REGION Network 16: Call the Event Manager logic for EM alarms
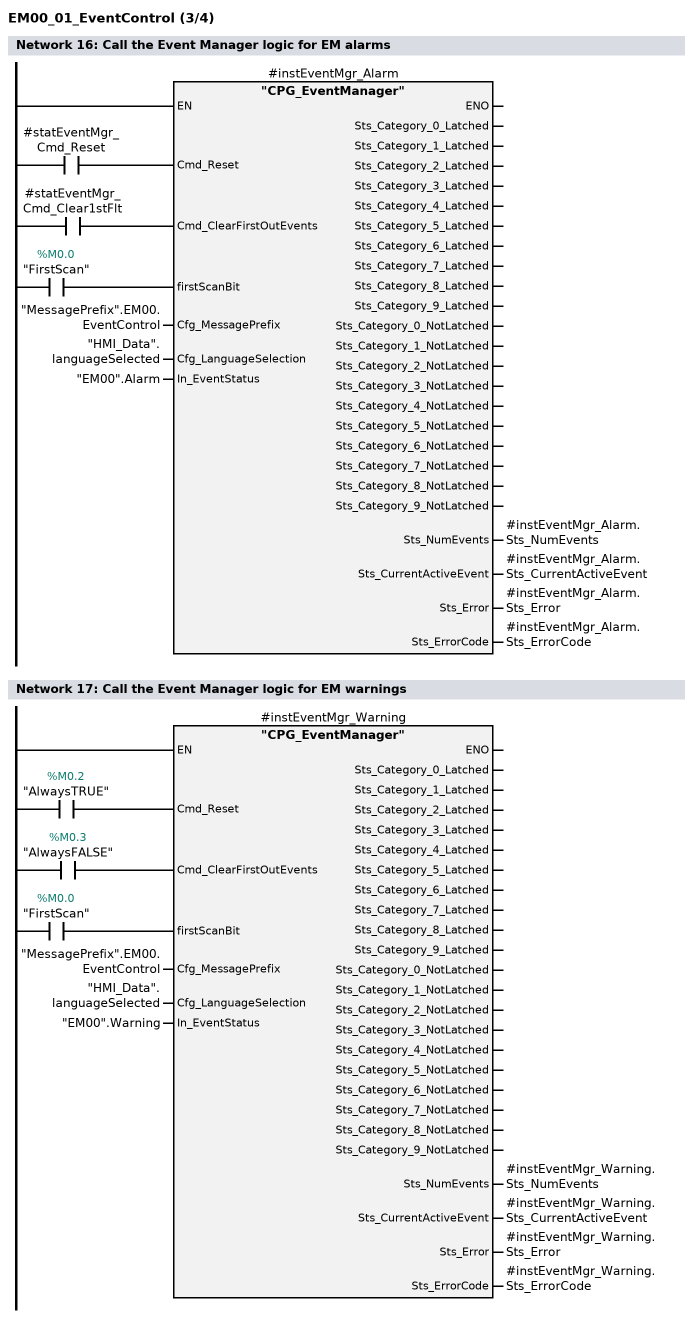
   RUNG wire#powerrail
      #instEventMgr_Alarm(Cmd_Reset := wire#w1, Cmd_ClearFirstOutEvents := wire#w2, firstScanBit := wire#w3, Cfg_MessagePrefix := "MessagePrefix".EM00.EventControl, Cfg_LanguageSelection := "HMI_Data".languageSelected, In_EventStatus := "EM00".Alarm, Sts_Category_0_Latched =>, Sts_Category_1_Latched =>, Sts_Category_2_Latched =>, Sts_Category_3_Latched =>, Sts_Category_4_Latched =>, Sts_Category_5_Latched =>, Sts_Category_6_Latched =>, Sts_Category_7_Latched =>, Sts_Category_8_Latched =>, Sts_Category_9_Latched =>, Sts_Category_0_NotLatched =>, Sts_Category_1_NotLatched =>, Sts_Category_2_NotLatched =>, Sts_Category_3_NotLatched =>, Sts_Category_4_NotLatched =>, Sts_Category_5_NotLatched =>, Sts_Category_6_NotLatched =>, Sts_Category_7_NotLatched =>, Sts_Category_8_NotLatched =>, Sts_Category_9_NotLatched =>, Sts_NumEvents => #instEventMgr_Alarm.Sts_NumEvents, Sts_CurrentActiveEvent => #instEventMgr_Alarm.Sts_CurrentActiveEvent, Sts_Error => #instEventMgr_Alarm.Sts_Error, Sts_ErrorCode => #instEventMgr_Alarm.Sts_ErrorCode)
   END_RUNG
   RUNG wire#powerrail
      Contact( #statEventMgr_Cmd_Reset )
   END_RUNG wire#w1
   RUNG wire#powerrail
      Contact( #statEventMgr_Cmd_Clear1stFlt )
   END_RUNG wire#w2
   RUNG wire#powerrail
      Contact( "FirstScan" )
   END_RUNG wire#w3
   // the same network as SCL:
   #instEventMgr_Alarm(Cmd_Reset := #statEventMgr_Cmd_Reset,   // "CPG_EventManager"
                       Cmd_ClearFirstOutEvents := #statEventMgr_Cmd_Clear1stFlt,
                       firstScanBit := "FirstScan",
                       Cfg_MessagePrefix := "MessagePrefix".EM00.EventControl,
                       Cfg_LanguageSelection := "HMI_Data".languageSelected,
                       In_EventStatus := "EM00".Alarm,
                       Sts_NumEvents => #instEventMgr_Alarm.Sts_NumEvents,
                       Sts_CurrentActiveEvent => #instEventMgr_Alarm.Sts_CurrentActiveEvent,
                       Sts_Error => #instEventMgr_Alarm.Sts_Error,
                       Sts_ErrorCode => #instEventMgr_Alarm.Sts_ErrorCode);
END_REGION

REGION Network 17: Call the Event Manager logic for EM warnings
   RUNG wire#powerrail
      #instEventMgr_Warning(Cmd_Reset := wire#w1, Cmd_ClearFirstOutEvents := wire#w2, firstScanBit := wire#w3, Cfg_MessagePrefix := "MessagePrefix".EM00.EventControl, Cfg_LanguageSelection := "HMI_Data".languageSelected, In_EventStatus := "EM00".Warning, Sts_Category_0_Latched =>, Sts_Category_1_Latched =>, Sts_Category_2_Latched =>, Sts_Category_3_Latched =>, Sts_Category_4_Latched =>, Sts_Category_5_Latched =>, Sts_Category_6_Latched =>, Sts_Category_7_Latched =>, Sts_Category_8_Latched =>, Sts_Category_9_Latched =>, Sts_Category_0_NotLatched =>, Sts_Category_1_NotLatched =>, Sts_Category_2_NotLatched =>, Sts_Category_3_NotLatched =>, Sts_Category_4_NotLatched =>, Sts_Category_5_NotLatched =>, Sts_Category_6_NotLatched =>, Sts_Category_7_NotLatched =>, Sts_Category_8_NotLatched =>, Sts_Category_9_NotLatched =>, Sts_NumEvents => #instEventMgr_Warning.Sts_NumEvents, Sts_CurrentActiveEvent => #instEventMgr_Warning.Sts_CurrentActiveEvent, Sts_Error => #instEventMgr_Warning.Sts_Error, Sts_ErrorCode => #instEventMgr_Warning.Sts_ErrorCode)
   END_RUNG
   RUNG wire#powerrail
      Contact( "AlwaysTRUE" )
   END_RUNG wire#w1
   RUNG wire#powerrail
      Contact( "AlwaysFALSE" )
   END_RUNG wire#w2
   RUNG wire#powerrail
      Contact( "FirstScan" )
   END_RUNG wire#w3
   // the same network as SCL:
   #instEventMgr_Warning(Cmd_Reset := "AlwaysTRUE",   // "CPG_EventManager"
                         Cmd_ClearFirstOutEvents := "AlwaysFALSE",
                         firstScanBit := "FirstScan",
                         Cfg_MessagePrefix := "MessagePrefix".EM00.EventControl,
                         Cfg_LanguageSelection := "HMI_Data".languageSelected,
                         In_EventStatus := "EM00".Warning,
                         Sts_NumEvents => #instEventMgr_Warning.Sts_NumEvents,
                         Sts_CurrentActiveEvent => #instEventMgr_Warning.Sts_CurrentActiveEvent,
                         Sts_Error => #instEventMgr_Warning.Sts_Error,
                         Sts_ErrorCode => #instEventMgr_Warning.Sts_ErrorCode);
END_REGION

REGION Network 18: Call the Event Manager logic for EM status
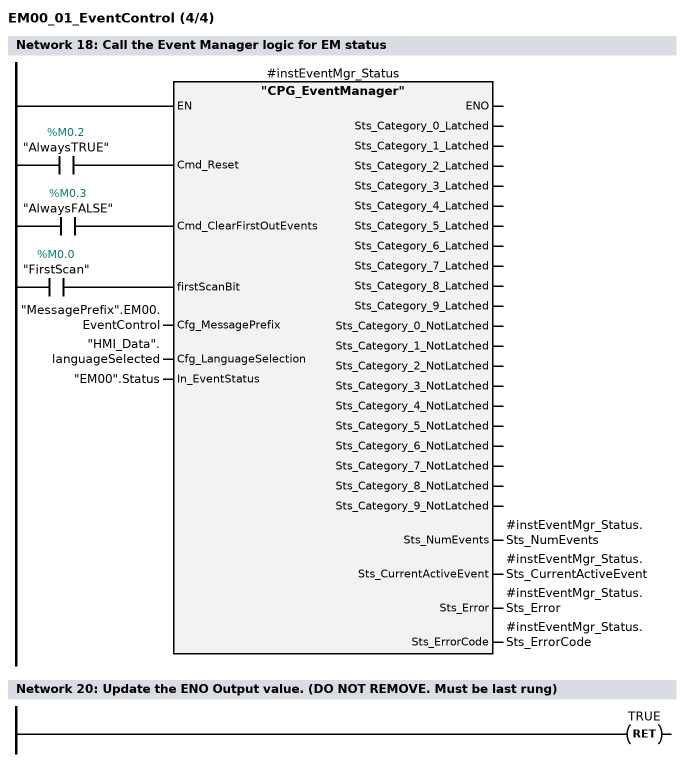
   RUNG wire#powerrail
      #instEventMgr_Status(Cmd_Reset := wire#w1, Cmd_ClearFirstOutEvents := wire#w2, firstScanBit := wire#w3, Cfg_MessagePrefix := "MessagePrefix".EM00.EventControl, Cfg_LanguageSelection := "HMI_Data".languageSelected, In_EventStatus := "EM00".Status, Sts_Category_0_Latched =>, Sts_Category_1_Latched =>, Sts_Category_2_Latched =>, Sts_Category_3_Latched =>, Sts_Category_4_Latched =>, Sts_Category_5_Latched =>, Sts_Category_6_Latched =>, Sts_Category_7_Latched =>, Sts_Category_8_Latched =>, Sts_Category_9_Latched =>, Sts_Category_0_NotLatched =>, Sts_Category_1_NotLatched =>, Sts_Category_2_NotLatched =>, Sts_Category_3_NotLatched =>, Sts_Category_4_NotLatched =>, Sts_Category_5_NotLatched =>, Sts_Category_6_NotLatched =>, Sts_Category_7_NotLatched =>, Sts_Category_8_NotLatched =>, Sts_Category_9_NotLatched =>, Sts_NumEvents => #instEventMgr_Status.Sts_NumEvents, Sts_CurrentActiveEvent => #instEventMgr_Status.Sts_CurrentActiveEvent, Sts_Error => #instEventMgr_Status.Sts_Error, Sts_ErrorCode => #instEventMgr_Status.Sts_ErrorCode)
   END_RUNG
   RUNG wire#powerrail
      Contact( "AlwaysTRUE" )
   END_RUNG wire#w1
   RUNG wire#powerrail
      Contact( "AlwaysFALSE" )
   END_RUNG wire#w2
   RUNG wire#powerrail
      Contact( "FirstScan" )
   END_RUNG wire#w3
   // the same network as SCL:
   #instEventMgr_Status(Cmd_Reset := "AlwaysTRUE",   // "CPG_EventManager"
                        Cmd_ClearFirstOutEvents := "AlwaysFALSE",
                        firstScanBit := "FirstScan",
                        Cfg_MessagePrefix := "MessagePrefix".EM00.EventControl,
                        Cfg_LanguageSelection := "HMI_Data".languageSelected,
                        In_EventStatus := "EM00".Status,
                        Sts_NumEvents => #instEventMgr_Status.Sts_NumEvents,
                        Sts_CurrentActiveEvent => #instEventMgr_Status.Sts_CurrentActiveEvent,
                        Sts_Error => #instEventMgr_Status.Sts_Error,
                        Sts_ErrorCode => #instEventMgr_Status.Sts_ErrorCode);
END_REGION

REGION Network 20: Update the ENO Output value. (DO NOT REMOVE. Must be last rung)
   RUNG wire#powerrail
      ReturnCoil( TRUE )
   END_RUNG
   // the same network as SCL:
   ENO := TRUE;
   RETURN;
END_REGION
END_FUNCTION_BLOCK

FUNCTION_BLOCK "EM00_02_PackML_ModuleSum"   // FB31642, LAD
TITLE = EM00_02_PackML_ModuleSummation
{ S7_Optimized_Access := 'TRUE' }
AUTHOR : tech.team.motioncontrol@siemens.com
FAMILY : CPG
VERSION : 1.1
// Support: tech.team.motioncontrol@siemens.com
// stored: AutoNumber true, IsIECCheckEnabled false, IsRetainMemResEnabled false, MemoryReserve 100, SetENOAutomatically false, UDAEnableTagReadback false
   VAR
      statDummyBool { ExternalAccessible := 'False'; ExternalVisible := 'False'; ExternalWritable := 'False'} : Bool;   // dummy bool - placeholder
   END_VAR
BEGIN

REGION Network 1: EM - Reset Command
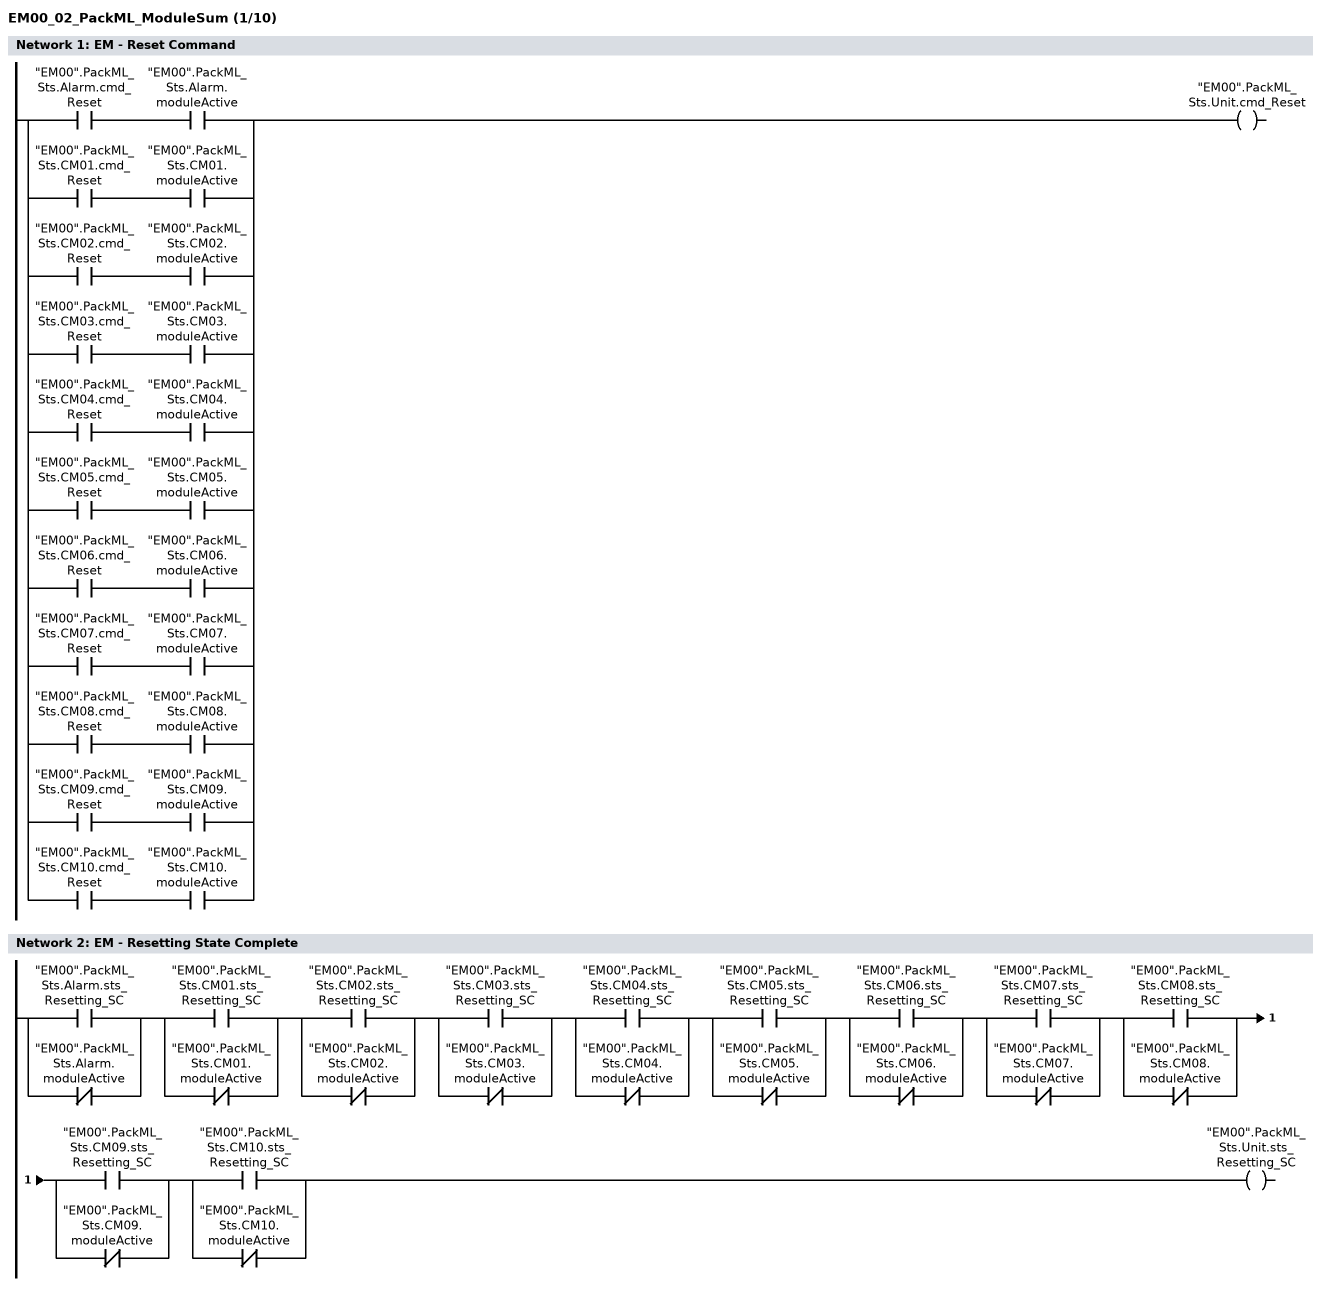
   RUNG wire#powerrail
      Contact( "EM00".PackML_Sts.Alarm.cmd_Reset )
      Contact( "EM00".PackML_Sts.Alarm.moduleActive )
      wire#w1
      Coil( "EM00".PackML_Sts.Unit.cmd_Reset )
   END_RUNG
   RUNG wire#powerrail
      Contact( "EM00".PackML_Sts.CM01.cmd_Reset )
      Contact( "EM00".PackML_Sts.CM01.moduleActive )
   END_RUNG wire#w1
   RUNG wire#powerrail
      Contact( "EM00".PackML_Sts.CM02.cmd_Reset )
      Contact( "EM00".PackML_Sts.CM02.moduleActive )
   END_RUNG wire#w1
   RUNG wire#powerrail
      Contact( "EM00".PackML_Sts.CM03.cmd_Reset )
      Contact( "EM00".PackML_Sts.CM03.moduleActive )
   END_RUNG wire#w1
   RUNG wire#powerrail
      Contact( "EM00".PackML_Sts.CM04.cmd_Reset )
      Contact( "EM00".PackML_Sts.CM04.moduleActive )
   END_RUNG wire#w1
   RUNG wire#powerrail
      Contact( "EM00".PackML_Sts.CM05.cmd_Reset )
      Contact( "EM00".PackML_Sts.CM05.moduleActive )
   END_RUNG wire#w1
   RUNG wire#powerrail
      Contact( "EM00".PackML_Sts.CM06.cmd_Reset )
      Contact( "EM00".PackML_Sts.CM06.moduleActive )
   END_RUNG wire#w1
   RUNG wire#powerrail
      Contact( "EM00".PackML_Sts.CM07.cmd_Reset )
      Contact( "EM00".PackML_Sts.CM07.moduleActive )
   END_RUNG wire#w1
   RUNG wire#powerrail
      Contact( "EM00".PackML_Sts.CM08.cmd_Reset )
      Contact( "EM00".PackML_Sts.CM08.moduleActive )
   END_RUNG wire#w1
   RUNG wire#powerrail
      Contact( "EM00".PackML_Sts.CM09.cmd_Reset )
      Contact( "EM00".PackML_Sts.CM09.moduleActive )
   END_RUNG wire#w1
   RUNG wire#powerrail
      Contact( "EM00".PackML_Sts.CM10.cmd_Reset )
      Contact( "EM00".PackML_Sts.CM10.moduleActive )
   END_RUNG wire#w1
   // the same network as SCL:
   "EM00".PackML_Sts.Unit.cmd_Reset := ("EM00".PackML_Sts.Alarm.cmd_Reset AND "EM00".PackML_Sts.Alarm.moduleActive) OR ("EM00".PackML_Sts.CM01.cmd_Reset AND "EM00".PackML_Sts.CM01.moduleActive) OR ("EM00".PackML_Sts.CM02.cmd_Reset AND "EM00".PackML_Sts.CM02.moduleActive) OR ("EM00".PackML_Sts.CM03.cmd_Reset AND "EM00".PackML_Sts.CM03.moduleActive) OR ("EM00".PackML_Sts.CM04.cmd_Reset AND "EM00".PackML_Sts.CM04.moduleActive) OR ("EM00".PackML_Sts.CM05.cmd_Reset AND "EM00".PackML_Sts.CM05.moduleActive) OR ("EM00".PackML_Sts.CM06.cmd_Reset AND "EM00".PackML_Sts.CM06.moduleActive) OR ("EM00".PackML_Sts.CM07.cmd_Reset AND "EM00".PackML_Sts.CM07.moduleActive) OR ("EM00".PackML_Sts.CM08.cmd_Reset AND "EM00".PackML_Sts.CM08.moduleActive) OR ("EM00".PackML_Sts.CM09.cmd_Reset AND "EM00".PackML_Sts.CM09.moduleActive) OR ("EM00".PackML_Sts.CM10.cmd_Reset AND "EM00".PackML_Sts.CM10.moduleActive);
END_REGION

REGION Network 2: EM - Resetting State Complete
   RUNG wire#powerrail
      Contact( "EM00".PackML_Sts.Alarm.sts_Resetting_SC )
      wire#w1
      Contact( "EM00".PackML_Sts.CM01.sts_Resetting_SC )
      wire#w2
      Contact( "EM00".PackML_Sts.CM02.sts_Resetting_SC )
      wire#w3
      Contact( "EM00".PackML_Sts.CM03.sts_Resetting_SC )
      wire#w4
      Contact( "EM00".PackML_Sts.CM04.sts_Resetting_SC )
      wire#w5
      Contact( "EM00".PackML_Sts.CM05.sts_Resetting_SC )
      wire#w6
      Contact( "EM00".PackML_Sts.CM06.sts_Resetting_SC )
      wire#w7
      Contact( "EM00".PackML_Sts.CM07.sts_Resetting_SC )
      wire#w8
      Contact( "EM00".PackML_Sts.CM08.sts_Resetting_SC )
      wire#w9
      Contact( "EM00".PackML_Sts.CM09.sts_Resetting_SC )
      wire#w10
      Contact( "EM00".PackML_Sts.CM10.sts_Resetting_SC )
      wire#w11
      Coil( "EM00".PackML_Sts.Unit.sts_Resetting_SC )
   END_RUNG
   RUNG wire#powerrail
      I_Contact( "EM00".PackML_Sts.Alarm.moduleActive )
   END_RUNG wire#w1
   RUNG wire#w1
      I_Contact( "EM00".PackML_Sts.CM01.moduleActive )
   END_RUNG wire#w2
   RUNG wire#w2
      I_Contact( "EM00".PackML_Sts.CM02.moduleActive )
   END_RUNG wire#w3
   RUNG wire#w3
      I_Contact( "EM00".PackML_Sts.CM03.moduleActive )
   END_RUNG wire#w4
   RUNG wire#w4
      I_Contact( "EM00".PackML_Sts.CM04.moduleActive )
   END_RUNG wire#w5
   RUNG wire#w5
      I_Contact( "EM00".PackML_Sts.CM05.moduleActive )
   END_RUNG wire#w6
   RUNG wire#w6
      I_Contact( "EM00".PackML_Sts.CM06.moduleActive )
   END_RUNG wire#w7
   RUNG wire#w7
      I_Contact( "EM00".PackML_Sts.CM07.moduleActive )
   END_RUNG wire#w8
   RUNG wire#w8
      I_Contact( "EM00".PackML_Sts.CM08.moduleActive )
   END_RUNG wire#w9
   RUNG wire#w9
      I_Contact( "EM00".PackML_Sts.CM09.moduleActive )
   END_RUNG wire#w10
   RUNG wire#w10
      I_Contact( "EM00".PackML_Sts.CM10.moduleActive )
   END_RUNG wire#w11
   // the same network as SCL:
   "EM00".PackML_Sts.Unit.sts_Resetting_SC := ("EM00".PackML_Sts.Alarm.sts_Resetting_SC OR NOT "EM00".PackML_Sts.Alarm.moduleActive) AND ("EM00".PackML_Sts.CM01.sts_Resetting_SC OR NOT "EM00".PackML_Sts.CM01.moduleActive) AND ("EM00".PackML_Sts.CM02.sts_Resetting_SC OR NOT "EM00".PackML_Sts.CM02.moduleActive) AND ("EM00".PackML_Sts.CM03.sts_Resetting_SC OR NOT "EM00".PackML_Sts.CM03.moduleActive) AND ("EM00".PackML_Sts.CM04.sts_Resetting_SC OR NOT "EM00".PackML_Sts.CM04.moduleActive) AND ("EM00".PackML_Sts.CM05.sts_Resetting_SC OR NOT "EM00".PackML_Sts.CM05.moduleActive) AND ("EM00".PackML_Sts.CM06.sts_Resetting_SC OR NOT "EM00".PackML_Sts.CM06.moduleActive) AND ("EM00".PackML_Sts.CM07.sts_Resetting_SC OR NOT "EM00".PackML_Sts.CM07.moduleActive) AND ("EM00".PackML_Sts.CM08.sts_Resetting_SC OR NOT "EM00".PackML_Sts.CM08.moduleActive) AND ("EM00".PackML_Sts.CM09.sts_Resetting_SC OR NOT "EM00".PackML_Sts.CM09.moduleActive) AND ("EM00".PackML_Sts.CM10.sts_Resetting_SC OR NOT "EM00".PackML_Sts.CM10.moduleActive);
END_REGION

REGION Network 3: EM - Start Command
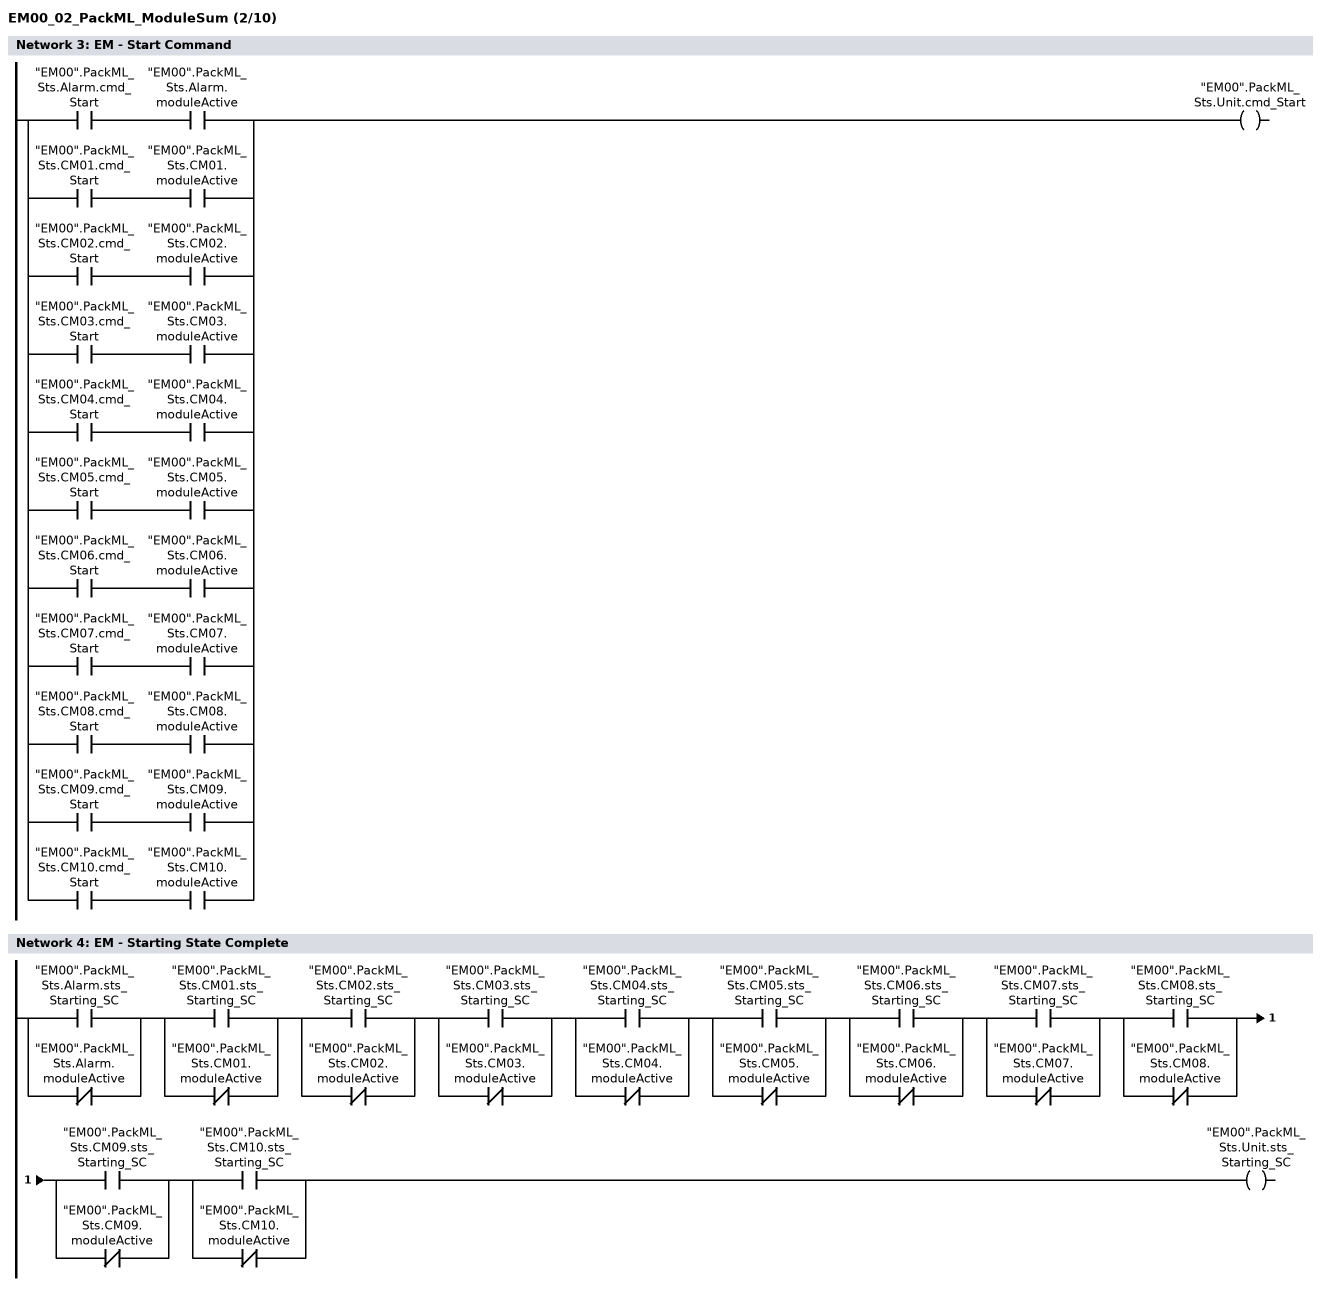
   RUNG wire#powerrail
      Contact( "EM00".PackML_Sts.Alarm.cmd_Start )
      Contact( "EM00".PackML_Sts.Alarm.moduleActive )
      wire#w1
      Coil( "EM00".PackML_Sts.Unit.cmd_Start )
   END_RUNG
   RUNG wire#powerrail
      Contact( "EM00".PackML_Sts.CM01.cmd_Start )
      Contact( "EM00".PackML_Sts.CM01.moduleActive )
   END_RUNG wire#w1
   RUNG wire#powerrail
      Contact( "EM00".PackML_Sts.CM02.cmd_Start )
      Contact( "EM00".PackML_Sts.CM02.moduleActive )
   END_RUNG wire#w1
   RUNG wire#powerrail
      Contact( "EM00".PackML_Sts.CM03.cmd_Start )
      Contact( "EM00".PackML_Sts.CM03.moduleActive )
   END_RUNG wire#w1
   RUNG wire#powerrail
      Contact( "EM00".PackML_Sts.CM04.cmd_Start )
      Contact( "EM00".PackML_Sts.CM04.moduleActive )
   END_RUNG wire#w1
   RUNG wire#powerrail
      Contact( "EM00".PackML_Sts.CM05.cmd_Start )
      Contact( "EM00".PackML_Sts.CM05.moduleActive )
   END_RUNG wire#w1
   RUNG wire#powerrail
      Contact( "EM00".PackML_Sts.CM06.cmd_Start )
      Contact( "EM00".PackML_Sts.CM06.moduleActive )
   END_RUNG wire#w1
   RUNG wire#powerrail
      Contact( "EM00".PackML_Sts.CM07.cmd_Start )
      Contact( "EM00".PackML_Sts.CM07.moduleActive )
   END_RUNG wire#w1
   RUNG wire#powerrail
      Contact( "EM00".PackML_Sts.CM08.cmd_Start )
      Contact( "EM00".PackML_Sts.CM08.moduleActive )
   END_RUNG wire#w1
   RUNG wire#powerrail
      Contact( "EM00".PackML_Sts.CM09.cmd_Start )
      Contact( "EM00".PackML_Sts.CM09.moduleActive )
   END_RUNG wire#w1
   RUNG wire#powerrail
      Contact( "EM00".PackML_Sts.CM10.cmd_Start )
      Contact( "EM00".PackML_Sts.CM10.moduleActive )
   END_RUNG wire#w1
   // the same network as SCL:
   "EM00".PackML_Sts.Unit.cmd_Start := ("EM00".PackML_Sts.Alarm.cmd_Start AND "EM00".PackML_Sts.Alarm.moduleActive) OR ("EM00".PackML_Sts.CM01.cmd_Start AND "EM00".PackML_Sts.CM01.moduleActive) OR ("EM00".PackML_Sts.CM02.cmd_Start AND "EM00".PackML_Sts.CM02.moduleActive) OR ("EM00".PackML_Sts.CM03.cmd_Start AND "EM00".PackML_Sts.CM03.moduleActive) OR ("EM00".PackML_Sts.CM04.cmd_Start AND "EM00".PackML_Sts.CM04.moduleActive) OR ("EM00".PackML_Sts.CM05.cmd_Start AND "EM00".PackML_Sts.CM05.moduleActive) OR ("EM00".PackML_Sts.CM06.cmd_Start AND "EM00".PackML_Sts.CM06.moduleActive) OR ("EM00".PackML_Sts.CM07.cmd_Start AND "EM00".PackML_Sts.CM07.moduleActive) OR ("EM00".PackML_Sts.CM08.cmd_Start AND "EM00".PackML_Sts.CM08.moduleActive) OR ("EM00".PackML_Sts.CM09.cmd_Start AND "EM00".PackML_Sts.CM09.moduleActive) OR ("EM00".PackML_Sts.CM10.cmd_Start AND "EM00".PackML_Sts.CM10.moduleActive);
END_REGION

REGION Network 4: EM - Starting State Complete
   RUNG wire#powerrail
      Contact( "EM00".PackML_Sts.Alarm.sts_Starting_SC )
      wire#w1
      Contact( "EM00".PackML_Sts.CM01.sts_Starting_SC )
      wire#w2
      Contact( "EM00".PackML_Sts.CM02.sts_Starting_SC )
      wire#w3
      Contact( "EM00".PackML_Sts.CM03.sts_Starting_SC )
      wire#w4
      Contact( "EM00".PackML_Sts.CM04.sts_Starting_SC )
      wire#w5
      Contact( "EM00".PackML_Sts.CM05.sts_Starting_SC )
      wire#w6
      Contact( "EM00".PackML_Sts.CM06.sts_Starting_SC )
      wire#w7
      Contact( "EM00".PackML_Sts.CM07.sts_Starting_SC )
      wire#w8
      Contact( "EM00".PackML_Sts.CM08.sts_Starting_SC )
      wire#w9
      Contact( "EM00".PackML_Sts.CM09.sts_Starting_SC )
      wire#w10
      Contact( "EM00".PackML_Sts.CM10.sts_Starting_SC )
      wire#w11
      Coil( "EM00".PackML_Sts.Unit.sts_Starting_SC )
   END_RUNG
   RUNG wire#powerrail
      I_Contact( "EM00".PackML_Sts.Alarm.moduleActive )
   END_RUNG wire#w1
   RUNG wire#w1
      I_Contact( "EM00".PackML_Sts.CM01.moduleActive )
   END_RUNG wire#w2
   RUNG wire#w2
      I_Contact( "EM00".PackML_Sts.CM02.moduleActive )
   END_RUNG wire#w3
   RUNG wire#w3
      I_Contact( "EM00".PackML_Sts.CM03.moduleActive )
   END_RUNG wire#w4
   RUNG wire#w4
      I_Contact( "EM00".PackML_Sts.CM04.moduleActive )
   END_RUNG wire#w5
   RUNG wire#w5
      I_Contact( "EM00".PackML_Sts.CM05.moduleActive )
   END_RUNG wire#w6
   RUNG wire#w6
      I_Contact( "EM00".PackML_Sts.CM06.moduleActive )
   END_RUNG wire#w7
   RUNG wire#w7
      I_Contact( "EM00".PackML_Sts.CM07.moduleActive )
   END_RUNG wire#w8
   RUNG wire#w8
      I_Contact( "EM00".PackML_Sts.CM08.moduleActive )
   END_RUNG wire#w9
   RUNG wire#w9
      I_Contact( "EM00".PackML_Sts.CM09.moduleActive )
   END_RUNG wire#w10
   RUNG wire#w10
      I_Contact( "EM00".PackML_Sts.CM10.moduleActive )
   END_RUNG wire#w11
   // the same network as SCL:
   "EM00".PackML_Sts.Unit.sts_Starting_SC := ("EM00".PackML_Sts.Alarm.sts_Starting_SC OR NOT "EM00".PackML_Sts.Alarm.moduleActive) AND ("EM00".PackML_Sts.CM01.sts_Starting_SC OR NOT "EM00".PackML_Sts.CM01.moduleActive) AND ("EM00".PackML_Sts.CM02.sts_Starting_SC OR NOT "EM00".PackML_Sts.CM02.moduleActive) AND ("EM00".PackML_Sts.CM03.sts_Starting_SC OR NOT "EM00".PackML_Sts.CM03.moduleActive) AND ("EM00".PackML_Sts.CM04.sts_Starting_SC OR NOT "EM00".PackML_Sts.CM04.moduleActive) AND ("EM00".PackML_Sts.CM05.sts_Starting_SC OR NOT "EM00".PackML_Sts.CM05.moduleActive) AND ("EM00".PackML_Sts.CM06.sts_Starting_SC OR NOT "EM00".PackML_Sts.CM06.moduleActive) AND ("EM00".PackML_Sts.CM07.sts_Starting_SC OR NOT "EM00".PackML_Sts.CM07.moduleActive) AND ("EM00".PackML_Sts.CM08.sts_Starting_SC OR NOT "EM00".PackML_Sts.CM08.moduleActive) AND ("EM00".PackML_Sts.CM09.sts_Starting_SC OR NOT "EM00".PackML_Sts.CM09.moduleActive) AND ("EM00".PackML_Sts.CM10.sts_Starting_SC OR NOT "EM00".PackML_Sts.CM10.moduleActive);
END_REGION

REGION Network 5: EM - Stop Command
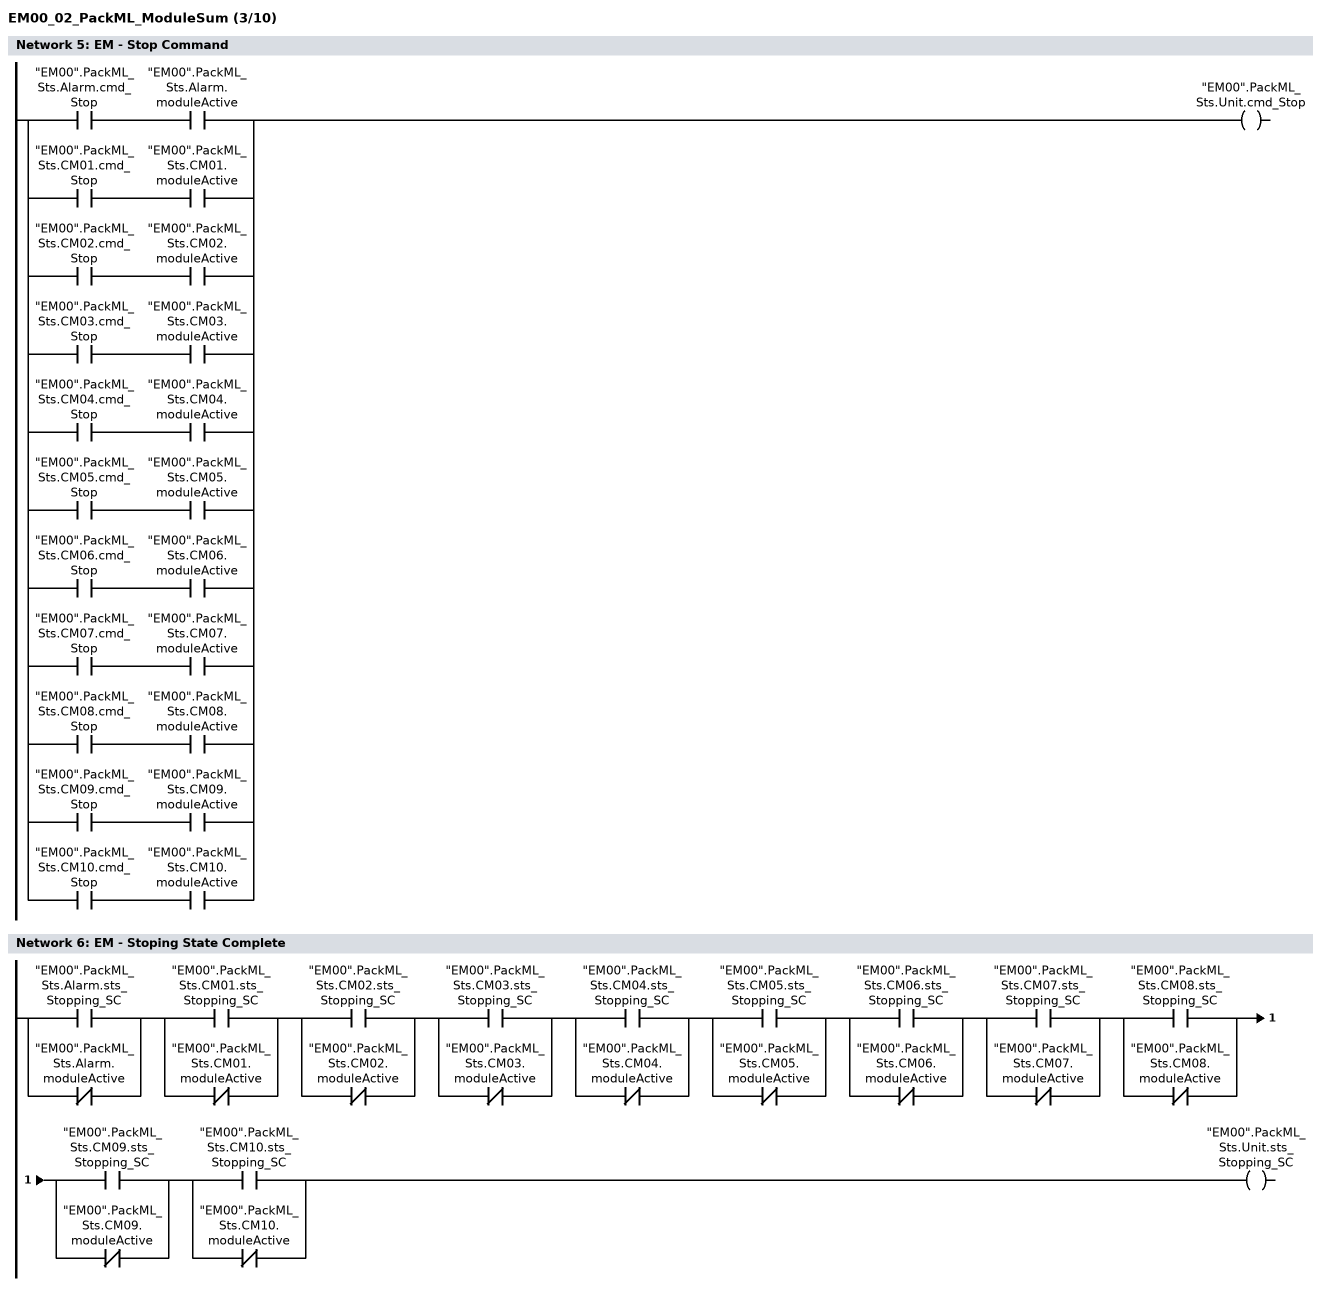
   RUNG wire#powerrail
      Contact( "EM00".PackML_Sts.Alarm.cmd_Stop )
      Contact( "EM00".PackML_Sts.Alarm.moduleActive )
      wire#w1
      Coil( "EM00".PackML_Sts.Unit.cmd_Stop )
   END_RUNG
   RUNG wire#powerrail
      Contact( "EM00".PackML_Sts.CM01.cmd_Stop )
      Contact( "EM00".PackML_Sts.CM01.moduleActive )
   END_RUNG wire#w1
   RUNG wire#powerrail
      Contact( "EM00".PackML_Sts.CM02.cmd_Stop )
      Contact( "EM00".PackML_Sts.CM02.moduleActive )
   END_RUNG wire#w1
   RUNG wire#powerrail
      Contact( "EM00".PackML_Sts.CM03.cmd_Stop )
      Contact( "EM00".PackML_Sts.CM03.moduleActive )
   END_RUNG wire#w1
   RUNG wire#powerrail
      Contact( "EM00".PackML_Sts.CM04.cmd_Stop )
      Contact( "EM00".PackML_Sts.CM04.moduleActive )
   END_RUNG wire#w1
   RUNG wire#powerrail
      Contact( "EM00".PackML_Sts.CM05.cmd_Stop )
      Contact( "EM00".PackML_Sts.CM05.moduleActive )
   END_RUNG wire#w1
   RUNG wire#powerrail
      Contact( "EM00".PackML_Sts.CM06.cmd_Stop )
      Contact( "EM00".PackML_Sts.CM06.moduleActive )
   END_RUNG wire#w1
   RUNG wire#powerrail
      Contact( "EM00".PackML_Sts.CM07.cmd_Stop )
      Contact( "EM00".PackML_Sts.CM07.moduleActive )
   END_RUNG wire#w1
   RUNG wire#powerrail
      Contact( "EM00".PackML_Sts.CM08.cmd_Stop )
      Contact( "EM00".PackML_Sts.CM08.moduleActive )
   END_RUNG wire#w1
   RUNG wire#powerrail
      Contact( "EM00".PackML_Sts.CM09.cmd_Stop )
      Contact( "EM00".PackML_Sts.CM09.moduleActive )
   END_RUNG wire#w1
   RUNG wire#powerrail
      Contact( "EM00".PackML_Sts.CM10.cmd_Stop )
      Contact( "EM00".PackML_Sts.CM10.moduleActive )
   END_RUNG wire#w1
   // the same network as SCL:
   "EM00".PackML_Sts.Unit.cmd_Stop := ("EM00".PackML_Sts.Alarm.cmd_Stop AND "EM00".PackML_Sts.Alarm.moduleActive) OR ("EM00".PackML_Sts.CM01.cmd_Stop AND "EM00".PackML_Sts.CM01.moduleActive) OR ("EM00".PackML_Sts.CM02.cmd_Stop AND "EM00".PackML_Sts.CM02.moduleActive) OR ("EM00".PackML_Sts.CM03.cmd_Stop AND "EM00".PackML_Sts.CM03.moduleActive) OR ("EM00".PackML_Sts.CM04.cmd_Stop AND "EM00".PackML_Sts.CM04.moduleActive) OR ("EM00".PackML_Sts.CM05.cmd_Stop AND "EM00".PackML_Sts.CM05.moduleActive) OR ("EM00".PackML_Sts.CM06.cmd_Stop AND "EM00".PackML_Sts.CM06.moduleActive) OR ("EM00".PackML_Sts.CM07.cmd_Stop AND "EM00".PackML_Sts.CM07.moduleActive) OR ("EM00".PackML_Sts.CM08.cmd_Stop AND "EM00".PackML_Sts.CM08.moduleActive) OR ("EM00".PackML_Sts.CM09.cmd_Stop AND "EM00".PackML_Sts.CM09.moduleActive) OR ("EM00".PackML_Sts.CM10.cmd_Stop AND "EM00".PackML_Sts.CM10.moduleActive);
END_REGION

REGION Network 6: EM - Stoping State Complete
   RUNG wire#powerrail
      Contact( "EM00".PackML_Sts.Alarm.sts_Stopping_SC )
      wire#w1
      Contact( "EM00".PackML_Sts.CM01.sts_Stopping_SC )
      wire#w2
      Contact( "EM00".PackML_Sts.CM02.sts_Stopping_SC )
      wire#w3
      Contact( "EM00".PackML_Sts.CM03.sts_Stopping_SC )
      wire#w4
      Contact( "EM00".PackML_Sts.CM04.sts_Stopping_SC )
      wire#w5
      Contact( "EM00".PackML_Sts.CM05.sts_Stopping_SC )
      wire#w6
      Contact( "EM00".PackML_Sts.CM06.sts_Stopping_SC )
      wire#w7
      Contact( "EM00".PackML_Sts.CM07.sts_Stopping_SC )
      wire#w8
      Contact( "EM00".PackML_Sts.CM08.sts_Stopping_SC )
      wire#w9
      Contact( "EM00".PackML_Sts.CM09.sts_Stopping_SC )
      wire#w10
      Contact( "EM00".PackML_Sts.CM10.sts_Stopping_SC )
      wire#w11
      Coil( "EM00".PackML_Sts.Unit.sts_Stopping_SC )
   END_RUNG
   RUNG wire#powerrail
      I_Contact( "EM00".PackML_Sts.Alarm.moduleActive )
   END_RUNG wire#w1
   RUNG wire#w1
      I_Contact( "EM00".PackML_Sts.CM01.moduleActive )
   END_RUNG wire#w2
   RUNG wire#w2
      I_Contact( "EM00".PackML_Sts.CM02.moduleActive )
   END_RUNG wire#w3
   RUNG wire#w3
      I_Contact( "EM00".PackML_Sts.CM03.moduleActive )
   END_RUNG wire#w4
   RUNG wire#w4
      I_Contact( "EM00".PackML_Sts.CM04.moduleActive )
   END_RUNG wire#w5
   RUNG wire#w5
      I_Contact( "EM00".PackML_Sts.CM05.moduleActive )
   END_RUNG wire#w6
   RUNG wire#w6
      I_Contact( "EM00".PackML_Sts.CM06.moduleActive )
   END_RUNG wire#w7
   RUNG wire#w7
      I_Contact( "EM00".PackML_Sts.CM07.moduleActive )
   END_RUNG wire#w8
   RUNG wire#w8
      I_Contact( "EM00".PackML_Sts.CM08.moduleActive )
   END_RUNG wire#w9
   RUNG wire#w9
      I_Contact( "EM00".PackML_Sts.CM09.moduleActive )
   END_RUNG wire#w10
   RUNG wire#w10
      I_Contact( "EM00".PackML_Sts.CM10.moduleActive )
   END_RUNG wire#w11
   // the same network as SCL:
   "EM00".PackML_Sts.Unit.sts_Stopping_SC := ("EM00".PackML_Sts.Alarm.sts_Stopping_SC OR NOT "EM00".PackML_Sts.Alarm.moduleActive) AND ("EM00".PackML_Sts.CM01.sts_Stopping_SC OR NOT "EM00".PackML_Sts.CM01.moduleActive) AND ("EM00".PackML_Sts.CM02.sts_Stopping_SC OR NOT "EM00".PackML_Sts.CM02.moduleActive) AND ("EM00".PackML_Sts.CM03.sts_Stopping_SC OR NOT "EM00".PackML_Sts.CM03.moduleActive) AND ("EM00".PackML_Sts.CM04.sts_Stopping_SC OR NOT "EM00".PackML_Sts.CM04.moduleActive) AND ("EM00".PackML_Sts.CM05.sts_Stopping_SC OR NOT "EM00".PackML_Sts.CM05.moduleActive) AND ("EM00".PackML_Sts.CM06.sts_Stopping_SC OR NOT "EM00".PackML_Sts.CM06.moduleActive) AND ("EM00".PackML_Sts.CM07.sts_Stopping_SC OR NOT "EM00".PackML_Sts.CM07.moduleActive) AND ("EM00".PackML_Sts.CM08.sts_Stopping_SC OR NOT "EM00".PackML_Sts.CM08.moduleActive) AND ("EM00".PackML_Sts.CM09.sts_Stopping_SC OR NOT "EM00".PackML_Sts.CM09.moduleActive) AND ("EM00".PackML_Sts.CM10.sts_Stopping_SC OR NOT "EM00".PackML_Sts.CM10.moduleActive);
END_REGION

REGION Network 7: EM - Hold Command
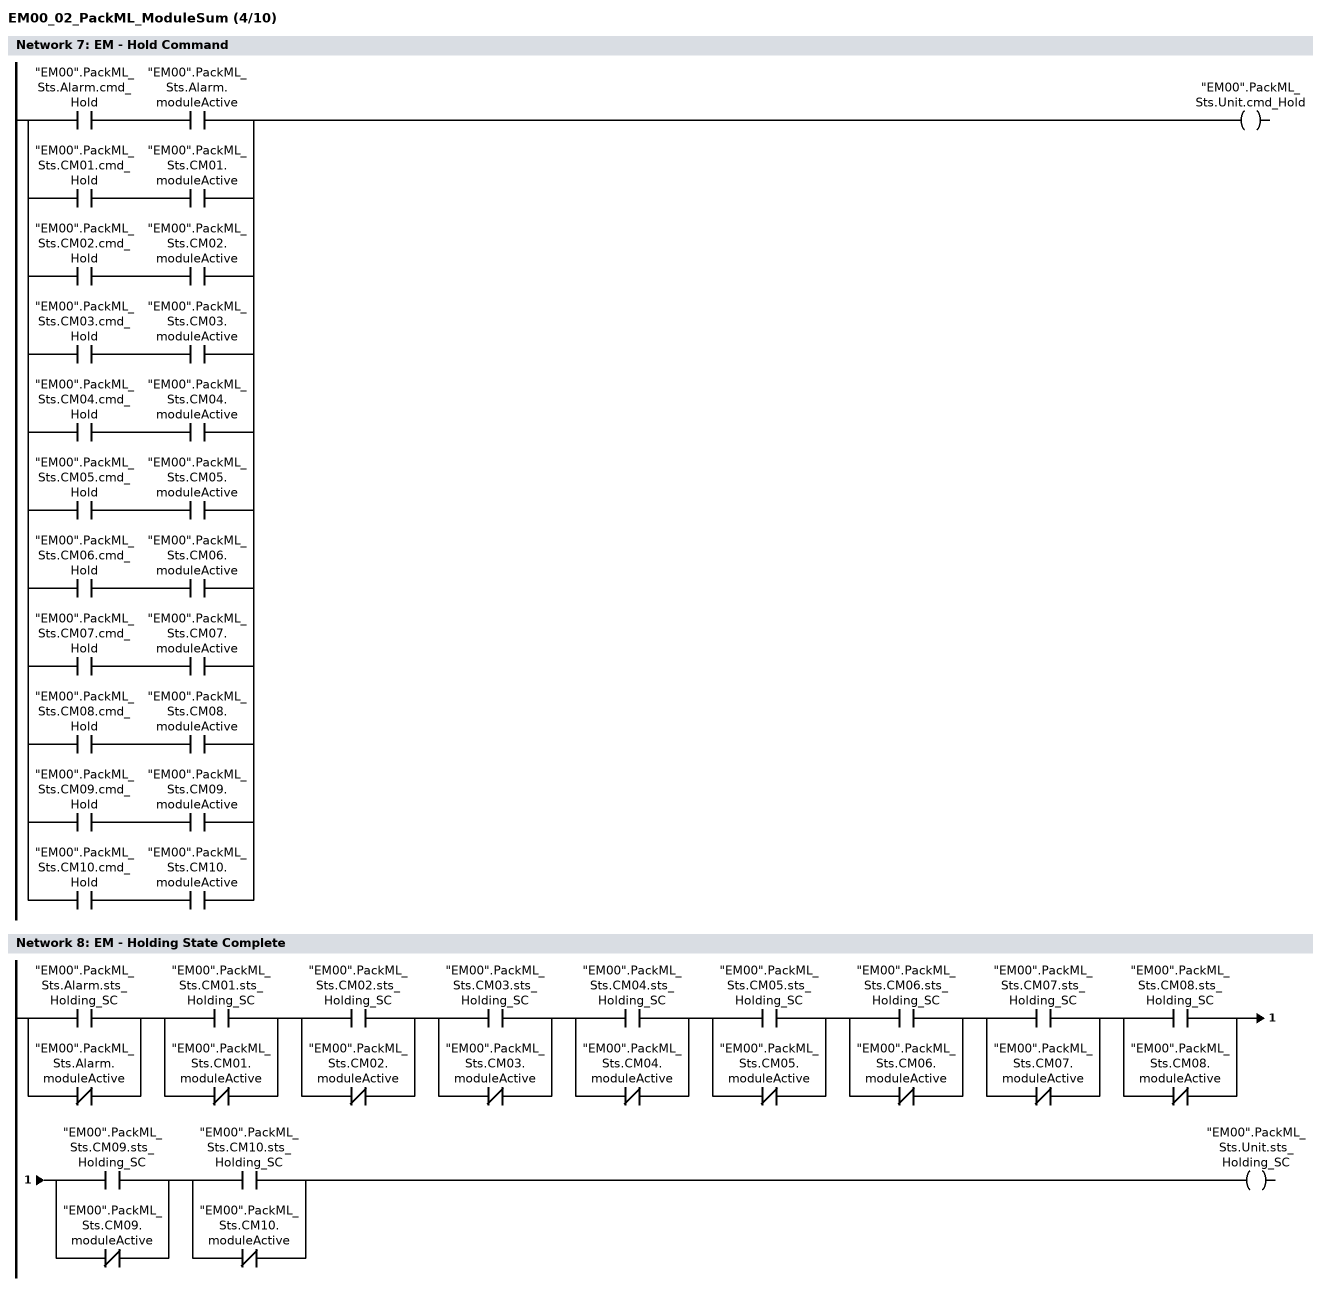
   RUNG wire#powerrail
      Contact( "EM00".PackML_Sts.Alarm.cmd_Hold )
      Contact( "EM00".PackML_Sts.Alarm.moduleActive )
      wire#w1
      Coil( "EM00".PackML_Sts.Unit.cmd_Hold )
   END_RUNG
   RUNG wire#powerrail
      Contact( "EM00".PackML_Sts.CM01.cmd_Hold )
      Contact( "EM00".PackML_Sts.CM01.moduleActive )
   END_RUNG wire#w1
   RUNG wire#powerrail
      Contact( "EM00".PackML_Sts.CM02.cmd_Hold )
      Contact( "EM00".PackML_Sts.CM02.moduleActive )
   END_RUNG wire#w1
   RUNG wire#powerrail
      Contact( "EM00".PackML_Sts.CM03.cmd_Hold )
      Contact( "EM00".PackML_Sts.CM03.moduleActive )
   END_RUNG wire#w1
   RUNG wire#powerrail
      Contact( "EM00".PackML_Sts.CM04.cmd_Hold )
      Contact( "EM00".PackML_Sts.CM04.moduleActive )
   END_RUNG wire#w1
   RUNG wire#powerrail
      Contact( "EM00".PackML_Sts.CM05.cmd_Hold )
      Contact( "EM00".PackML_Sts.CM05.moduleActive )
   END_RUNG wire#w1
   RUNG wire#powerrail
      Contact( "EM00".PackML_Sts.CM06.cmd_Hold )
      Contact( "EM00".PackML_Sts.CM06.moduleActive )
   END_RUNG wire#w1
   RUNG wire#powerrail
      Contact( "EM00".PackML_Sts.CM07.cmd_Hold )
      Contact( "EM00".PackML_Sts.CM07.moduleActive )
   END_RUNG wire#w1
   RUNG wire#powerrail
      Contact( "EM00".PackML_Sts.CM08.cmd_Hold )
      Contact( "EM00".PackML_Sts.CM08.moduleActive )
   END_RUNG wire#w1
   RUNG wire#powerrail
      Contact( "EM00".PackML_Sts.CM09.cmd_Hold )
      Contact( "EM00".PackML_Sts.CM09.moduleActive )
   END_RUNG wire#w1
   RUNG wire#powerrail
      Contact( "EM00".PackML_Sts.CM10.cmd_Hold )
      Contact( "EM00".PackML_Sts.CM10.moduleActive )
   END_RUNG wire#w1
   // the same network as SCL:
   "EM00".PackML_Sts.Unit.cmd_Hold := ("EM00".PackML_Sts.Alarm.cmd_Hold AND "EM00".PackML_Sts.Alarm.moduleActive) OR ("EM00".PackML_Sts.CM01.cmd_Hold AND "EM00".PackML_Sts.CM01.moduleActive) OR ("EM00".PackML_Sts.CM02.cmd_Hold AND "EM00".PackML_Sts.CM02.moduleActive) OR ("EM00".PackML_Sts.CM03.cmd_Hold AND "EM00".PackML_Sts.CM03.moduleActive) OR ("EM00".PackML_Sts.CM04.cmd_Hold AND "EM00".PackML_Sts.CM04.moduleActive) OR ("EM00".PackML_Sts.CM05.cmd_Hold AND "EM00".PackML_Sts.CM05.moduleActive) OR ("EM00".PackML_Sts.CM06.cmd_Hold AND "EM00".PackML_Sts.CM06.moduleActive) OR ("EM00".PackML_Sts.CM07.cmd_Hold AND "EM00".PackML_Sts.CM07.moduleActive) OR ("EM00".PackML_Sts.CM08.cmd_Hold AND "EM00".PackML_Sts.CM08.moduleActive) OR ("EM00".PackML_Sts.CM09.cmd_Hold AND "EM00".PackML_Sts.CM09.moduleActive) OR ("EM00".PackML_Sts.CM10.cmd_Hold AND "EM00".PackML_Sts.CM10.moduleActive);
END_REGION

REGION Network 8: EM - Holding State Complete
   RUNG wire#powerrail
      Contact( "EM00".PackML_Sts.Alarm.sts_Holding_SC )
      wire#w1
      Contact( "EM00".PackML_Sts.CM01.sts_Holding_SC )
      wire#w2
      Contact( "EM00".PackML_Sts.CM02.sts_Holding_SC )
      wire#w3
      Contact( "EM00".PackML_Sts.CM03.sts_Holding_SC )
      wire#w4
      Contact( "EM00".PackML_Sts.CM04.sts_Holding_SC )
      wire#w5
      Contact( "EM00".PackML_Sts.CM05.sts_Holding_SC )
      wire#w6
      Contact( "EM00".PackML_Sts.CM06.sts_Holding_SC )
      wire#w7
      Contact( "EM00".PackML_Sts.CM07.sts_Holding_SC )
      wire#w8
      Contact( "EM00".PackML_Sts.CM08.sts_Holding_SC )
      wire#w9
      Contact( "EM00".PackML_Sts.CM09.sts_Holding_SC )
      wire#w10
      Contact( "EM00".PackML_Sts.CM10.sts_Holding_SC )
      wire#w11
      Coil( "EM00".PackML_Sts.Unit.sts_Holding_SC )
   END_RUNG
   RUNG wire#powerrail
      I_Contact( "EM00".PackML_Sts.Alarm.moduleActive )
   END_RUNG wire#w1
   RUNG wire#w1
      I_Contact( "EM00".PackML_Sts.CM01.moduleActive )
   END_RUNG wire#w2
   RUNG wire#w2
      I_Contact( "EM00".PackML_Sts.CM02.moduleActive )
   END_RUNG wire#w3
   RUNG wire#w3
      I_Contact( "EM00".PackML_Sts.CM03.moduleActive )
   END_RUNG wire#w4
   RUNG wire#w4
      I_Contact( "EM00".PackML_Sts.CM04.moduleActive )
   END_RUNG wire#w5
   RUNG wire#w5
      I_Contact( "EM00".PackML_Sts.CM05.moduleActive )
   END_RUNG wire#w6
   RUNG wire#w6
      I_Contact( "EM00".PackML_Sts.CM06.moduleActive )
   END_RUNG wire#w7
   RUNG wire#w7
      I_Contact( "EM00".PackML_Sts.CM07.moduleActive )
   END_RUNG wire#w8
   RUNG wire#w8
      I_Contact( "EM00".PackML_Sts.CM08.moduleActive )
   END_RUNG wire#w9
   RUNG wire#w9
      I_Contact( "EM00".PackML_Sts.CM09.moduleActive )
   END_RUNG wire#w10
   RUNG wire#w10
      I_Contact( "EM00".PackML_Sts.CM10.moduleActive )
   END_RUNG wire#w11
   // the same network as SCL:
   "EM00".PackML_Sts.Unit.sts_Holding_SC := ("EM00".PackML_Sts.Alarm.sts_Holding_SC OR NOT "EM00".PackML_Sts.Alarm.moduleActive) AND ("EM00".PackML_Sts.CM01.sts_Holding_SC OR NOT "EM00".PackML_Sts.CM01.moduleActive) AND ("EM00".PackML_Sts.CM02.sts_Holding_SC OR NOT "EM00".PackML_Sts.CM02.moduleActive) AND ("EM00".PackML_Sts.CM03.sts_Holding_SC OR NOT "EM00".PackML_Sts.CM03.moduleActive) AND ("EM00".PackML_Sts.CM04.sts_Holding_SC OR NOT "EM00".PackML_Sts.CM04.moduleActive) AND ("EM00".PackML_Sts.CM05.sts_Holding_SC OR NOT "EM00".PackML_Sts.CM05.moduleActive) AND ("EM00".PackML_Sts.CM06.sts_Holding_SC OR NOT "EM00".PackML_Sts.CM06.moduleActive) AND ("EM00".PackML_Sts.CM07.sts_Holding_SC OR NOT "EM00".PackML_Sts.CM07.moduleActive) AND ("EM00".PackML_Sts.CM08.sts_Holding_SC OR NOT "EM00".PackML_Sts.CM08.moduleActive) AND ("EM00".PackML_Sts.CM09.sts_Holding_SC OR NOT "EM00".PackML_Sts.CM09.moduleActive) AND ("EM00".PackML_Sts.CM10.sts_Holding_SC OR NOT "EM00".PackML_Sts.CM10.moduleActive);
END_REGION

REGION Network 9: EM - UnHold Command
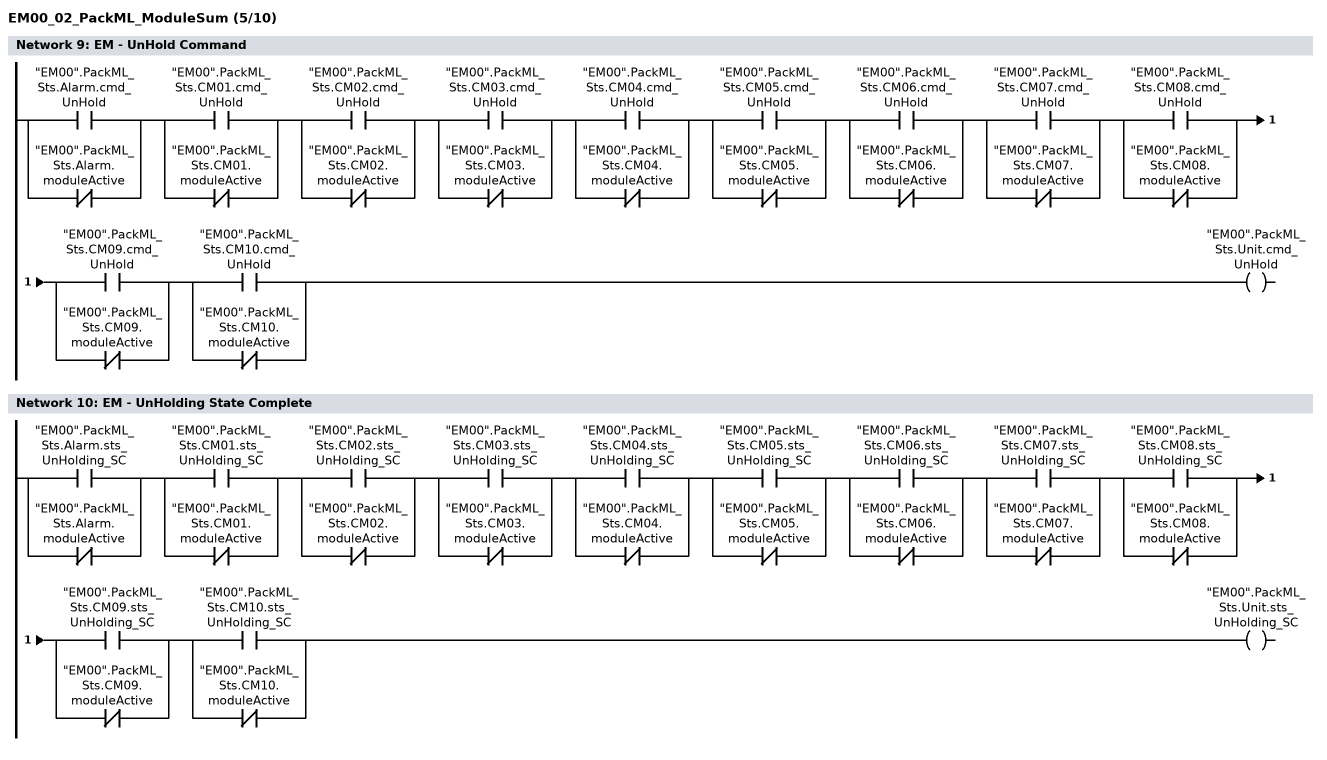
   RUNG wire#powerrail
      Contact( "EM00".PackML_Sts.Alarm.cmd_UnHold )
      wire#w1
      Contact( "EM00".PackML_Sts.CM01.cmd_UnHold )
      wire#w2
      Contact( "EM00".PackML_Sts.CM02.cmd_UnHold )
      wire#w3
      Contact( "EM00".PackML_Sts.CM03.cmd_UnHold )
      wire#w4
      Contact( "EM00".PackML_Sts.CM04.cmd_UnHold )
      wire#w5
      Contact( "EM00".PackML_Sts.CM05.cmd_UnHold )
      wire#w6
      Contact( "EM00".PackML_Sts.CM06.cmd_UnHold )
      wire#w7
      Contact( "EM00".PackML_Sts.CM07.cmd_UnHold )
      wire#w8
      Contact( "EM00".PackML_Sts.CM08.cmd_UnHold )
      wire#w9
      Contact( "EM00".PackML_Sts.CM09.cmd_UnHold )
      wire#w10
      Contact( "EM00".PackML_Sts.CM10.cmd_UnHold )
      wire#w11
      Coil( "EM00".PackML_Sts.Unit.cmd_UnHold )
   END_RUNG
   RUNG wire#powerrail
      I_Contact( "EM00".PackML_Sts.Alarm.moduleActive )
   END_RUNG wire#w1
   RUNG wire#w1
      I_Contact( "EM00".PackML_Sts.CM01.moduleActive )
   END_RUNG wire#w2
   RUNG wire#w2
      I_Contact( "EM00".PackML_Sts.CM02.moduleActive )
   END_RUNG wire#w3
   RUNG wire#w3
      I_Contact( "EM00".PackML_Sts.CM03.moduleActive )
   END_RUNG wire#w4
   RUNG wire#w4
      I_Contact( "EM00".PackML_Sts.CM04.moduleActive )
   END_RUNG wire#w5
   RUNG wire#w5
      I_Contact( "EM00".PackML_Sts.CM05.moduleActive )
   END_RUNG wire#w6
   RUNG wire#w6
      I_Contact( "EM00".PackML_Sts.CM06.moduleActive )
   END_RUNG wire#w7
   RUNG wire#w7
      I_Contact( "EM00".PackML_Sts.CM07.moduleActive )
   END_RUNG wire#w8
   RUNG wire#w8
      I_Contact( "EM00".PackML_Sts.CM08.moduleActive )
   END_RUNG wire#w9
   RUNG wire#w9
      I_Contact( "EM00".PackML_Sts.CM09.moduleActive )
   END_RUNG wire#w10
   RUNG wire#w10
      I_Contact( "EM00".PackML_Sts.CM10.moduleActive )
   END_RUNG wire#w11
   // the same network as SCL:
   "EM00".PackML_Sts.Unit.cmd_UnHold := ("EM00".PackML_Sts.Alarm.cmd_UnHold OR NOT "EM00".PackML_Sts.Alarm.moduleActive) AND ("EM00".PackML_Sts.CM01.cmd_UnHold OR NOT "EM00".PackML_Sts.CM01.moduleActive) AND ("EM00".PackML_Sts.CM02.cmd_UnHold OR NOT "EM00".PackML_Sts.CM02.moduleActive) AND ("EM00".PackML_Sts.CM03.cmd_UnHold OR NOT "EM00".PackML_Sts.CM03.moduleActive) AND ("EM00".PackML_Sts.CM04.cmd_UnHold OR NOT "EM00".PackML_Sts.CM04.moduleActive) AND ("EM00".PackML_Sts.CM05.cmd_UnHold OR NOT "EM00".PackML_Sts.CM05.moduleActive) AND ("EM00".PackML_Sts.CM06.cmd_UnHold OR NOT "EM00".PackML_Sts.CM06.moduleActive) AND ("EM00".PackML_Sts.CM07.cmd_UnHold OR NOT "EM00".PackML_Sts.CM07.moduleActive) AND ("EM00".PackML_Sts.CM08.cmd_UnHold OR NOT "EM00".PackML_Sts.CM08.moduleActive) AND ("EM00".PackML_Sts.CM09.cmd_UnHold OR NOT "EM00".PackML_Sts.CM09.moduleActive) AND ("EM00".PackML_Sts.CM10.cmd_UnHold OR NOT "EM00".PackML_Sts.CM10.moduleActive);
END_REGION

REGION Network 10: EM - UnHolding State Complete
   RUNG wire#powerrail
      Contact( "EM00".PackML_Sts.Alarm.sts_UnHolding_SC )
      wire#w1
      Contact( "EM00".PackML_Sts.CM01.sts_UnHolding_SC )
      wire#w2
      Contact( "EM00".PackML_Sts.CM02.sts_UnHolding_SC )
      wire#w3
      Contact( "EM00".PackML_Sts.CM03.sts_UnHolding_SC )
      wire#w4
      Contact( "EM00".PackML_Sts.CM04.sts_UnHolding_SC )
      wire#w5
      Contact( "EM00".PackML_Sts.CM05.sts_UnHolding_SC )
      wire#w6
      Contact( "EM00".PackML_Sts.CM06.sts_UnHolding_SC )
      wire#w7
      Contact( "EM00".PackML_Sts.CM07.sts_UnHolding_SC )
      wire#w8
      Contact( "EM00".PackML_Sts.CM08.sts_UnHolding_SC )
      wire#w9
      Contact( "EM00".PackML_Sts.CM09.sts_UnHolding_SC )
      wire#w10
      Contact( "EM00".PackML_Sts.CM10.sts_UnHolding_SC )
      wire#w11
      Coil( "EM00".PackML_Sts.Unit.sts_UnHolding_SC )
   END_RUNG
   RUNG wire#powerrail
      I_Contact( "EM00".PackML_Sts.Alarm.moduleActive )
   END_RUNG wire#w1
   RUNG wire#w1
      I_Contact( "EM00".PackML_Sts.CM01.moduleActive )
   END_RUNG wire#w2
   RUNG wire#w2
      I_Contact( "EM00".PackML_Sts.CM02.moduleActive )
   END_RUNG wire#w3
   RUNG wire#w3
      I_Contact( "EM00".PackML_Sts.CM03.moduleActive )
   END_RUNG wire#w4
   RUNG wire#w4
      I_Contact( "EM00".PackML_Sts.CM04.moduleActive )
   END_RUNG wire#w5
   RUNG wire#w5
      I_Contact( "EM00".PackML_Sts.CM05.moduleActive )
   END_RUNG wire#w6
   RUNG wire#w6
      I_Contact( "EM00".PackML_Sts.CM06.moduleActive )
   END_RUNG wire#w7
   RUNG wire#w7
      I_Contact( "EM00".PackML_Sts.CM07.moduleActive )
   END_RUNG wire#w8
   RUNG wire#w8
      I_Contact( "EM00".PackML_Sts.CM08.moduleActive )
   END_RUNG wire#w9
   RUNG wire#w9
      I_Contact( "EM00".PackML_Sts.CM09.moduleActive )
   END_RUNG wire#w10
   RUNG wire#w10
      I_Contact( "EM00".PackML_Sts.CM10.moduleActive )
   END_RUNG wire#w11
   // the same network as SCL:
   "EM00".PackML_Sts.Unit.sts_UnHolding_SC := ("EM00".PackML_Sts.Alarm.sts_UnHolding_SC OR NOT "EM00".PackML_Sts.Alarm.moduleActive) AND ("EM00".PackML_Sts.CM01.sts_UnHolding_SC OR NOT "EM00".PackML_Sts.CM01.moduleActive) AND ("EM00".PackML_Sts.CM02.sts_UnHolding_SC OR NOT "EM00".PackML_Sts.CM02.moduleActive) AND ("EM00".PackML_Sts.CM03.sts_UnHolding_SC OR NOT "EM00".PackML_Sts.CM03.moduleActive) AND ("EM00".PackML_Sts.CM04.sts_UnHolding_SC OR NOT "EM00".PackML_Sts.CM04.moduleActive) AND ("EM00".PackML_Sts.CM05.sts_UnHolding_SC OR NOT "EM00".PackML_Sts.CM05.moduleActive) AND ("EM00".PackML_Sts.CM06.sts_UnHolding_SC OR NOT "EM00".PackML_Sts.CM06.moduleActive) AND ("EM00".PackML_Sts.CM07.sts_UnHolding_SC OR NOT "EM00".PackML_Sts.CM07.moduleActive) AND ("EM00".PackML_Sts.CM08.sts_UnHolding_SC OR NOT "EM00".PackML_Sts.CM08.moduleActive) AND ("EM00".PackML_Sts.CM09.sts_UnHolding_SC OR NOT "EM00".PackML_Sts.CM09.moduleActive) AND ("EM00".PackML_Sts.CM10.sts_UnHolding_SC OR NOT "EM00".PackML_Sts.CM10.moduleActive);
END_REGION

REGION Network 11: EM - Suspend Command
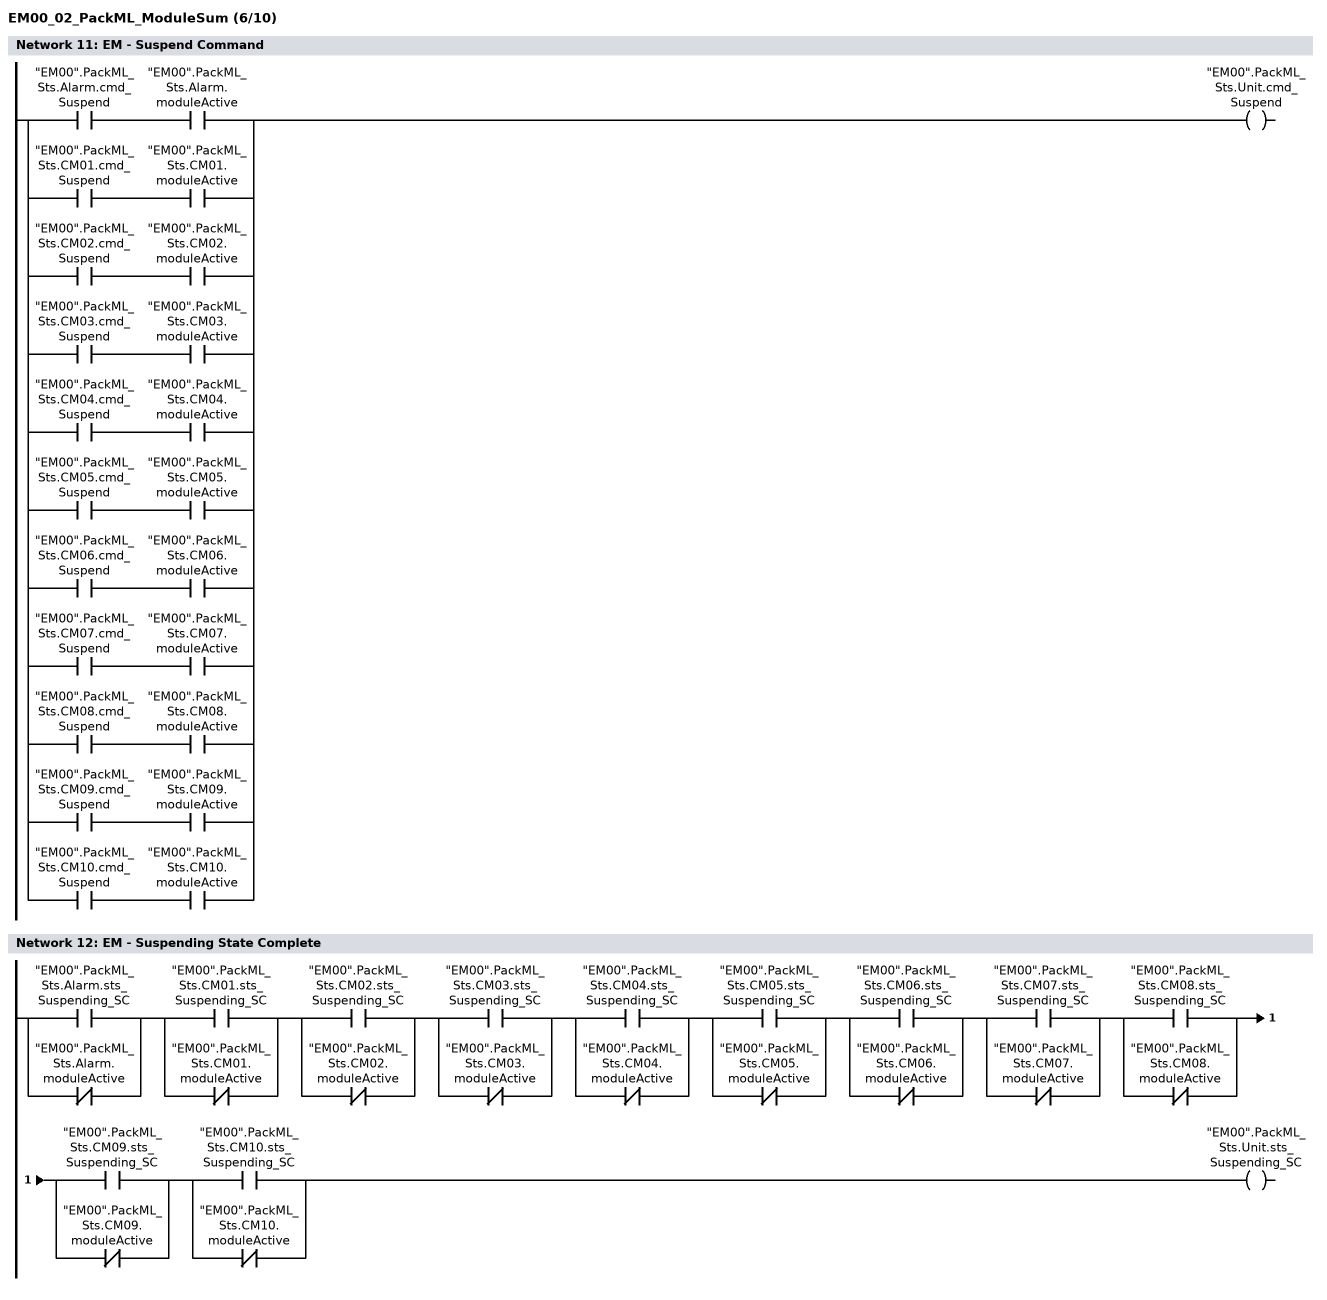
   RUNG wire#powerrail
      Contact( "EM00".PackML_Sts.Alarm.cmd_Suspend )
      Contact( "EM00".PackML_Sts.Alarm.moduleActive )
      wire#w1
      Coil( "EM00".PackML_Sts.Unit.cmd_Suspend )
   END_RUNG
   RUNG wire#powerrail
      Contact( "EM00".PackML_Sts.CM01.cmd_Suspend )
      Contact( "EM00".PackML_Sts.CM01.moduleActive )
   END_RUNG wire#w1
   RUNG wire#powerrail
      Contact( "EM00".PackML_Sts.CM02.cmd_Suspend )
      Contact( "EM00".PackML_Sts.CM02.moduleActive )
   END_RUNG wire#w1
   RUNG wire#powerrail
      Contact( "EM00".PackML_Sts.CM03.cmd_Suspend )
      Contact( "EM00".PackML_Sts.CM03.moduleActive )
   END_RUNG wire#w1
   RUNG wire#powerrail
      Contact( "EM00".PackML_Sts.CM04.cmd_Suspend )
      Contact( "EM00".PackML_Sts.CM04.moduleActive )
   END_RUNG wire#w1
   RUNG wire#powerrail
      Contact( "EM00".PackML_Sts.CM05.cmd_Suspend )
      Contact( "EM00".PackML_Sts.CM05.moduleActive )
   END_RUNG wire#w1
   RUNG wire#powerrail
      Contact( "EM00".PackML_Sts.CM06.cmd_Suspend )
      Contact( "EM00".PackML_Sts.CM06.moduleActive )
   END_RUNG wire#w1
   RUNG wire#powerrail
      Contact( "EM00".PackML_Sts.CM07.cmd_Suspend )
      Contact( "EM00".PackML_Sts.CM07.moduleActive )
   END_RUNG wire#w1
   RUNG wire#powerrail
      Contact( "EM00".PackML_Sts.CM08.cmd_Suspend )
      Contact( "EM00".PackML_Sts.CM08.moduleActive )
   END_RUNG wire#w1
   RUNG wire#powerrail
      Contact( "EM00".PackML_Sts.CM09.cmd_Suspend )
      Contact( "EM00".PackML_Sts.CM09.moduleActive )
   END_RUNG wire#w1
   RUNG wire#powerrail
      Contact( "EM00".PackML_Sts.CM10.cmd_Suspend )
      Contact( "EM00".PackML_Sts.CM10.moduleActive )
   END_RUNG wire#w1
   // the same network as SCL:
   "EM00".PackML_Sts.Unit.cmd_Suspend := ("EM00".PackML_Sts.Alarm.cmd_Suspend AND "EM00".PackML_Sts.Alarm.moduleActive) OR ("EM00".PackML_Sts.CM01.cmd_Suspend AND "EM00".PackML_Sts.CM01.moduleActive) OR ("EM00".PackML_Sts.CM02.cmd_Suspend AND "EM00".PackML_Sts.CM02.moduleActive) OR ("EM00".PackML_Sts.CM03.cmd_Suspend AND "EM00".PackML_Sts.CM03.moduleActive) OR ("EM00".PackML_Sts.CM04.cmd_Suspend AND "EM00".PackML_Sts.CM04.moduleActive) OR ("EM00".PackML_Sts.CM05.cmd_Suspend AND "EM00".PackML_Sts.CM05.moduleActive) OR ("EM00".PackML_Sts.CM06.cmd_Suspend AND "EM00".PackML_Sts.CM06.moduleActive) OR ("EM00".PackML_Sts.CM07.cmd_Suspend AND "EM00".PackML_Sts.CM07.moduleActive) OR ("EM00".PackML_Sts.CM08.cmd_Suspend AND "EM00".PackML_Sts.CM08.moduleActive) OR ("EM00".PackML_Sts.CM09.cmd_Suspend AND "EM00".PackML_Sts.CM09.moduleActive) OR ("EM00".PackML_Sts.CM10.cmd_Suspend AND "EM00".PackML_Sts.CM10.moduleActive);
END_REGION

REGION Network 12: EM - Suspending State Complete
   RUNG wire#powerrail
      Contact( "EM00".PackML_Sts.Alarm.sts_Suspending_SC )
      wire#w1
      Contact( "EM00".PackML_Sts.CM01.sts_Suspending_SC )
      wire#w2
      Contact( "EM00".PackML_Sts.CM02.sts_Suspending_SC )
      wire#w3
      Contact( "EM00".PackML_Sts.CM03.sts_Suspending_SC )
      wire#w4
      Contact( "EM00".PackML_Sts.CM04.sts_Suspending_SC )
      wire#w5
      Contact( "EM00".PackML_Sts.CM05.sts_Suspending_SC )
      wire#w6
      Contact( "EM00".PackML_Sts.CM06.sts_Suspending_SC )
      wire#w7
      Contact( "EM00".PackML_Sts.CM07.sts_Suspending_SC )
      wire#w8
      Contact( "EM00".PackML_Sts.CM08.sts_Suspending_SC )
      wire#w9
      Contact( "EM00".PackML_Sts.CM09.sts_Suspending_SC )
      wire#w10
      Contact( "EM00".PackML_Sts.CM10.sts_Suspending_SC )
      wire#w11
      Coil( "EM00".PackML_Sts.Unit.sts_Suspending_SC )
   END_RUNG
   RUNG wire#powerrail
      I_Contact( "EM00".PackML_Sts.Alarm.moduleActive )
   END_RUNG wire#w1
   RUNG wire#w1
      I_Contact( "EM00".PackML_Sts.CM01.moduleActive )
   END_RUNG wire#w2
   RUNG wire#w2
      I_Contact( "EM00".PackML_Sts.CM02.moduleActive )
   END_RUNG wire#w3
   RUNG wire#w3
      I_Contact( "EM00".PackML_Sts.CM03.moduleActive )
   END_RUNG wire#w4
   RUNG wire#w4
      I_Contact( "EM00".PackML_Sts.CM04.moduleActive )
   END_RUNG wire#w5
   RUNG wire#w5
      I_Contact( "EM00".PackML_Sts.CM05.moduleActive )
   END_RUNG wire#w6
   RUNG wire#w6
      I_Contact( "EM00".PackML_Sts.CM06.moduleActive )
   END_RUNG wire#w7
   RUNG wire#w7
      I_Contact( "EM00".PackML_Sts.CM07.moduleActive )
   END_RUNG wire#w8
   RUNG wire#w8
      I_Contact( "EM00".PackML_Sts.CM08.moduleActive )
   END_RUNG wire#w9
   RUNG wire#w9
      I_Contact( "EM00".PackML_Sts.CM09.moduleActive )
   END_RUNG wire#w10
   RUNG wire#w10
      I_Contact( "EM00".PackML_Sts.CM10.moduleActive )
   END_RUNG wire#w11
   // the same network as SCL:
   "EM00".PackML_Sts.Unit.sts_Suspending_SC := ("EM00".PackML_Sts.Alarm.sts_Suspending_SC OR NOT "EM00".PackML_Sts.Alarm.moduleActive) AND ("EM00".PackML_Sts.CM01.sts_Suspending_SC OR NOT "EM00".PackML_Sts.CM01.moduleActive) AND ("EM00".PackML_Sts.CM02.sts_Suspending_SC OR NOT "EM00".PackML_Sts.CM02.moduleActive) AND ("EM00".PackML_Sts.CM03.sts_Suspending_SC OR NOT "EM00".PackML_Sts.CM03.moduleActive) AND ("EM00".PackML_Sts.CM04.sts_Suspending_SC OR NOT "EM00".PackML_Sts.CM04.moduleActive) AND ("EM00".PackML_Sts.CM05.sts_Suspending_SC OR NOT "EM00".PackML_Sts.CM05.moduleActive) AND ("EM00".PackML_Sts.CM06.sts_Suspending_SC OR NOT "EM00".PackML_Sts.CM06.moduleActive) AND ("EM00".PackML_Sts.CM07.sts_Suspending_SC OR NOT "EM00".PackML_Sts.CM07.moduleActive) AND ("EM00".PackML_Sts.CM08.sts_Suspending_SC OR NOT "EM00".PackML_Sts.CM08.moduleActive) AND ("EM00".PackML_Sts.CM09.sts_Suspending_SC OR NOT "EM00".PackML_Sts.CM09.moduleActive) AND ("EM00".PackML_Sts.CM10.sts_Suspending_SC OR NOT "EM00".PackML_Sts.CM10.moduleActive);
END_REGION

REGION Network 13: EM - UnSuspend Command
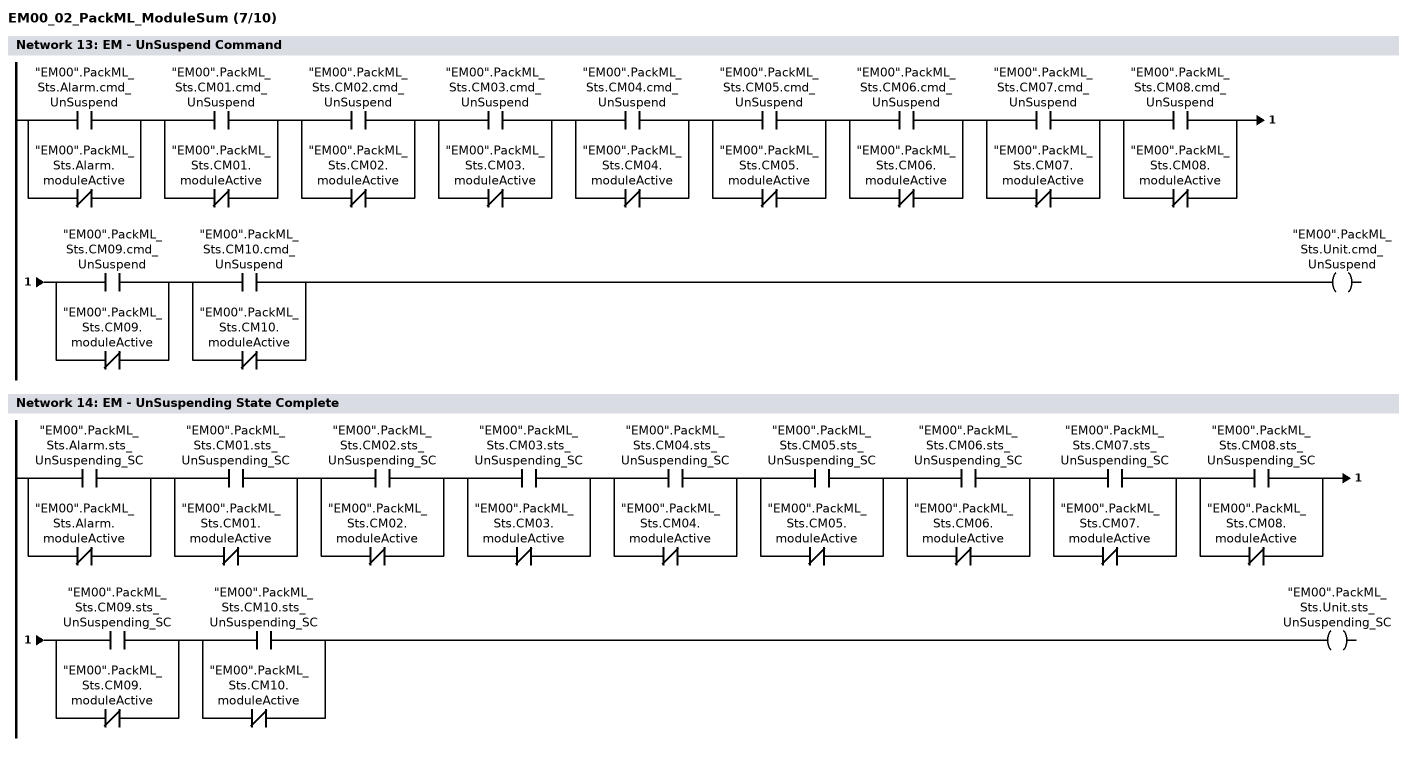
   RUNG wire#powerrail
      Contact( "EM00".PackML_Sts.Alarm.cmd_UnSuspend )
      wire#w1
      Contact( "EM00".PackML_Sts.CM01.cmd_UnSuspend )
      wire#w2
      Contact( "EM00".PackML_Sts.CM02.cmd_UnSuspend )
      wire#w3
      Contact( "EM00".PackML_Sts.CM03.cmd_UnSuspend )
      wire#w4
      Contact( "EM00".PackML_Sts.CM04.cmd_UnSuspend )
      wire#w5
      Contact( "EM00".PackML_Sts.CM05.cmd_UnSuspend )
      wire#w6
      Contact( "EM00".PackML_Sts.CM06.cmd_UnSuspend )
      wire#w7
      Contact( "EM00".PackML_Sts.CM07.cmd_UnSuspend )
      wire#w8
      Contact( "EM00".PackML_Sts.CM08.cmd_UnSuspend )
      wire#w9
      Contact( "EM00".PackML_Sts.CM09.cmd_UnSuspend )
      wire#w10
      Contact( "EM00".PackML_Sts.CM10.cmd_UnSuspend )
      wire#w11
      Coil( "EM00".PackML_Sts.Unit.cmd_UnSuspend )
   END_RUNG
   RUNG wire#powerrail
      I_Contact( "EM00".PackML_Sts.Alarm.moduleActive )
   END_RUNG wire#w1
   RUNG wire#w1
      I_Contact( "EM00".PackML_Sts.CM01.moduleActive )
   END_RUNG wire#w2
   RUNG wire#w2
      I_Contact( "EM00".PackML_Sts.CM02.moduleActive )
   END_RUNG wire#w3
   RUNG wire#w3
      I_Contact( "EM00".PackML_Sts.CM03.moduleActive )
   END_RUNG wire#w4
   RUNG wire#w4
      I_Contact( "EM00".PackML_Sts.CM04.moduleActive )
   END_RUNG wire#w5
   RUNG wire#w5
      I_Contact( "EM00".PackML_Sts.CM05.moduleActive )
   END_RUNG wire#w6
   RUNG wire#w6
      I_Contact( "EM00".PackML_Sts.CM06.moduleActive )
   END_RUNG wire#w7
   RUNG wire#w7
      I_Contact( "EM00".PackML_Sts.CM07.moduleActive )
   END_RUNG wire#w8
   RUNG wire#w8
      I_Contact( "EM00".PackML_Sts.CM08.moduleActive )
   END_RUNG wire#w9
   RUNG wire#w9
      I_Contact( "EM00".PackML_Sts.CM09.moduleActive )
   END_RUNG wire#w10
   RUNG wire#w10
      I_Contact( "EM00".PackML_Sts.CM10.moduleActive )
   END_RUNG wire#w11
   // the same network as SCL:
   "EM00".PackML_Sts.Unit.cmd_UnSuspend := ("EM00".PackML_Sts.Alarm.cmd_UnSuspend OR NOT "EM00".PackML_Sts.Alarm.moduleActive) AND ("EM00".PackML_Sts.CM01.cmd_UnSuspend OR NOT "EM00".PackML_Sts.CM01.moduleActive) AND ("EM00".PackML_Sts.CM02.cmd_UnSuspend OR NOT "EM00".PackML_Sts.CM02.moduleActive) AND ("EM00".PackML_Sts.CM03.cmd_UnSuspend OR NOT "EM00".PackML_Sts.CM03.moduleActive) AND ("EM00".PackML_Sts.CM04.cmd_UnSuspend OR NOT "EM00".PackML_Sts.CM04.moduleActive) AND ("EM00".PackML_Sts.CM05.cmd_UnSuspend OR NOT "EM00".PackML_Sts.CM05.moduleActive) AND ("EM00".PackML_Sts.CM06.cmd_UnSuspend OR NOT "EM00".PackML_Sts.CM06.moduleActive) AND ("EM00".PackML_Sts.CM07.cmd_UnSuspend OR NOT "EM00".PackML_Sts.CM07.moduleActive) AND ("EM00".PackML_Sts.CM08.cmd_UnSuspend OR NOT "EM00".PackML_Sts.CM08.moduleActive) AND ("EM00".PackML_Sts.CM09.cmd_UnSuspend OR NOT "EM00".PackML_Sts.CM09.moduleActive) AND ("EM00".PackML_Sts.CM10.cmd_UnSuspend OR NOT "EM00".PackML_Sts.CM10.moduleActive);
END_REGION

REGION Network 14: EM - UnSuspending State Complete
   RUNG wire#powerrail
      Contact( "EM00".PackML_Sts.Alarm.sts_UnSuspending_SC )
      wire#w1
      Contact( "EM00".PackML_Sts.CM01.sts_UnSuspending_SC )
      wire#w2
      Contact( "EM00".PackML_Sts.CM02.sts_UnSuspending_SC )
      wire#w3
      Contact( "EM00".PackML_Sts.CM03.sts_UnSuspending_SC )
      wire#w4
      Contact( "EM00".PackML_Sts.CM04.sts_UnSuspending_SC )
      wire#w5
      Contact( "EM00".PackML_Sts.CM05.sts_UnSuspending_SC )
      wire#w6
      Contact( "EM00".PackML_Sts.CM06.sts_UnSuspending_SC )
      wire#w7
      Contact( "EM00".PackML_Sts.CM07.sts_UnSuspending_SC )
      wire#w8
      Contact( "EM00".PackML_Sts.CM08.sts_UnSuspending_SC )
      wire#w9
      Contact( "EM00".PackML_Sts.CM09.sts_UnSuspending_SC )
      wire#w10
      Contact( "EM00".PackML_Sts.CM10.sts_UnSuspending_SC )
      wire#w11
      Coil( "EM00".PackML_Sts.Unit.sts_UnSuspending_SC )
   END_RUNG
   RUNG wire#powerrail
      I_Contact( "EM00".PackML_Sts.Alarm.moduleActive )
   END_RUNG wire#w1
   RUNG wire#w1
      I_Contact( "EM00".PackML_Sts.CM01.moduleActive )
   END_RUNG wire#w2
   RUNG wire#w2
      I_Contact( "EM00".PackML_Sts.CM02.moduleActive )
   END_RUNG wire#w3
   RUNG wire#w3
      I_Contact( "EM00".PackML_Sts.CM03.moduleActive )
   END_RUNG wire#w4
   RUNG wire#w4
      I_Contact( "EM00".PackML_Sts.CM04.moduleActive )
   END_RUNG wire#w5
   RUNG wire#w5
      I_Contact( "EM00".PackML_Sts.CM05.moduleActive )
   END_RUNG wire#w6
   RUNG wire#w6
      I_Contact( "EM00".PackML_Sts.CM06.moduleActive )
   END_RUNG wire#w7
   RUNG wire#w7
      I_Contact( "EM00".PackML_Sts.CM07.moduleActive )
   END_RUNG wire#w8
   RUNG wire#w8
      I_Contact( "EM00".PackML_Sts.CM08.moduleActive )
   END_RUNG wire#w9
   RUNG wire#w9
      I_Contact( "EM00".PackML_Sts.CM09.moduleActive )
   END_RUNG wire#w10
   RUNG wire#w10
      I_Contact( "EM00".PackML_Sts.CM10.moduleActive )
   END_RUNG wire#w11
   // the same network as SCL:
   "EM00".PackML_Sts.Unit.sts_UnSuspending_SC := ("EM00".PackML_Sts.Alarm.sts_UnSuspending_SC OR NOT "EM00".PackML_Sts.Alarm.moduleActive) AND ("EM00".PackML_Sts.CM01.sts_UnSuspending_SC OR NOT "EM00".PackML_Sts.CM01.moduleActive) AND ("EM00".PackML_Sts.CM02.sts_UnSuspending_SC OR NOT "EM00".PackML_Sts.CM02.moduleActive) AND ("EM00".PackML_Sts.CM03.sts_UnSuspending_SC OR NOT "EM00".PackML_Sts.CM03.moduleActive) AND ("EM00".PackML_Sts.CM04.sts_UnSuspending_SC OR NOT "EM00".PackML_Sts.CM04.moduleActive) AND ("EM00".PackML_Sts.CM05.sts_UnSuspending_SC OR NOT "EM00".PackML_Sts.CM05.moduleActive) AND ("EM00".PackML_Sts.CM06.sts_UnSuspending_SC OR NOT "EM00".PackML_Sts.CM06.moduleActive) AND ("EM00".PackML_Sts.CM07.sts_UnSuspending_SC OR NOT "EM00".PackML_Sts.CM07.moduleActive) AND ("EM00".PackML_Sts.CM08.sts_UnSuspending_SC OR NOT "EM00".PackML_Sts.CM08.moduleActive) AND ("EM00".PackML_Sts.CM09.sts_UnSuspending_SC OR NOT "EM00".PackML_Sts.CM09.moduleActive) AND ("EM00".PackML_Sts.CM10.sts_UnSuspending_SC OR NOT "EM00".PackML_Sts.CM10.moduleActive);
END_REGION

REGION Network 15: EM - Abort Command
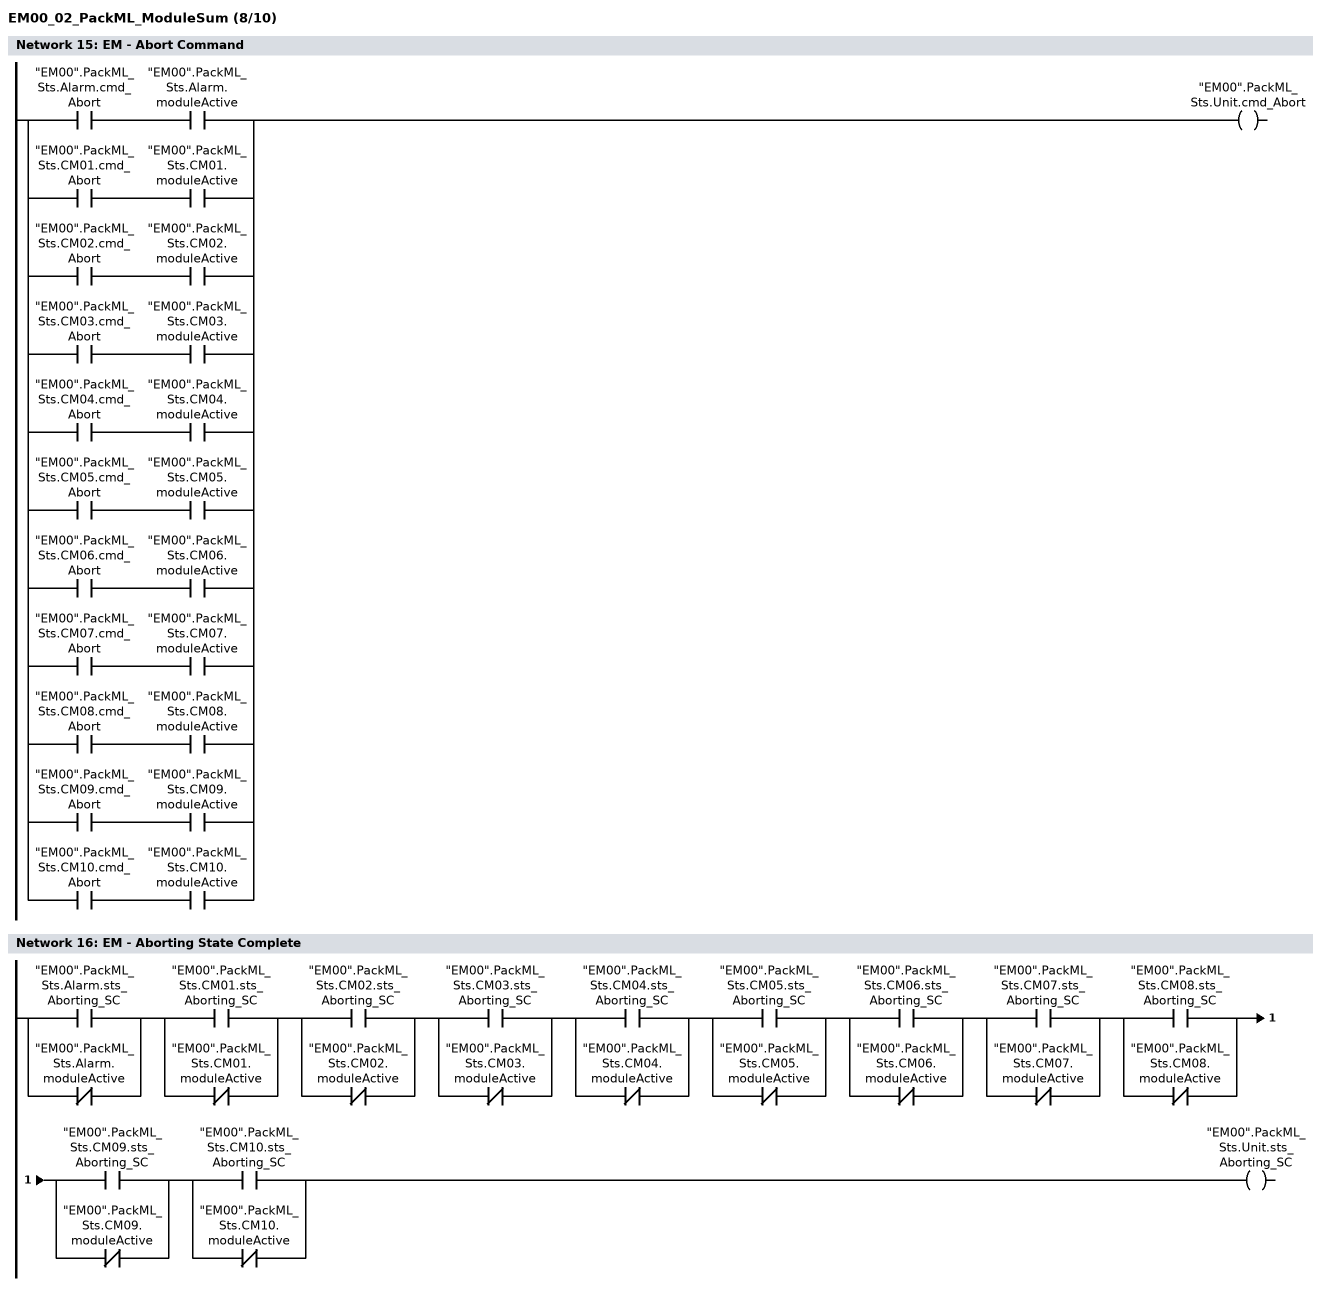
   RUNG wire#powerrail
      Contact( "EM00".PackML_Sts.Alarm.cmd_Abort )
      Contact( "EM00".PackML_Sts.Alarm.moduleActive )
      wire#w1
      Coil( "EM00".PackML_Sts.Unit.cmd_Abort )
   END_RUNG
   RUNG wire#powerrail
      Contact( "EM00".PackML_Sts.CM01.cmd_Abort )
      Contact( "EM00".PackML_Sts.CM01.moduleActive )
   END_RUNG wire#w1
   RUNG wire#powerrail
      Contact( "EM00".PackML_Sts.CM02.cmd_Abort )
      Contact( "EM00".PackML_Sts.CM02.moduleActive )
   END_RUNG wire#w1
   RUNG wire#powerrail
      Contact( "EM00".PackML_Sts.CM03.cmd_Abort )
      Contact( "EM00".PackML_Sts.CM03.moduleActive )
   END_RUNG wire#w1
   RUNG wire#powerrail
      Contact( "EM00".PackML_Sts.CM04.cmd_Abort )
      Contact( "EM00".PackML_Sts.CM04.moduleActive )
   END_RUNG wire#w1
   RUNG wire#powerrail
      Contact( "EM00".PackML_Sts.CM05.cmd_Abort )
      Contact( "EM00".PackML_Sts.CM05.moduleActive )
   END_RUNG wire#w1
   RUNG wire#powerrail
      Contact( "EM00".PackML_Sts.CM06.cmd_Abort )
      Contact( "EM00".PackML_Sts.CM06.moduleActive )
   END_RUNG wire#w1
   RUNG wire#powerrail
      Contact( "EM00".PackML_Sts.CM07.cmd_Abort )
      Contact( "EM00".PackML_Sts.CM07.moduleActive )
   END_RUNG wire#w1
   RUNG wire#powerrail
      Contact( "EM00".PackML_Sts.CM08.cmd_Abort )
      Contact( "EM00".PackML_Sts.CM08.moduleActive )
   END_RUNG wire#w1
   RUNG wire#powerrail
      Contact( "EM00".PackML_Sts.CM09.cmd_Abort )
      Contact( "EM00".PackML_Sts.CM09.moduleActive )
   END_RUNG wire#w1
   RUNG wire#powerrail
      Contact( "EM00".PackML_Sts.CM10.cmd_Abort )
      Contact( "EM00".PackML_Sts.CM10.moduleActive )
   END_RUNG wire#w1
   // the same network as SCL:
   "EM00".PackML_Sts.Unit.cmd_Abort := ("EM00".PackML_Sts.Alarm.cmd_Abort AND "EM00".PackML_Sts.Alarm.moduleActive) OR ("EM00".PackML_Sts.CM01.cmd_Abort AND "EM00".PackML_Sts.CM01.moduleActive) OR ("EM00".PackML_Sts.CM02.cmd_Abort AND "EM00".PackML_Sts.CM02.moduleActive) OR ("EM00".PackML_Sts.CM03.cmd_Abort AND "EM00".PackML_Sts.CM03.moduleActive) OR ("EM00".PackML_Sts.CM04.cmd_Abort AND "EM00".PackML_Sts.CM04.moduleActive) OR ("EM00".PackML_Sts.CM05.cmd_Abort AND "EM00".PackML_Sts.CM05.moduleActive) OR ("EM00".PackML_Sts.CM06.cmd_Abort AND "EM00".PackML_Sts.CM06.moduleActive) OR ("EM00".PackML_Sts.CM07.cmd_Abort AND "EM00".PackML_Sts.CM07.moduleActive) OR ("EM00".PackML_Sts.CM08.cmd_Abort AND "EM00".PackML_Sts.CM08.moduleActive) OR ("EM00".PackML_Sts.CM09.cmd_Abort AND "EM00".PackML_Sts.CM09.moduleActive) OR ("EM00".PackML_Sts.CM10.cmd_Abort AND "EM00".PackML_Sts.CM10.moduleActive);
END_REGION

REGION Network 16: EM - Aborting State Complete
   RUNG wire#powerrail
      Contact( "EM00".PackML_Sts.Alarm.sts_Aborting_SC )
      wire#w1
      Contact( "EM00".PackML_Sts.CM01.sts_Aborting_SC )
      wire#w2
      Contact( "EM00".PackML_Sts.CM02.sts_Aborting_SC )
      wire#w3
      Contact( "EM00".PackML_Sts.CM03.sts_Aborting_SC )
      wire#w4
      Contact( "EM00".PackML_Sts.CM04.sts_Aborting_SC )
      wire#w5
      Contact( "EM00".PackML_Sts.CM05.sts_Aborting_SC )
      wire#w6
      Contact( "EM00".PackML_Sts.CM06.sts_Aborting_SC )
      wire#w7
      Contact( "EM00".PackML_Sts.CM07.sts_Aborting_SC )
      wire#w8
      Contact( "EM00".PackML_Sts.CM08.sts_Aborting_SC )
      wire#w9
      Contact( "EM00".PackML_Sts.CM09.sts_Aborting_SC )
      wire#w10
      Contact( "EM00".PackML_Sts.CM10.sts_Aborting_SC )
      wire#w11
      Coil( "EM00".PackML_Sts.Unit.sts_Aborting_SC )
   END_RUNG
   RUNG wire#powerrail
      I_Contact( "EM00".PackML_Sts.Alarm.moduleActive )
   END_RUNG wire#w1
   RUNG wire#w1
      I_Contact( "EM00".PackML_Sts.CM01.moduleActive )
   END_RUNG wire#w2
   RUNG wire#w2
      I_Contact( "EM00".PackML_Sts.CM02.moduleActive )
   END_RUNG wire#w3
   RUNG wire#w3
      I_Contact( "EM00".PackML_Sts.CM03.moduleActive )
   END_RUNG wire#w4
   RUNG wire#w4
      I_Contact( "EM00".PackML_Sts.CM04.moduleActive )
   END_RUNG wire#w5
   RUNG wire#w5
      I_Contact( "EM00".PackML_Sts.CM05.moduleActive )
   END_RUNG wire#w6
   RUNG wire#w6
      I_Contact( "EM00".PackML_Sts.CM06.moduleActive )
   END_RUNG wire#w7
   RUNG wire#w7
      I_Contact( "EM00".PackML_Sts.CM07.moduleActive )
   END_RUNG wire#w8
   RUNG wire#w8
      I_Contact( "EM00".PackML_Sts.CM08.moduleActive )
   END_RUNG wire#w9
   RUNG wire#w9
      I_Contact( "EM00".PackML_Sts.CM09.moduleActive )
   END_RUNG wire#w10
   RUNG wire#w10
      I_Contact( "EM00".PackML_Sts.CM10.moduleActive )
   END_RUNG wire#w11
   // the same network as SCL:
   "EM00".PackML_Sts.Unit.sts_Aborting_SC := ("EM00".PackML_Sts.Alarm.sts_Aborting_SC OR NOT "EM00".PackML_Sts.Alarm.moduleActive) AND ("EM00".PackML_Sts.CM01.sts_Aborting_SC OR NOT "EM00".PackML_Sts.CM01.moduleActive) AND ("EM00".PackML_Sts.CM02.sts_Aborting_SC OR NOT "EM00".PackML_Sts.CM02.moduleActive) AND ("EM00".PackML_Sts.CM03.sts_Aborting_SC OR NOT "EM00".PackML_Sts.CM03.moduleActive) AND ("EM00".PackML_Sts.CM04.sts_Aborting_SC OR NOT "EM00".PackML_Sts.CM04.moduleActive) AND ("EM00".PackML_Sts.CM05.sts_Aborting_SC OR NOT "EM00".PackML_Sts.CM05.moduleActive) AND ("EM00".PackML_Sts.CM06.sts_Aborting_SC OR NOT "EM00".PackML_Sts.CM06.moduleActive) AND ("EM00".PackML_Sts.CM07.sts_Aborting_SC OR NOT "EM00".PackML_Sts.CM07.moduleActive) AND ("EM00".PackML_Sts.CM08.sts_Aborting_SC OR NOT "EM00".PackML_Sts.CM08.moduleActive) AND ("EM00".PackML_Sts.CM09.sts_Aborting_SC OR NOT "EM00".PackML_Sts.CM09.moduleActive) AND ("EM00".PackML_Sts.CM10.sts_Aborting_SC OR NOT "EM00".PackML_Sts.CM10.moduleActive);
END_REGION

REGION Network 17: EM - Clear Command
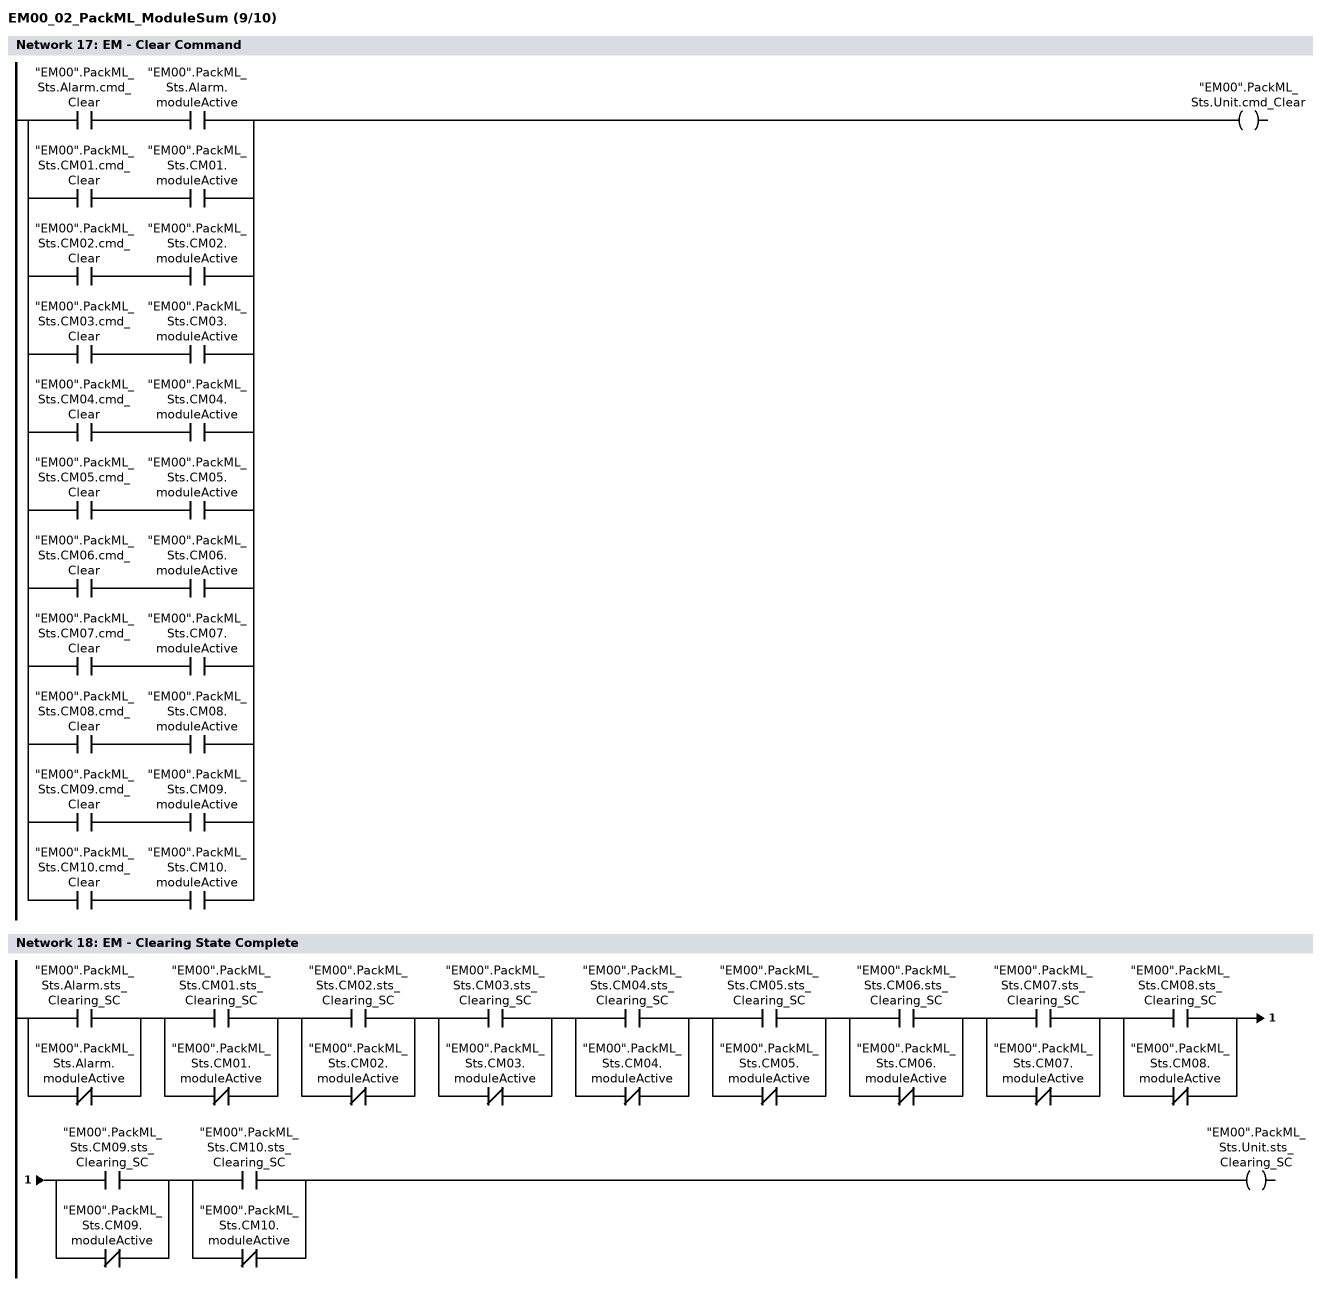
   RUNG wire#powerrail
      Contact( "EM00".PackML_Sts.Alarm.cmd_Clear )
      Contact( "EM00".PackML_Sts.Alarm.moduleActive )
      wire#w1
      Coil( "EM00".PackML_Sts.Unit.cmd_Clear )
   END_RUNG
   RUNG wire#powerrail
      Contact( "EM00".PackML_Sts.CM01.cmd_Clear )
      Contact( "EM00".PackML_Sts.CM01.moduleActive )
   END_RUNG wire#w1
   RUNG wire#powerrail
      Contact( "EM00".PackML_Sts.CM02.cmd_Clear )
      Contact( "EM00".PackML_Sts.CM02.moduleActive )
   END_RUNG wire#w1
   RUNG wire#powerrail
      Contact( "EM00".PackML_Sts.CM03.cmd_Clear )
      Contact( "EM00".PackML_Sts.CM03.moduleActive )
   END_RUNG wire#w1
   RUNG wire#powerrail
      Contact( "EM00".PackML_Sts.CM04.cmd_Clear )
      Contact( "EM00".PackML_Sts.CM04.moduleActive )
   END_RUNG wire#w1
   RUNG wire#powerrail
      Contact( "EM00".PackML_Sts.CM05.cmd_Clear )
      Contact( "EM00".PackML_Sts.CM05.moduleActive )
   END_RUNG wire#w1
   RUNG wire#powerrail
      Contact( "EM00".PackML_Sts.CM06.cmd_Clear )
      Contact( "EM00".PackML_Sts.CM06.moduleActive )
   END_RUNG wire#w1
   RUNG wire#powerrail
      Contact( "EM00".PackML_Sts.CM07.cmd_Clear )
      Contact( "EM00".PackML_Sts.CM07.moduleActive )
   END_RUNG wire#w1
   RUNG wire#powerrail
      Contact( "EM00".PackML_Sts.CM08.cmd_Clear )
      Contact( "EM00".PackML_Sts.CM08.moduleActive )
   END_RUNG wire#w1
   RUNG wire#powerrail
      Contact( "EM00".PackML_Sts.CM09.cmd_Clear )
      Contact( "EM00".PackML_Sts.CM09.moduleActive )
   END_RUNG wire#w1
   RUNG wire#powerrail
      Contact( "EM00".PackML_Sts.CM10.cmd_Clear )
      Contact( "EM00".PackML_Sts.CM10.moduleActive )
   END_RUNG wire#w1
   // the same network as SCL:
   "EM00".PackML_Sts.Unit.cmd_Clear := ("EM00".PackML_Sts.Alarm.cmd_Clear AND "EM00".PackML_Sts.Alarm.moduleActive) OR ("EM00".PackML_Sts.CM01.cmd_Clear AND "EM00".PackML_Sts.CM01.moduleActive) OR ("EM00".PackML_Sts.CM02.cmd_Clear AND "EM00".PackML_Sts.CM02.moduleActive) OR ("EM00".PackML_Sts.CM03.cmd_Clear AND "EM00".PackML_Sts.CM03.moduleActive) OR ("EM00".PackML_Sts.CM04.cmd_Clear AND "EM00".PackML_Sts.CM04.moduleActive) OR ("EM00".PackML_Sts.CM05.cmd_Clear AND "EM00".PackML_Sts.CM05.moduleActive) OR ("EM00".PackML_Sts.CM06.cmd_Clear AND "EM00".PackML_Sts.CM06.moduleActive) OR ("EM00".PackML_Sts.CM07.cmd_Clear AND "EM00".PackML_Sts.CM07.moduleActive) OR ("EM00".PackML_Sts.CM08.cmd_Clear AND "EM00".PackML_Sts.CM08.moduleActive) OR ("EM00".PackML_Sts.CM09.cmd_Clear AND "EM00".PackML_Sts.CM09.moduleActive) OR ("EM00".PackML_Sts.CM10.cmd_Clear AND "EM00".PackML_Sts.CM10.moduleActive);
END_REGION

REGION Network 18: EM - Clearing State Complete
   RUNG wire#powerrail
      Contact( "EM00".PackML_Sts.Alarm.sts_Clearing_SC )
      wire#w1
      Contact( "EM00".PackML_Sts.CM01.sts_Clearing_SC )
      wire#w2
      Contact( "EM00".PackML_Sts.CM02.sts_Clearing_SC )
      wire#w3
      Contact( "EM00".PackML_Sts.CM03.sts_Clearing_SC )
      wire#w4
      Contact( "EM00".PackML_Sts.CM04.sts_Clearing_SC )
      wire#w5
      Contact( "EM00".PackML_Sts.CM05.sts_Clearing_SC )
      wire#w6
      Contact( "EM00".PackML_Sts.CM06.sts_Clearing_SC )
      wire#w7
      Contact( "EM00".PackML_Sts.CM07.sts_Clearing_SC )
      wire#w8
      Contact( "EM00".PackML_Sts.CM08.sts_Clearing_SC )
      wire#w9
      Contact( "EM00".PackML_Sts.CM09.sts_Clearing_SC )
      wire#w10
      Contact( "EM00".PackML_Sts.CM10.sts_Clearing_SC )
      wire#w11
      Coil( "EM00".PackML_Sts.Unit.sts_Clearing_SC )
   END_RUNG
   RUNG wire#powerrail
      I_Contact( "EM00".PackML_Sts.Alarm.moduleActive )
   END_RUNG wire#w1
   RUNG wire#w1
      I_Contact( "EM00".PackML_Sts.CM01.moduleActive )
   END_RUNG wire#w2
   RUNG wire#w2
      I_Contact( "EM00".PackML_Sts.CM02.moduleActive )
   END_RUNG wire#w3
   RUNG wire#w3
      I_Contact( "EM00".PackML_Sts.CM03.moduleActive )
   END_RUNG wire#w4
   RUNG wire#w4
      I_Contact( "EM00".PackML_Sts.CM04.moduleActive )
   END_RUNG wire#w5
   RUNG wire#w5
      I_Contact( "EM00".PackML_Sts.CM05.moduleActive )
   END_RUNG wire#w6
   RUNG wire#w6
      I_Contact( "EM00".PackML_Sts.CM06.moduleActive )
   END_RUNG wire#w7
   RUNG wire#w7
      I_Contact( "EM00".PackML_Sts.CM07.moduleActive )
   END_RUNG wire#w8
   RUNG wire#w8
      I_Contact( "EM00".PackML_Sts.CM08.moduleActive )
   END_RUNG wire#w9
   RUNG wire#w9
      I_Contact( "EM00".PackML_Sts.CM09.moduleActive )
   END_RUNG wire#w10
   RUNG wire#w10
      I_Contact( "EM00".PackML_Sts.CM10.moduleActive )
   END_RUNG wire#w11
   // the same network as SCL:
   "EM00".PackML_Sts.Unit.sts_Clearing_SC := ("EM00".PackML_Sts.Alarm.sts_Clearing_SC OR NOT "EM00".PackML_Sts.Alarm.moduleActive) AND ("EM00".PackML_Sts.CM01.sts_Clearing_SC OR NOT "EM00".PackML_Sts.CM01.moduleActive) AND ("EM00".PackML_Sts.CM02.sts_Clearing_SC OR NOT "EM00".PackML_Sts.CM02.moduleActive) AND ("EM00".PackML_Sts.CM03.sts_Clearing_SC OR NOT "EM00".PackML_Sts.CM03.moduleActive) AND ("EM00".PackML_Sts.CM04.sts_Clearing_SC OR NOT "EM00".PackML_Sts.CM04.moduleActive) AND ("EM00".PackML_Sts.CM05.sts_Clearing_SC OR NOT "EM00".PackML_Sts.CM05.moduleActive) AND ("EM00".PackML_Sts.CM06.sts_Clearing_SC OR NOT "EM00".PackML_Sts.CM06.moduleActive) AND ("EM00".PackML_Sts.CM07.sts_Clearing_SC OR NOT "EM00".PackML_Sts.CM07.moduleActive) AND ("EM00".PackML_Sts.CM08.sts_Clearing_SC OR NOT "EM00".PackML_Sts.CM08.moduleActive) AND ("EM00".PackML_Sts.CM09.sts_Clearing_SC OR NOT "EM00".PackML_Sts.CM09.moduleActive) AND ("EM00".PackML_Sts.CM10.sts_Clearing_SC OR NOT "EM00".PackML_Sts.CM10.moduleActive);
END_REGION

REGION Network 19: EM - Execute State Complete
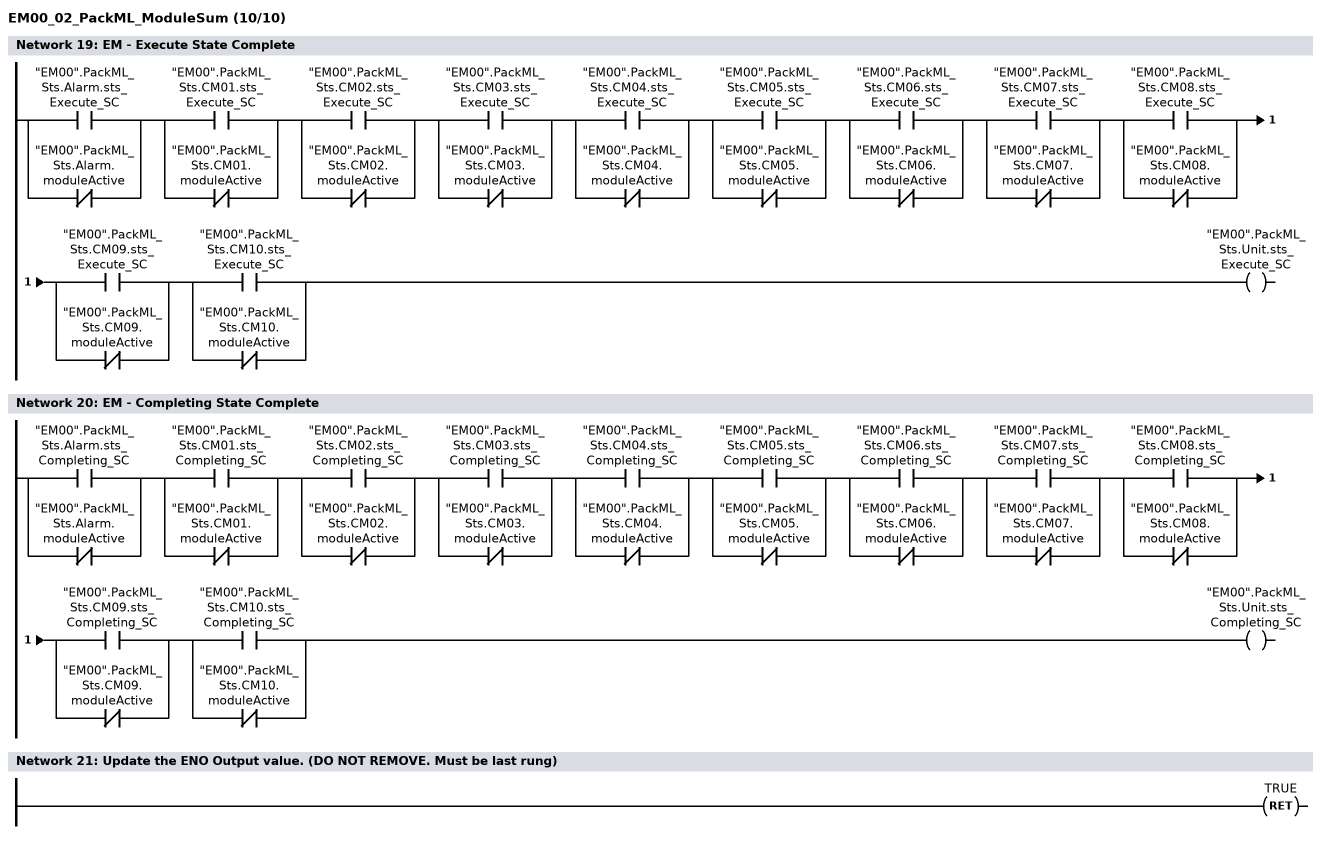
   RUNG wire#powerrail
      Contact( "EM00".PackML_Sts.Alarm.sts_Execute_SC )
      wire#w1
      Contact( "EM00".PackML_Sts.CM01.sts_Execute_SC )
      wire#w2
      Contact( "EM00".PackML_Sts.CM02.sts_Execute_SC )
      wire#w3
      Contact( "EM00".PackML_Sts.CM03.sts_Execute_SC )
      wire#w4
      Contact( "EM00".PackML_Sts.CM04.sts_Execute_SC )
      wire#w5
      Contact( "EM00".PackML_Sts.CM05.sts_Execute_SC )
      wire#w6
      Contact( "EM00".PackML_Sts.CM06.sts_Execute_SC )
      wire#w7
      Contact( "EM00".PackML_Sts.CM07.sts_Execute_SC )
      wire#w8
      Contact( "EM00".PackML_Sts.CM08.sts_Execute_SC )
      wire#w9
      Contact( "EM00".PackML_Sts.CM09.sts_Execute_SC )
      wire#w10
      Contact( "EM00".PackML_Sts.CM10.sts_Execute_SC )
      wire#w11
      Coil( "EM00".PackML_Sts.Unit.sts_Execute_SC )
   END_RUNG
   RUNG wire#powerrail
      I_Contact( "EM00".PackML_Sts.Alarm.moduleActive )
   END_RUNG wire#w1
   RUNG wire#w1
      I_Contact( "EM00".PackML_Sts.CM01.moduleActive )
   END_RUNG wire#w2
   RUNG wire#w2
      I_Contact( "EM00".PackML_Sts.CM02.moduleActive )
   END_RUNG wire#w3
   RUNG wire#w3
      I_Contact( "EM00".PackML_Sts.CM03.moduleActive )
   END_RUNG wire#w4
   RUNG wire#w4
      I_Contact( "EM00".PackML_Sts.CM04.moduleActive )
   END_RUNG wire#w5
   RUNG wire#w5
      I_Contact( "EM00".PackML_Sts.CM05.moduleActive )
   END_RUNG wire#w6
   RUNG wire#w6
      I_Contact( "EM00".PackML_Sts.CM06.moduleActive )
   END_RUNG wire#w7
   RUNG wire#w7
      I_Contact( "EM00".PackML_Sts.CM07.moduleActive )
   END_RUNG wire#w8
   RUNG wire#w8
      I_Contact( "EM00".PackML_Sts.CM08.moduleActive )
   END_RUNG wire#w9
   RUNG wire#w9
      I_Contact( "EM00".PackML_Sts.CM09.moduleActive )
   END_RUNG wire#w10
   RUNG wire#w10
      I_Contact( "EM00".PackML_Sts.CM10.moduleActive )
   END_RUNG wire#w11
   // the same network as SCL:
   "EM00".PackML_Sts.Unit.sts_Execute_SC := ("EM00".PackML_Sts.Alarm.sts_Execute_SC OR NOT "EM00".PackML_Sts.Alarm.moduleActive) AND ("EM00".PackML_Sts.CM01.sts_Execute_SC OR NOT "EM00".PackML_Sts.CM01.moduleActive) AND ("EM00".PackML_Sts.CM02.sts_Execute_SC OR NOT "EM00".PackML_Sts.CM02.moduleActive) AND ("EM00".PackML_Sts.CM03.sts_Execute_SC OR NOT "EM00".PackML_Sts.CM03.moduleActive) AND ("EM00".PackML_Sts.CM04.sts_Execute_SC OR NOT "EM00".PackML_Sts.CM04.moduleActive) AND ("EM00".PackML_Sts.CM05.sts_Execute_SC OR NOT "EM00".PackML_Sts.CM05.moduleActive) AND ("EM00".PackML_Sts.CM06.sts_Execute_SC OR NOT "EM00".PackML_Sts.CM06.moduleActive) AND ("EM00".PackML_Sts.CM07.sts_Execute_SC OR NOT "EM00".PackML_Sts.CM07.moduleActive) AND ("EM00".PackML_Sts.CM08.sts_Execute_SC OR NOT "EM00".PackML_Sts.CM08.moduleActive) AND ("EM00".PackML_Sts.CM09.sts_Execute_SC OR NOT "EM00".PackML_Sts.CM09.moduleActive) AND ("EM00".PackML_Sts.CM10.sts_Execute_SC OR NOT "EM00".PackML_Sts.CM10.moduleActive);
END_REGION

REGION Network 20: EM - Completing State Complete
   RUNG wire#powerrail
      Contact( "EM00".PackML_Sts.Alarm.sts_Completing_SC )
      wire#w1
      Contact( "EM00".PackML_Sts.CM01.sts_Completing_SC )
      wire#w2
      Contact( "EM00".PackML_Sts.CM02.sts_Completing_SC )
      wire#w3
      Contact( "EM00".PackML_Sts.CM03.sts_Completing_SC )
      wire#w4
      Contact( "EM00".PackML_Sts.CM04.sts_Completing_SC )
      wire#w5
      Contact( "EM00".PackML_Sts.CM05.sts_Completing_SC )
      wire#w6
      Contact( "EM00".PackML_Sts.CM06.sts_Completing_SC )
      wire#w7
      Contact( "EM00".PackML_Sts.CM07.sts_Completing_SC )
      wire#w8
      Contact( "EM00".PackML_Sts.CM08.sts_Completing_SC )
      wire#w9
      Contact( "EM00".PackML_Sts.CM09.sts_Completing_SC )
      wire#w10
      Contact( "EM00".PackML_Sts.CM10.sts_Completing_SC )
      wire#w11
      Coil( "EM00".PackML_Sts.Unit.sts_Completing_SC )
   END_RUNG
   RUNG wire#powerrail
      I_Contact( "EM00".PackML_Sts.Alarm.moduleActive )
   END_RUNG wire#w1
   RUNG wire#w1
      I_Contact( "EM00".PackML_Sts.CM01.moduleActive )
   END_RUNG wire#w2
   RUNG wire#w2
      I_Contact( "EM00".PackML_Sts.CM02.moduleActive )
   END_RUNG wire#w3
   RUNG wire#w3
      I_Contact( "EM00".PackML_Sts.CM03.moduleActive )
   END_RUNG wire#w4
   RUNG wire#w4
      I_Contact( "EM00".PackML_Sts.CM04.moduleActive )
   END_RUNG wire#w5
   RUNG wire#w5
      I_Contact( "EM00".PackML_Sts.CM05.moduleActive )
   END_RUNG wire#w6
   RUNG wire#w6
      I_Contact( "EM00".PackML_Sts.CM06.moduleActive )
   END_RUNG wire#w7
   RUNG wire#w7
      I_Contact( "EM00".PackML_Sts.CM07.moduleActive )
   END_RUNG wire#w8
   RUNG wire#w8
      I_Contact( "EM00".PackML_Sts.CM08.moduleActive )
   END_RUNG wire#w9
   RUNG wire#w9
      I_Contact( "EM00".PackML_Sts.CM09.moduleActive )
   END_RUNG wire#w10
   RUNG wire#w10
      I_Contact( "EM00".PackML_Sts.CM10.moduleActive )
   END_RUNG wire#w11
   // the same network as SCL:
   "EM00".PackML_Sts.Unit.sts_Completing_SC := ("EM00".PackML_Sts.Alarm.sts_Completing_SC OR NOT "EM00".PackML_Sts.Alarm.moduleActive) AND ("EM00".PackML_Sts.CM01.sts_Completing_SC OR NOT "EM00".PackML_Sts.CM01.moduleActive) AND ("EM00".PackML_Sts.CM02.sts_Completing_SC OR NOT "EM00".PackML_Sts.CM02.moduleActive) AND ("EM00".PackML_Sts.CM03.sts_Completing_SC OR NOT "EM00".PackML_Sts.CM03.moduleActive) AND ("EM00".PackML_Sts.CM04.sts_Completing_SC OR NOT "EM00".PackML_Sts.CM04.moduleActive) AND ("EM00".PackML_Sts.CM05.sts_Completing_SC OR NOT "EM00".PackML_Sts.CM05.moduleActive) AND ("EM00".PackML_Sts.CM06.sts_Completing_SC OR NOT "EM00".PackML_Sts.CM06.moduleActive) AND ("EM00".PackML_Sts.CM07.sts_Completing_SC OR NOT "EM00".PackML_Sts.CM07.moduleActive) AND ("EM00".PackML_Sts.CM08.sts_Completing_SC OR NOT "EM00".PackML_Sts.CM08.moduleActive) AND ("EM00".PackML_Sts.CM09.sts_Completing_SC OR NOT "EM00".PackML_Sts.CM09.moduleActive) AND ("EM00".PackML_Sts.CM10.sts_Completing_SC OR NOT "EM00".PackML_Sts.CM10.moduleActive);
END_REGION

REGION Network 21: Update the ENO Output value. (DO NOT REMOVE. Must be last rung)
   RUNG wire#powerrail
      ReturnCoil( TRUE )
   END_RUNG
   // the same network as SCL:
   ENO := TRUE;
   RETURN;
END_REGION
END_FUNCTION_BLOCK

FUNCTION_BLOCK "EM01_00_Main"   // FB31660, LAD
TITLE = EM01_00_Main
{ S7_Optimized_Access := 'TRUE' }
AUTHOR : tech.team.motioncontrol@siemens.com
FAMILY : CPG
VERSION : 1.1
// Support: tech.team.motioncontrol@siemens.com
// stored: AutoNumber true, IsIECCheckEnabled false, IsRetainMemResEnabled false, MemoryReserve 100, SetENOAutomatically false, UDAEnableTagReadback false
   VAR
      instEventControl { ExternalAccessible := 'False'; ExternalVisible := 'False'; ExternalWritable := 'False'; S7_SetPoint := 'True'} : "EM01_01_EventControl";   // Instance DB - EM's Event Control Logic
      instPackML_ModuleSum { ExternalAccessible := 'False'; ExternalVisible := 'False'; ExternalWritable := 'False'; S7_SetPoint := 'True'} : "EM01_02_PackML_ModuleSum";   // Instance DB - EM's PackML Module Summation Logic
      instCM01 { ExternalAccessible := 'False'; ExternalVisible := 'False'; ExternalWritable := 'False'; S7_SetPoint := 'True'} : "EM01_CM01_Conveyor";   // Instance DB - CM01
      instCM02 { ExternalAccessible := 'False'; ExternalVisible := 'False'; ExternalWritable := 'False'; S7_SetPoint := 'True'} : "EM01_CM02_Palletizer";   // Instance DB - CM02
   END_VAR
   VAR_TEMP   // added for the SCL form of the ladder/FBD networks
      _w1 : Bool;
   END_VAR
BEGIN

REGION Network 1: *** BEGIN MAIN LOGIC SECTION ***
END_REGION

REGION Network 2: Call the Control Module Logic - CM01
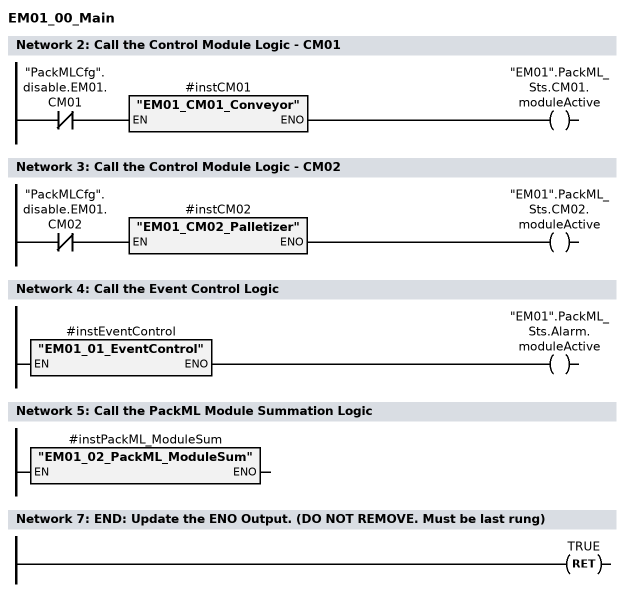
   RUNG wire#powerrail
      I_Contact( "PackMLCfg".disable.EM01.CM01 )
      #instCM01()
      Coil( "EM01".PackML_Sts.CM01.moduleActive )
   END_RUNG
   // the same network as SCL:
   #instCM01(EN := NOT "PackMLCfg".disable.EM01.CM01, ENO => #_w1);   // "EM01_CM01_Conveyor"
   "EM01".PackML_Sts.CM01.moduleActive := #_w1;
END_REGION

REGION Network 3: Call the Control Module Logic - CM02
   RUNG wire#powerrail
      I_Contact( "PackMLCfg".disable.EM01.CM02 )
      #instCM02()
      Coil( "EM01".PackML_Sts.CM02.moduleActive )
   END_RUNG
   // the same network as SCL:
   #instCM02(EN := NOT "PackMLCfg".disable.EM01.CM02, ENO => #_w1);   // "EM01_CM02_Palletizer"
   "EM01".PackML_Sts.CM02.moduleActive := #_w1;
END_REGION

REGION Network 4: Call the Event Control Logic
   RUNG wire#powerrail
      #instEventControl()
      Coil( "EM01".PackML_Sts.Alarm.moduleActive )
   END_RUNG
   // the same network as SCL:
   #instEventControl(ENO => #_w1);   // "EM01_01_EventControl"
   "EM01".PackML_Sts.Alarm.moduleActive := #_w1;
END_REGION

REGION Network 5: Call the PackML Module Summation Logic
   RUNG wire#powerrail
      #instPackML_ModuleSum()
   END_RUNG
   // the same network as SCL:
   #instPackML_ModuleSum();   // "EM01_02_PackML_ModuleSum"
END_REGION

REGION Network 7: END: Update the ENO Output. (DO NOT REMOVE. Must be last rung)
   RUNG wire#powerrail
      ReturnCoil( TRUE )
   END_RUNG
   // the same network as SCL:
   ENO := TRUE;
   RETURN;
END_REGION
END_FUNCTION_BLOCK

FUNCTION_BLOCK "EM01_CM01_Conveyor"   // FB31671, LAD
TITLE = EM01_CM01
{ S7_Optimized_Access := 'TRUE' }
AUTHOR : tech.team.motioncontrol@siemens.com
FAMILY : CPG
VERSION : 1.1
// Support: tech.team.motioncontrol@siemens.com
// stored: AutoNumber true, IsIECCheckEnabled false, IsRetainMemResEnabled false, MemoryReserve 100, SetENOAutomatically false, UDAEnableTagReadback false
   VAR
      statDummyBool { ExternalAccessible := 'False'; ExternalVisible := 'False'; ExternalWritable := 'False'} : Bool;   // dummy bool - placeholder
   END_VAR
BEGIN

REGION Network 1: *** Begin the Setpoint Management Information Section ***
END_REGION

REGION Network 2: *** Begin the Logic Section ***
END_REGION

REGION Network 3: *** Begin the Event Information Section ***
END_REGION

REGION Network 4: *** Begin the State Model Status Feedback Section ***
END_REGION

REGION Network 5: *** Call the PackML Module Initialize Logic ***
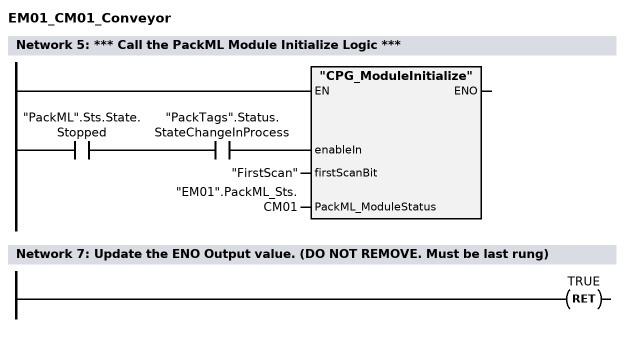
   RUNG wire#powerrail
      "CPG_ModuleInitialize"(enableIn := wire#w1, firstScanBit := "FirstScan", PackML_ModuleStatus := "EM01".PackML_Sts.CM01)
   END_RUNG
   RUNG wire#powerrail
      Contact( "PackML".Sts.State.Stopped )
      Contact( "PackTags".Status.StateChangeInProcess )
   END_RUNG wire#w1
   // the same network as SCL:
   "CPG_ModuleInitialize"(enableIn := "PackML".Sts.State.Stopped AND "PackTags".Status.StateChangeInProcess,
                          firstScanBit := "FirstScan",
                          PackML_ModuleStatus := "EM01".PackML_Sts.CM01);
END_REGION

REGION Network 7: Update the ENO Output value. (DO NOT REMOVE. Must be last rung)
   RUNG wire#powerrail
      ReturnCoil( TRUE )
   END_RUNG
   // the same network as SCL:
   ENO := TRUE;
   RETURN;
END_REGION
END_FUNCTION_BLOCK

FUNCTION_BLOCK "EM01_CM02_Palletizer"   // FB31672, LAD
TITLE = EM01_CM02
{ S7_Optimized_Access := 'TRUE' }
AUTHOR : tech.team.motioncontrol@siemens.com
FAMILY : CPG
VERSION : 1.1
// Support: tech.team.motioncontrol@siemens.com
// stored: AutoNumber true, IsIECCheckEnabled false, IsRetainMemResEnabled false, MemoryReserve 100, SetENOAutomatically false, UDAEnableTagReadback false
   VAR
      statDummyBool { ExternalAccessible := 'False'; ExternalVisible := 'False'; ExternalWritable := 'False'} : Bool;   // dummy bool - placeholder
   END_VAR
BEGIN

REGION Network 1: *** Begin the Setpoint Management Information Section ***
END_REGION

REGION Network 2: *** Begin the Logic Section ***
END_REGION

REGION Network 3: *** Begin the Event Information Section ***
END_REGION

REGION Network 4: *** Begin the State Model Status Feedback Section ***
END_REGION

REGION Network 5: *** Call the PackML Module Initialize Logic ***
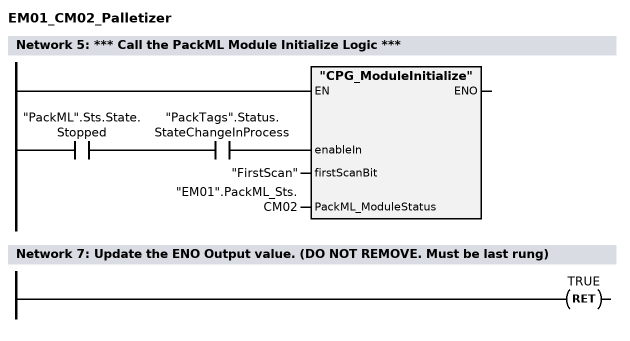
   RUNG wire#powerrail
      "CPG_ModuleInitialize"(enableIn := wire#w1, firstScanBit := "FirstScan", PackML_ModuleStatus := "EM01".PackML_Sts.CM02)
   END_RUNG
   RUNG wire#powerrail
      Contact( "PackML".Sts.State.Stopped )
      Contact( "PackTags".Status.StateChangeInProcess )
   END_RUNG wire#w1
   // the same network as SCL:
   "CPG_ModuleInitialize"(enableIn := "PackML".Sts.State.Stopped AND "PackTags".Status.StateChangeInProcess,
                          firstScanBit := "FirstScan",
                          PackML_ModuleStatus := "EM01".PackML_Sts.CM02);
END_REGION

REGION Network 7: Update the ENO Output value. (DO NOT REMOVE. Must be last rung)
   RUNG wire#powerrail
      ReturnCoil( TRUE )
   END_RUNG
   // the same network as SCL:
   ENO := TRUE;
   RETURN;
END_REGION
END_FUNCTION_BLOCK

FUNCTION_BLOCK "EM01_01_EventControl"   // FB31661, LAD
TITLE = EM01_01_EventControl
{ S7_Optimized_Access := 'TRUE' }
AUTHOR : tech.team.motioncontrol@siemens.com
FAMILY : CPG
VERSION : 1.1
// Support: tech.team.motioncontrol@siemens.com
// stored: AutoNumber true, IsIECCheckEnabled false, IsRetainMemResEnabled false, MemoryReserve 100, SetENOAutomatically false, UDAEnableTagReadback false
   VAR
      instEventMgr_Alarm { ExternalAccessible := 'False'; ExternalVisible := 'False'; ExternalWritable := 'False'; S7_SetPoint := 'True'} : "CPG_EventManager";   // instance FB - Event Manager - Alarm Events
      instEventMgr_Warning { ExternalAccessible := 'False'; ExternalVisible := 'False'; ExternalWritable := 'False'; S7_SetPoint := 'True'} : "CPG_EventManager";   // instance FB - Event Manager - Warning Events
      instEventMgr_Status { ExternalAccessible := 'False'; ExternalVisible := 'False'; ExternalWritable := 'False'; S7_SetPoint := 'True'} : "CPG_EventManager";   // instance FB - Event Manager - Status Events
      instStatus_AlarmNotReset { ExternalAccessible := 'False'; ExternalVisible := 'False'; ExternalWritable := 'False'; S7_SetPoint := 'True'} : "CPG_Event";   // instance FB - PackML Event - Alarms not reset
      statEventMgr_Cmd_Reset { ExternalAccessible := 'False'; ExternalVisible := 'False'; ExternalWritable := 'False'} : Bool;   // Reset Cmd for all event managers
      statEventMgr_Cmd_Clear1stFlt { ExternalAccessible := 'False'; ExternalVisible := 'False'; ExternalWritable := 'False'} : Bool;   // Clear 1st Fault Cmd for all event managers
      statEventMgr_Clear1stFlt_OS { ExternalAccessible := 'False'; ExternalVisible := 'False'; ExternalWritable := 'False'} : Bool;   // Clear 1st Fault Cmd - One shot
   END_VAR
   VAR_TEMP   // added for the SCL form of the ladder/FBD networks
      _w1 : Bool;
      _w2 : Bool;
   END_VAR
BEGIN

REGION Network 1: ** STATE MODEL REPORTING STATUS ****
END_REGION

REGION Network 2: *** Call the PackML Module Initialize Logic ***
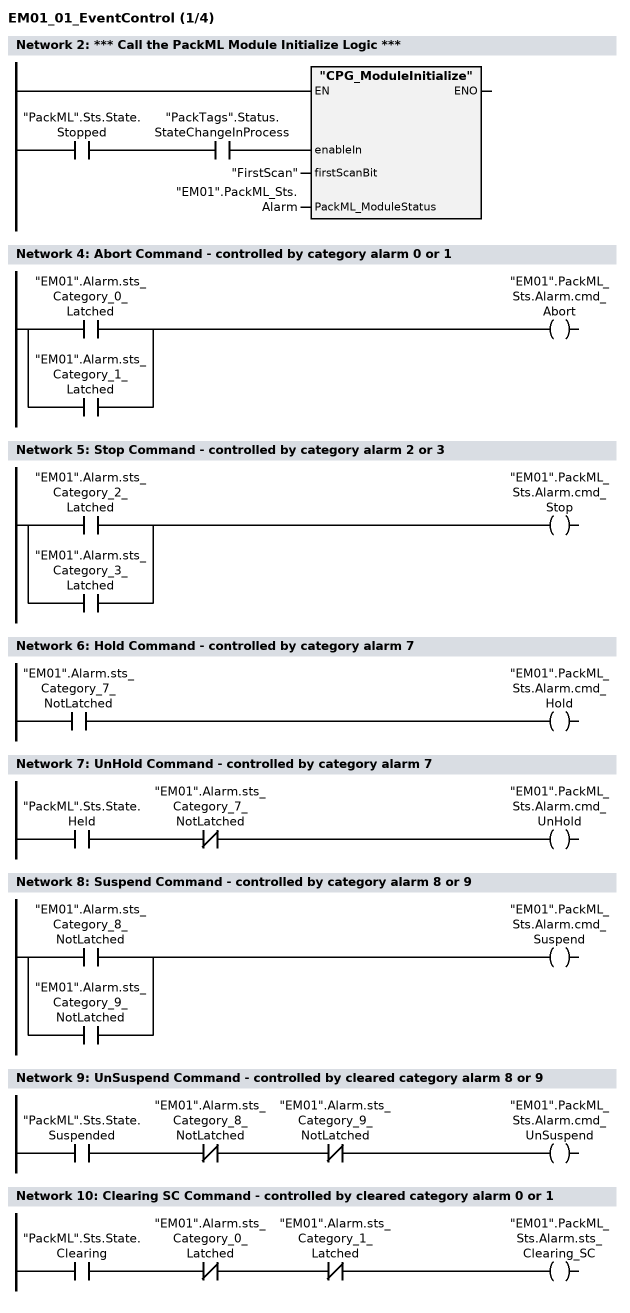
   RUNG wire#powerrail
      "CPG_ModuleInitialize"(enableIn := wire#w1, firstScanBit := "FirstScan", PackML_ModuleStatus := "EM01".PackML_Sts.Alarm)
   END_RUNG
   RUNG wire#powerrail
      Contact( "PackML".Sts.State.Stopped )
      Contact( "PackTags".Status.StateChangeInProcess )
   END_RUNG wire#w1
   // the same network as SCL:
   "CPG_ModuleInitialize"(enableIn := "PackML".Sts.State.Stopped AND "PackTags".Status.StateChangeInProcess,
                          firstScanBit := "FirstScan",
                          PackML_ModuleStatus := "EM01".PackML_Sts.Alarm);
END_REGION

REGION Network 3: Begin the LOGIC section.
END_REGION

REGION Network 4: Abort Command - controlled by category alarm 0 or 1
   RUNG wire#powerrail
      Contact( "EM01".Alarm.sts_Category_0_Latched )
      wire#w1
      Coil( "EM01".PackML_Sts.Alarm.cmd_Abort )
   END_RUNG
   RUNG wire#powerrail
      Contact( "EM01".Alarm.sts_Category_1_Latched )
   END_RUNG wire#w1
   // the same network as SCL:
   "EM01".PackML_Sts.Alarm.cmd_Abort := "EM01".Alarm.sts_Category_0_Latched OR "EM01".Alarm.sts_Category_1_Latched;
END_REGION

REGION Network 5: Stop Command - controlled by category alarm 2 or 3
   RUNG wire#powerrail
      Contact( "EM01".Alarm.sts_Category_2_Latched )
      wire#w1
      Coil( "EM01".PackML_Sts.Alarm.cmd_Stop )
   END_RUNG
   RUNG wire#powerrail
      Contact( "EM01".Alarm.sts_Category_3_Latched )
   END_RUNG wire#w1
   // the same network as SCL:
   "EM01".PackML_Sts.Alarm.cmd_Stop := "EM01".Alarm.sts_Category_2_Latched OR "EM01".Alarm.sts_Category_3_Latched;
END_REGION

REGION Network 6: Hold Command - controlled by category alarm 7
   RUNG wire#powerrail
      Contact( "EM01".Alarm.sts_Category_7_NotLatched )
      Coil( "EM01".PackML_Sts.Alarm.cmd_Hold )
   END_RUNG
   // the same network as SCL:
   "EM01".PackML_Sts.Alarm.cmd_Hold := "EM01".Alarm.sts_Category_7_NotLatched;
END_REGION

REGION Network 7: UnHold Command - controlled by category alarm 7
   RUNG wire#powerrail
      Contact( "PackML".Sts.State.Held )
      I_Contact( "EM01".Alarm.sts_Category_7_NotLatched )
      Coil( "EM01".PackML_Sts.Alarm.cmd_UnHold )
   END_RUNG
   // the same network as SCL:
   "EM01".PackML_Sts.Alarm.cmd_UnHold := "PackML".Sts.State.Held AND NOT "EM01".Alarm.sts_Category_7_NotLatched;
END_REGION

REGION Network 8: Suspend Command - controlled by category alarm 8 or 9
   RUNG wire#powerrail
      Contact( "EM01".Alarm.sts_Category_8_NotLatched )
      wire#w1
      Coil( "EM01".PackML_Sts.Alarm.cmd_Suspend )
   END_RUNG
   RUNG wire#powerrail
      Contact( "EM01".Alarm.sts_Category_9_NotLatched )
   END_RUNG wire#w1
   // the same network as SCL:
   "EM01".PackML_Sts.Alarm.cmd_Suspend := "EM01".Alarm.sts_Category_8_NotLatched OR "EM01".Alarm.sts_Category_9_NotLatched;
END_REGION

REGION Network 9: UnSuspend Command - controlled by cleared category alarm 8 or 9
   RUNG wire#powerrail
      Contact( "PackML".Sts.State.Suspended )
      I_Contact( "EM01".Alarm.sts_Category_8_NotLatched )
      I_Contact( "EM01".Alarm.sts_Category_9_NotLatched )
      Coil( "EM01".PackML_Sts.Alarm.cmd_UnSuspend )
   END_RUNG
   // the same network as SCL:
   "EM01".PackML_Sts.Alarm.cmd_UnSuspend := "PackML".Sts.State.Suspended AND NOT "EM01".Alarm.sts_Category_8_NotLatched AND NOT "EM01".Alarm.sts_Category_9_NotLatched;
END_REGION

REGION Network 10: Clearing SC Command - controlled by cleared category alarm 0 or 1
   RUNG wire#powerrail
      Contact( "PackML".Sts.State.Clearing )
      I_Contact( "EM01".Alarm.sts_Category_0_Latched )
      I_Contact( "EM01".Alarm.sts_Category_1_Latched )
      Coil( "EM01".PackML_Sts.Alarm.sts_Clearing_SC )
   END_RUNG
   // the same network as SCL:
   "EM01".PackML_Sts.Alarm.sts_Clearing_SC := "PackML".Sts.State.Clearing AND NOT "EM01".Alarm.sts_Category_0_Latched AND NOT "EM01".Alarm.sts_Category_1_Latched;
END_REGION

REGION Network 11: Resetting SC Command - controlled by cleared category alarm 0-3
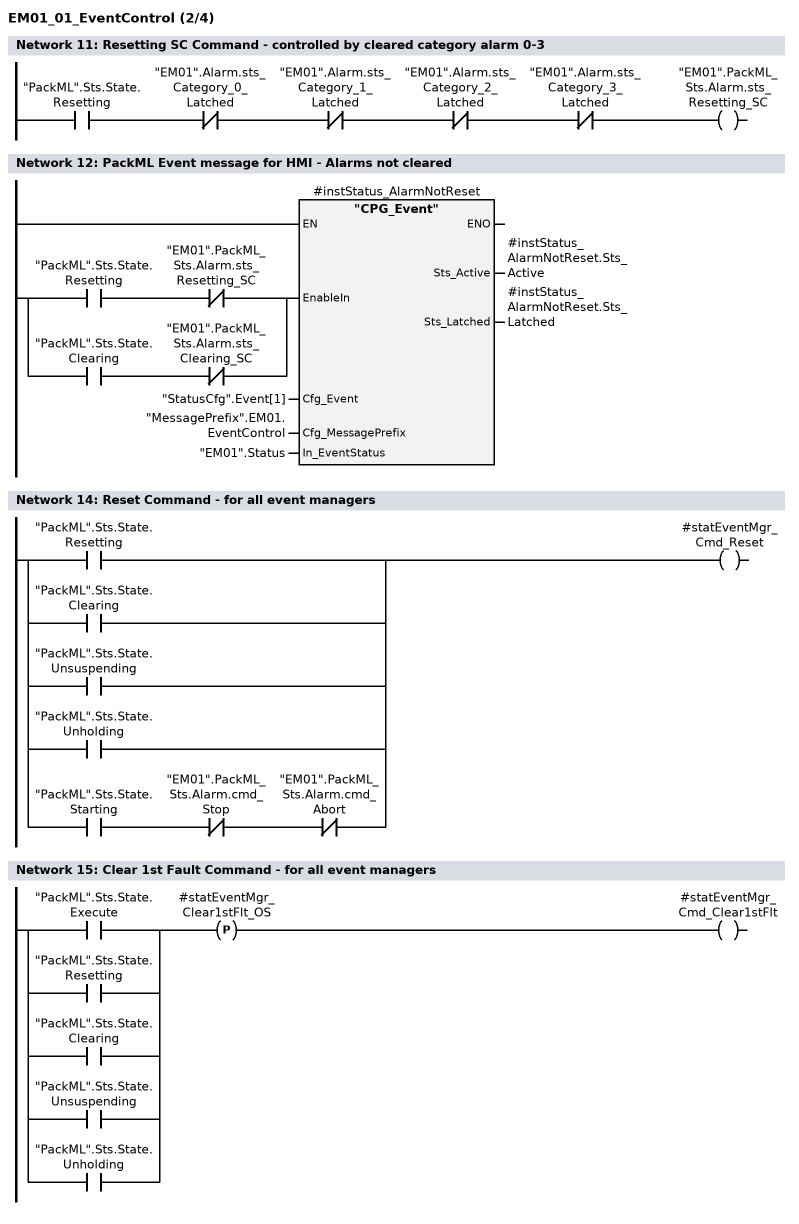
   RUNG wire#powerrail
      Contact( "PackML".Sts.State.Resetting )
      I_Contact( "EM01".Alarm.sts_Category_0_Latched )
      I_Contact( "EM01".Alarm.sts_Category_1_Latched )
      I_Contact( "EM01".Alarm.sts_Category_2_Latched )
      I_Contact( "EM01".Alarm.sts_Category_3_Latched )
      Coil( "EM01".PackML_Sts.Alarm.sts_Resetting_SC )
   END_RUNG
   // the same network as SCL:
   "EM01".PackML_Sts.Alarm.sts_Resetting_SC := "PackML".Sts.State.Resetting AND NOT "EM01".Alarm.sts_Category_0_Latched AND NOT "EM01".Alarm.sts_Category_1_Latched AND NOT "EM01".Alarm.sts_Category_2_Latched AND NOT "EM01".Alarm.sts_Category_3_Latched;
END_REGION

REGION Network 12: PackML Event message for HMI - Alarms not cleared
   RUNG wire#powerrail
      #instStatus_AlarmNotReset(EnableIn := wire#w1, Cfg_Event := "StatusCfg".Event[1], Cfg_MessagePrefix := "MessagePrefix".EM01.EventControl, In_EventStatus := "EM01".Status, Sts_Active => #instStatus_AlarmNotReset.Sts_Active, Sts_Latched => #instStatus_AlarmNotReset.Sts_Latched)
   END_RUNG
   RUNG wire#powerrail
      Contact( "PackML".Sts.State.Resetting )
      I_Contact( "EM01".PackML_Sts.Alarm.sts_Resetting_SC )
   END_RUNG wire#w1
   RUNG wire#powerrail
      Contact( "PackML".Sts.State.Clearing )
      I_Contact( "EM01".PackML_Sts.Alarm.sts_Clearing_SC )
   END_RUNG wire#w1
   // the same network as SCL:
   #instStatus_AlarmNotReset(EnableIn := ("PackML".Sts.State.Resetting AND NOT "EM01".PackML_Sts.Alarm.sts_Resetting_SC) OR ("PackML".Sts.State.Clearing AND NOT "EM01".PackML_Sts.Alarm.sts_Clearing_SC),   // "CPG_Event"
                           Cfg_Event := "StatusCfg".Event[1],
                           Cfg_MessagePrefix := "MessagePrefix".EM01.EventControl,
                           In_EventStatus := "EM01".Status,
                           Sts_Active => #instStatus_AlarmNotReset.Sts_Active,
                           Sts_Latched => #instStatus_AlarmNotReset.Sts_Latched);
END_REGION

REGION Network 13: *** EVENT CONTROL MANAGERS ***
END_REGION

REGION Network 14: Reset Command - for all event managers
   RUNG wire#powerrail
      Contact( "PackML".Sts.State.Resetting )
      wire#w1
      Coil( #statEventMgr_Cmd_Reset )
   END_RUNG
   RUNG wire#powerrail
      Contact( "PackML".Sts.State.Clearing )
   END_RUNG wire#w1
   RUNG wire#powerrail
      Contact( "PackML".Sts.State.Unsuspending )
   END_RUNG wire#w1
   RUNG wire#powerrail
      Contact( "PackML".Sts.State.Unholding )
   END_RUNG wire#w1
   RUNG wire#powerrail
      Contact( "PackML".Sts.State.Starting )
      I_Contact( "EM01".PackML_Sts.Alarm.cmd_Stop )
      I_Contact( "EM01".PackML_Sts.Alarm.cmd_Abort )
   END_RUNG wire#w1
   // the same network as SCL:
   #statEventMgr_Cmd_Reset := "PackML".Sts.State.Resetting OR "PackML".Sts.State.Clearing OR "PackML".Sts.State.Unsuspending OR "PackML".Sts.State.Unholding OR ("PackML".Sts.State.Starting AND NOT "EM01".PackML_Sts.Alarm.cmd_Stop AND NOT "EM01".PackML_Sts.Alarm.cmd_Abort);
END_REGION

REGION Network 15: Clear 1st Fault Command - for all event managers
   RUNG wire#powerrail
      Contact( "PackML".Sts.State.Execute )
      wire#w1
      P_Trig( #statEventMgr_Clear1stFlt_OS )
      Coil( #statEventMgr_Cmd_Clear1stFlt )
   END_RUNG
   RUNG wire#powerrail
      Contact( "PackML".Sts.State.Resetting )
   END_RUNG wire#w1
   RUNG wire#powerrail
      Contact( "PackML".Sts.State.Clearing )
   END_RUNG wire#w1
   RUNG wire#powerrail
      Contact( "PackML".Sts.State.Unsuspending )
   END_RUNG wire#w1
   RUNG wire#powerrail
      Contact( "PackML".Sts.State.Unholding )
   END_RUNG wire#w1
   // the same network as SCL:
   #_w1 := "PackML".Sts.State.Execute OR "PackML".Sts.State.Resetting OR "PackML".Sts.State.Clearing OR "PackML".Sts.State.Unsuspending OR "PackML".Sts.State.Unholding;
   #_w2 := #_w1 AND NOT #statEventMgr_Clear1stFlt_OS;   // rising edge
   #statEventMgr_Clear1stFlt_OS := #_w1;
   #statEventMgr_Cmd_Clear1stFlt := #_w2;
END_REGION

REGION Network 16: Call the Event Manager logic for EM alarms
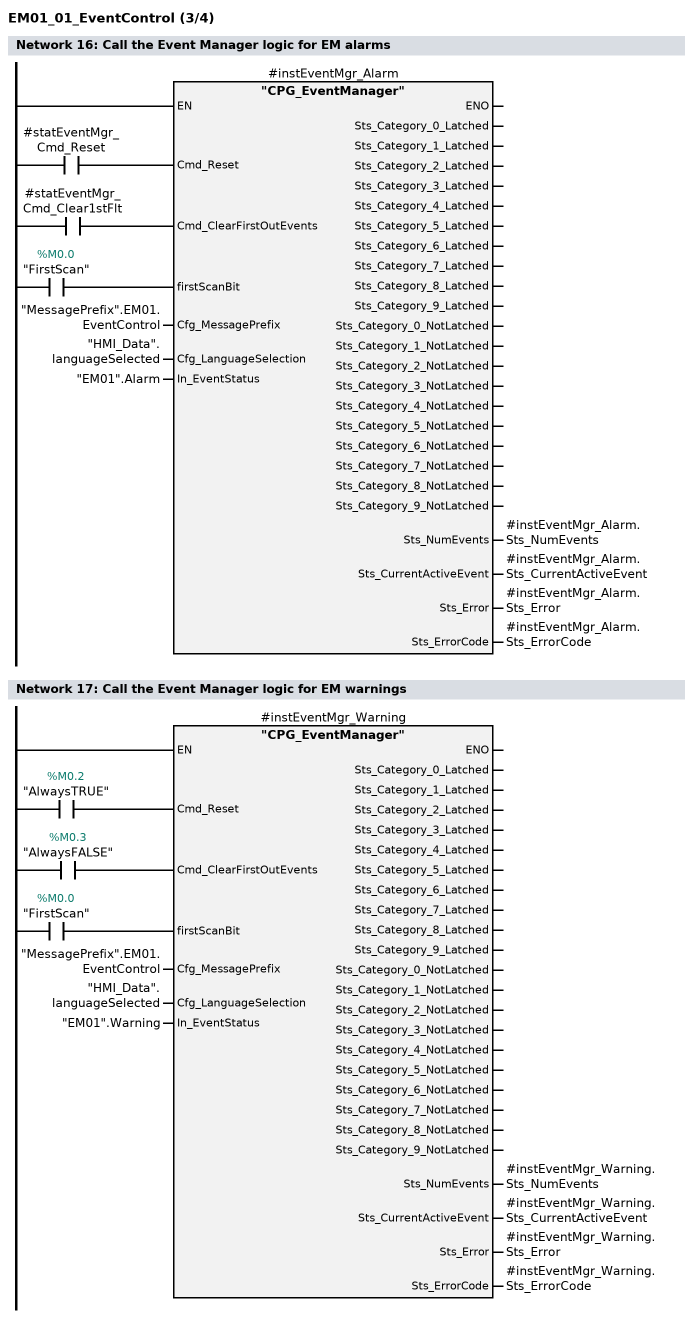
   RUNG wire#powerrail
      #instEventMgr_Alarm(Cmd_Reset := wire#w1, Cmd_ClearFirstOutEvents := wire#w2, firstScanBit := wire#w3, Cfg_MessagePrefix := "MessagePrefix".EM01.EventControl, Cfg_LanguageSelection := "HMI_Data".languageSelected, In_EventStatus := "EM01".Alarm, Sts_Category_0_Latched =>, Sts_Category_1_Latched =>, Sts_Category_2_Latched =>, Sts_Category_3_Latched =>, Sts_Category_4_Latched =>, Sts_Category_5_Latched =>, Sts_Category_6_Latched =>, Sts_Category_7_Latched =>, Sts_Category_8_Latched =>, Sts_Category_9_Latched =>, Sts_Category_0_NotLatched =>, Sts_Category_1_NotLatched =>, Sts_Category_2_NotLatched =>, Sts_Category_3_NotLatched =>, Sts_Category_4_NotLatched =>, Sts_Category_5_NotLatched =>, Sts_Category_6_NotLatched =>, Sts_Category_7_NotLatched =>, Sts_Category_8_NotLatched =>, Sts_Category_9_NotLatched =>, Sts_NumEvents => #instEventMgr_Alarm.Sts_NumEvents, Sts_CurrentActiveEvent => #instEventMgr_Alarm.Sts_CurrentActiveEvent, Sts_Error => #instEventMgr_Alarm.Sts_Error, Sts_ErrorCode => #instEventMgr_Alarm.Sts_ErrorCode)
   END_RUNG
   RUNG wire#powerrail
      Contact( #statEventMgr_Cmd_Reset )
   END_RUNG wire#w1
   RUNG wire#powerrail
      Contact( #statEventMgr_Cmd_Clear1stFlt )
   END_RUNG wire#w2
   RUNG wire#powerrail
      Contact( "FirstScan" )
   END_RUNG wire#w3
   // the same network as SCL:
   #instEventMgr_Alarm(Cmd_Reset := #statEventMgr_Cmd_Reset,   // "CPG_EventManager"
                       Cmd_ClearFirstOutEvents := #statEventMgr_Cmd_Clear1stFlt,
                       firstScanBit := "FirstScan",
                       Cfg_MessagePrefix := "MessagePrefix".EM01.EventControl,
                       Cfg_LanguageSelection := "HMI_Data".languageSelected,
                       In_EventStatus := "EM01".Alarm,
                       Sts_NumEvents => #instEventMgr_Alarm.Sts_NumEvents,
                       Sts_CurrentActiveEvent => #instEventMgr_Alarm.Sts_CurrentActiveEvent,
                       Sts_Error => #instEventMgr_Alarm.Sts_Error,
                       Sts_ErrorCode => #instEventMgr_Alarm.Sts_ErrorCode);
END_REGION

REGION Network 17: Call the Event Manager logic for EM warnings
   RUNG wire#powerrail
      #instEventMgr_Warning(Cmd_Reset := wire#w1, Cmd_ClearFirstOutEvents := wire#w2, firstScanBit := wire#w3, Cfg_MessagePrefix := "MessagePrefix".EM01.EventControl, Cfg_LanguageSelection := "HMI_Data".languageSelected, In_EventStatus := "EM01".Warning, Sts_Category_0_Latched =>, Sts_Category_1_Latched =>, Sts_Category_2_Latched =>, Sts_Category_3_Latched =>, Sts_Category_4_Latched =>, Sts_Category_5_Latched =>, Sts_Category_6_Latched =>, Sts_Category_7_Latched =>, Sts_Category_8_Latched =>, Sts_Category_9_Latched =>, Sts_Category_0_NotLatched =>, Sts_Category_1_NotLatched =>, Sts_Category_2_NotLatched =>, Sts_Category_3_NotLatched =>, Sts_Category_4_NotLatched =>, Sts_Category_5_NotLatched =>, Sts_Category_6_NotLatched =>, Sts_Category_7_NotLatched =>, Sts_Category_8_NotLatched =>, Sts_Category_9_NotLatched =>, Sts_NumEvents => #instEventMgr_Warning.Sts_NumEvents, Sts_CurrentActiveEvent => #instEventMgr_Warning.Sts_CurrentActiveEvent, Sts_Error => #instEventMgr_Warning.Sts_Error, Sts_ErrorCode => #instEventMgr_Warning.Sts_ErrorCode)
   END_RUNG
   RUNG wire#powerrail
      Contact( "AlwaysTRUE" )
   END_RUNG wire#w1
   RUNG wire#powerrail
      Contact( "AlwaysFALSE" )
   END_RUNG wire#w2
   RUNG wire#powerrail
      Contact( "FirstScan" )
   END_RUNG wire#w3
   // the same network as SCL:
   #instEventMgr_Warning(Cmd_Reset := "AlwaysTRUE",   // "CPG_EventManager"
                         Cmd_ClearFirstOutEvents := "AlwaysFALSE",
                         firstScanBit := "FirstScan",
                         Cfg_MessagePrefix := "MessagePrefix".EM01.EventControl,
                         Cfg_LanguageSelection := "HMI_Data".languageSelected,
                         In_EventStatus := "EM01".Warning,
                         Sts_NumEvents => #instEventMgr_Warning.Sts_NumEvents,
                         Sts_CurrentActiveEvent => #instEventMgr_Warning.Sts_CurrentActiveEvent,
                         Sts_Error => #instEventMgr_Warning.Sts_Error,
                         Sts_ErrorCode => #instEventMgr_Warning.Sts_ErrorCode);
END_REGION

REGION Network 18: Call the Event Manager logic for EM status
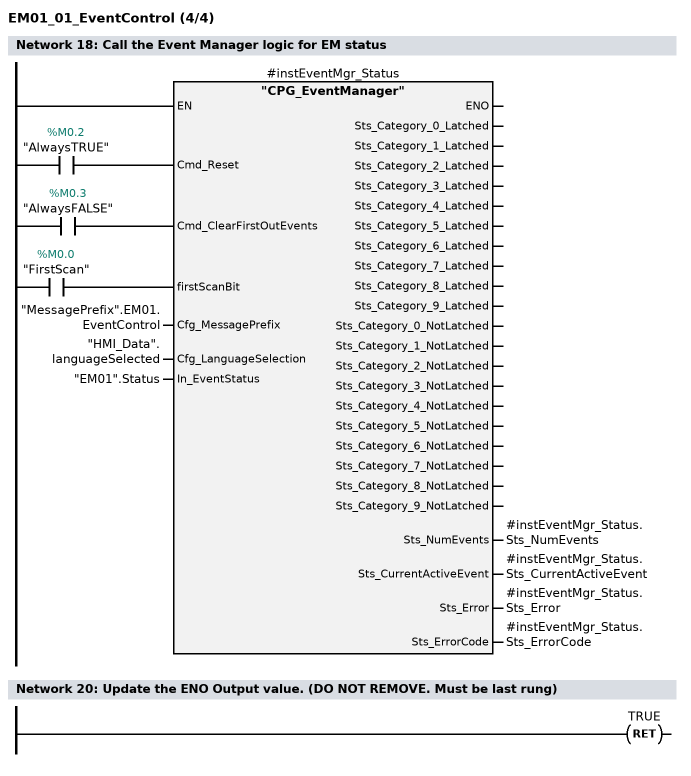
   RUNG wire#powerrail
      #instEventMgr_Status(Cmd_Reset := wire#w1, Cmd_ClearFirstOutEvents := wire#w2, firstScanBit := wire#w3, Cfg_MessagePrefix := "MessagePrefix".EM01.EventControl, Cfg_LanguageSelection := "HMI_Data".languageSelected, In_EventStatus := "EM01".Status, Sts_Category_0_Latched =>, Sts_Category_1_Latched =>, Sts_Category_2_Latched =>, Sts_Category_3_Latched =>, Sts_Category_4_Latched =>, Sts_Category_5_Latched =>, Sts_Category_6_Latched =>, Sts_Category_7_Latched =>, Sts_Category_8_Latched =>, Sts_Category_9_Latched =>, Sts_Category_0_NotLatched =>, Sts_Category_1_NotLatched =>, Sts_Category_2_NotLatched =>, Sts_Category_3_NotLatched =>, Sts_Category_4_NotLatched =>, Sts_Category_5_NotLatched =>, Sts_Category_6_NotLatched =>, Sts_Category_7_NotLatched =>, Sts_Category_8_NotLatched =>, Sts_Category_9_NotLatched =>, Sts_NumEvents => #instEventMgr_Status.Sts_NumEvents, Sts_CurrentActiveEvent => #instEventMgr_Status.Sts_CurrentActiveEvent, Sts_Error => #instEventMgr_Status.Sts_Error, Sts_ErrorCode => #instEventMgr_Status.Sts_ErrorCode)
   END_RUNG
   RUNG wire#powerrail
      Contact( "AlwaysTRUE" )
   END_RUNG wire#w1
   RUNG wire#powerrail
      Contact( "AlwaysFALSE" )
   END_RUNG wire#w2
   RUNG wire#powerrail
      Contact( "FirstScan" )
   END_RUNG wire#w3
   // the same network as SCL:
   #instEventMgr_Status(Cmd_Reset := "AlwaysTRUE",   // "CPG_EventManager"
                        Cmd_ClearFirstOutEvents := "AlwaysFALSE",
                        firstScanBit := "FirstScan",
                        Cfg_MessagePrefix := "MessagePrefix".EM01.EventControl,
                        Cfg_LanguageSelection := "HMI_Data".languageSelected,
                        In_EventStatus := "EM01".Status,
                        Sts_NumEvents => #instEventMgr_Status.Sts_NumEvents,
                        Sts_CurrentActiveEvent => #instEventMgr_Status.Sts_CurrentActiveEvent,
                        Sts_Error => #instEventMgr_Status.Sts_Error,
                        Sts_ErrorCode => #instEventMgr_Status.Sts_ErrorCode);
END_REGION

REGION Network 20: Update the ENO Output value. (DO NOT REMOVE. Must be last rung)
   RUNG wire#powerrail
      ReturnCoil( TRUE )
   END_RUNG
   // the same network as SCL:
   ENO := TRUE;
   RETURN;
END_REGION
END_FUNCTION_BLOCK

FUNCTION_BLOCK "EM01_02_PackML_ModuleSum"   // FB31662, LAD
TITLE = EM01_02_PackML_ModuleSum
{ S7_Optimized_Access := 'TRUE' }
AUTHOR : tech.team.motioncontrol@siemens.com
FAMILY : CPG
VERSION : 1.1
// Support: tech.team.motioncontrol@siemens.com
// stored: AutoNumber true, IsIECCheckEnabled false, IsRetainMemResEnabled false, MemoryReserve 100, SetENOAutomatically false, UDAEnableTagReadback false
   VAR
      statDummyBool { ExternalAccessible := 'False'; ExternalVisible := 'False'; ExternalWritable := 'False'} : Bool;   // dummy bool - placeholder
   END_VAR
BEGIN

REGION Network 1: EM - Reset Command
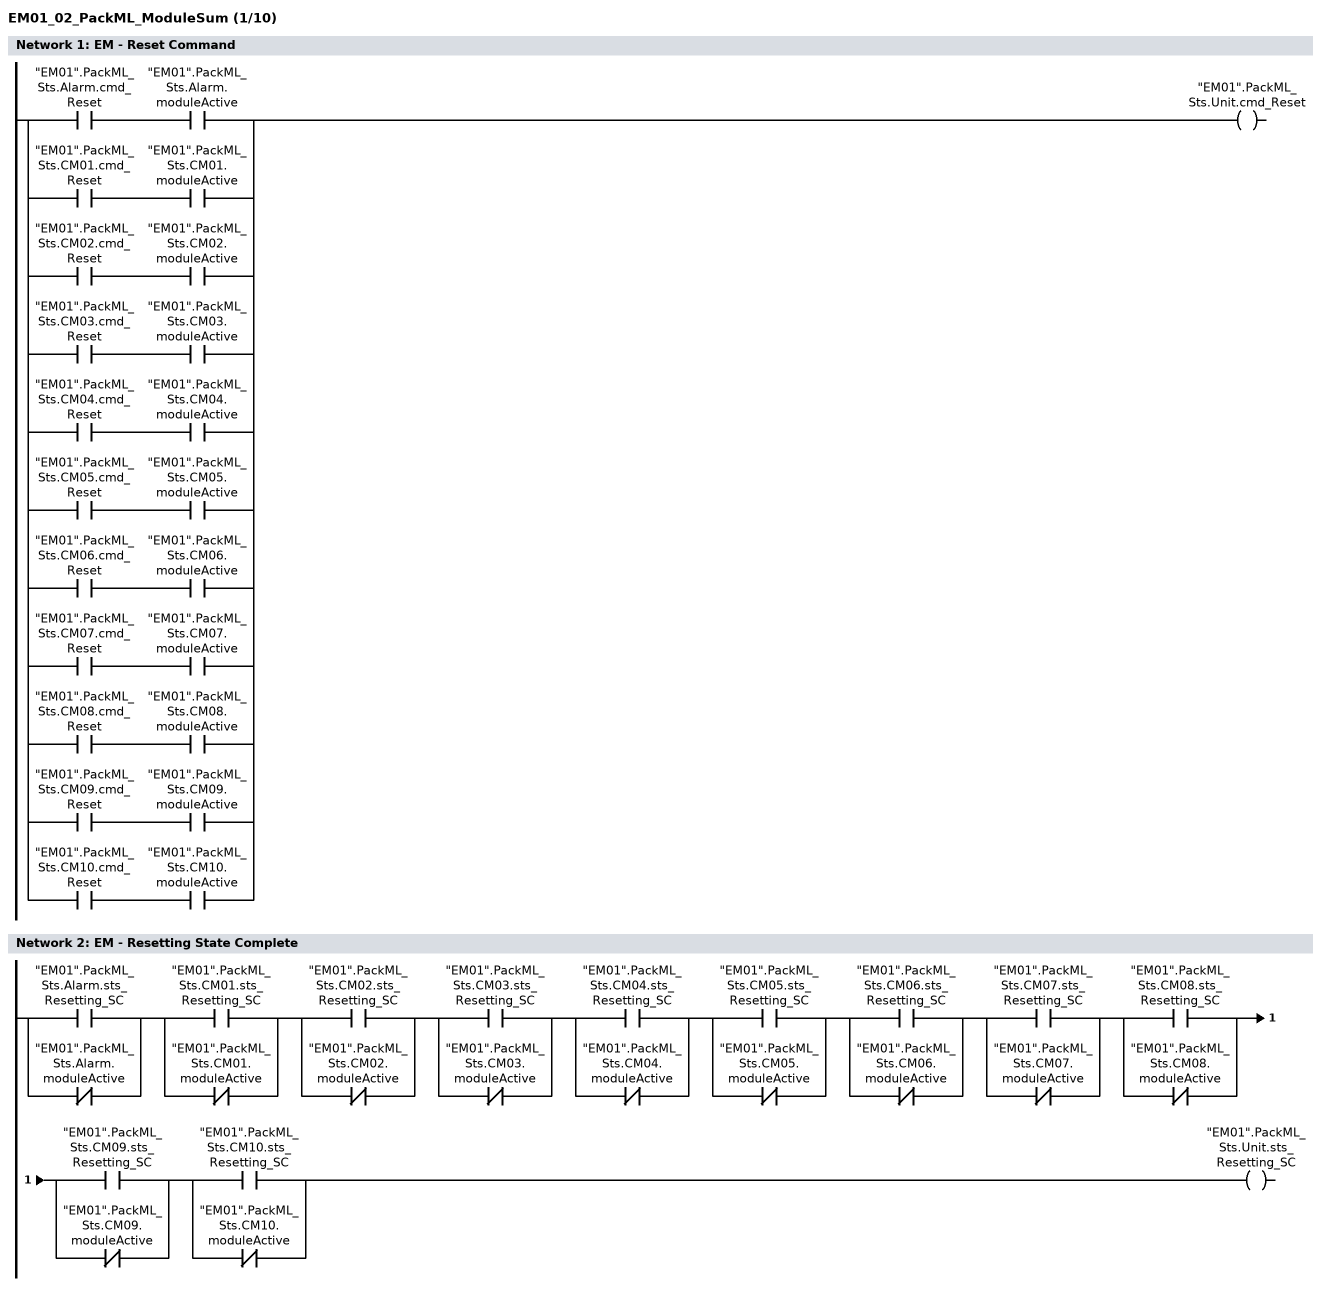
   RUNG wire#powerrail
      Contact( "EM01".PackML_Sts.Alarm.cmd_Reset )
      Contact( "EM01".PackML_Sts.Alarm.moduleActive )
      wire#w1
      Coil( "EM01".PackML_Sts.Unit.cmd_Reset )
   END_RUNG
   RUNG wire#powerrail
      Contact( "EM01".PackML_Sts.CM01.cmd_Reset )
      Contact( "EM01".PackML_Sts.CM01.moduleActive )
   END_RUNG wire#w1
   RUNG wire#powerrail
      Contact( "EM01".PackML_Sts.CM02.cmd_Reset )
      Contact( "EM01".PackML_Sts.CM02.moduleActive )
   END_RUNG wire#w1
   RUNG wire#powerrail
      Contact( "EM01".PackML_Sts.CM03.cmd_Reset )
      Contact( "EM01".PackML_Sts.CM03.moduleActive )
   END_RUNG wire#w1
   RUNG wire#powerrail
      Contact( "EM01".PackML_Sts.CM04.cmd_Reset )
      Contact( "EM01".PackML_Sts.CM04.moduleActive )
   END_RUNG wire#w1
   RUNG wire#powerrail
      Contact( "EM01".PackML_Sts.CM05.cmd_Reset )
      Contact( "EM01".PackML_Sts.CM05.moduleActive )
   END_RUNG wire#w1
   RUNG wire#powerrail
      Contact( "EM01".PackML_Sts.CM06.cmd_Reset )
      Contact( "EM01".PackML_Sts.CM06.moduleActive )
   END_RUNG wire#w1
   RUNG wire#powerrail
      Contact( "EM01".PackML_Sts.CM07.cmd_Reset )
      Contact( "EM01".PackML_Sts.CM07.moduleActive )
   END_RUNG wire#w1
   RUNG wire#powerrail
      Contact( "EM01".PackML_Sts.CM08.cmd_Reset )
      Contact( "EM01".PackML_Sts.CM08.moduleActive )
   END_RUNG wire#w1
   RUNG wire#powerrail
      Contact( "EM01".PackML_Sts.CM09.cmd_Reset )
      Contact( "EM01".PackML_Sts.CM09.moduleActive )
   END_RUNG wire#w1
   RUNG wire#powerrail
      Contact( "EM01".PackML_Sts.CM10.cmd_Reset )
      Contact( "EM01".PackML_Sts.CM10.moduleActive )
   END_RUNG wire#w1
   // the same network as SCL:
   "EM01".PackML_Sts.Unit.cmd_Reset := ("EM01".PackML_Sts.Alarm.cmd_Reset AND "EM01".PackML_Sts.Alarm.moduleActive) OR ("EM01".PackML_Sts.CM01.cmd_Reset AND "EM01".PackML_Sts.CM01.moduleActive) OR ("EM01".PackML_Sts.CM02.cmd_Reset AND "EM01".PackML_Sts.CM02.moduleActive) OR ("EM01".PackML_Sts.CM03.cmd_Reset AND "EM01".PackML_Sts.CM03.moduleActive) OR ("EM01".PackML_Sts.CM04.cmd_Reset AND "EM01".PackML_Sts.CM04.moduleActive) OR ("EM01".PackML_Sts.CM05.cmd_Reset AND "EM01".PackML_Sts.CM05.moduleActive) OR ("EM01".PackML_Sts.CM06.cmd_Reset AND "EM01".PackML_Sts.CM06.moduleActive) OR ("EM01".PackML_Sts.CM07.cmd_Reset AND "EM01".PackML_Sts.CM07.moduleActive) OR ("EM01".PackML_Sts.CM08.cmd_Reset AND "EM01".PackML_Sts.CM08.moduleActive) OR ("EM01".PackML_Sts.CM09.cmd_Reset AND "EM01".PackML_Sts.CM09.moduleActive) OR ("EM01".PackML_Sts.CM10.cmd_Reset AND "EM01".PackML_Sts.CM10.moduleActive);
END_REGION

REGION Network 2: EM - Resetting State Complete
   RUNG wire#powerrail
      Contact( "EM01".PackML_Sts.Alarm.sts_Resetting_SC )
      wire#w1
      Contact( "EM01".PackML_Sts.CM01.sts_Resetting_SC )
      wire#w2
      Contact( "EM01".PackML_Sts.CM02.sts_Resetting_SC )
      wire#w3
      Contact( "EM01".PackML_Sts.CM03.sts_Resetting_SC )
      wire#w4
      Contact( "EM01".PackML_Sts.CM04.sts_Resetting_SC )
      wire#w5
      Contact( "EM01".PackML_Sts.CM05.sts_Resetting_SC )
      wire#w6
      Contact( "EM01".PackML_Sts.CM06.sts_Resetting_SC )
      wire#w7
      Contact( "EM01".PackML_Sts.CM07.sts_Resetting_SC )
      wire#w8
      Contact( "EM01".PackML_Sts.CM08.sts_Resetting_SC )
      wire#w9
      Contact( "EM01".PackML_Sts.CM09.sts_Resetting_SC )
      wire#w10
      Contact( "EM01".PackML_Sts.CM10.sts_Resetting_SC )
      wire#w11
      Coil( "EM01".PackML_Sts.Unit.sts_Resetting_SC )
   END_RUNG
   RUNG wire#powerrail
      I_Contact( "EM01".PackML_Sts.Alarm.moduleActive )
   END_RUNG wire#w1
   RUNG wire#w1
      I_Contact( "EM01".PackML_Sts.CM01.moduleActive )
   END_RUNG wire#w2
   RUNG wire#w2
      I_Contact( "EM01".PackML_Sts.CM02.moduleActive )
   END_RUNG wire#w3
   RUNG wire#w3
      I_Contact( "EM01".PackML_Sts.CM03.moduleActive )
   END_RUNG wire#w4
   RUNG wire#w4
      I_Contact( "EM01".PackML_Sts.CM04.moduleActive )
   END_RUNG wire#w5
   RUNG wire#w5
      I_Contact( "EM01".PackML_Sts.CM05.moduleActive )
   END_RUNG wire#w6
   RUNG wire#w6
      I_Contact( "EM01".PackML_Sts.CM06.moduleActive )
   END_RUNG wire#w7
   RUNG wire#w7
      I_Contact( "EM01".PackML_Sts.CM07.moduleActive )
   END_RUNG wire#w8
   RUNG wire#w8
      I_Contact( "EM01".PackML_Sts.CM08.moduleActive )
   END_RUNG wire#w9
   RUNG wire#w9
      I_Contact( "EM01".PackML_Sts.CM09.moduleActive )
   END_RUNG wire#w10
   RUNG wire#w10
      I_Contact( "EM01".PackML_Sts.CM10.moduleActive )
   END_RUNG wire#w11
   // the same network as SCL:
   "EM01".PackML_Sts.Unit.sts_Resetting_SC := ("EM01".PackML_Sts.Alarm.sts_Resetting_SC OR NOT "EM01".PackML_Sts.Alarm.moduleActive) AND ("EM01".PackML_Sts.CM01.sts_Resetting_SC OR NOT "EM01".PackML_Sts.CM01.moduleActive) AND ("EM01".PackML_Sts.CM02.sts_Resetting_SC OR NOT "EM01".PackML_Sts.CM02.moduleActive) AND ("EM01".PackML_Sts.CM03.sts_Resetting_SC OR NOT "EM01".PackML_Sts.CM03.moduleActive) AND ("EM01".PackML_Sts.CM04.sts_Resetting_SC OR NOT "EM01".PackML_Sts.CM04.moduleActive) AND ("EM01".PackML_Sts.CM05.sts_Resetting_SC OR NOT "EM01".PackML_Sts.CM05.moduleActive) AND ("EM01".PackML_Sts.CM06.sts_Resetting_SC OR NOT "EM01".PackML_Sts.CM06.moduleActive) AND ("EM01".PackML_Sts.CM07.sts_Resetting_SC OR NOT "EM01".PackML_Sts.CM07.moduleActive) AND ("EM01".PackML_Sts.CM08.sts_Resetting_SC OR NOT "EM01".PackML_Sts.CM08.moduleActive) AND ("EM01".PackML_Sts.CM09.sts_Resetting_SC OR NOT "EM01".PackML_Sts.CM09.moduleActive) AND ("EM01".PackML_Sts.CM10.sts_Resetting_SC OR NOT "EM01".PackML_Sts.CM10.moduleActive);
END_REGION

REGION Network 3: EM - Start Command
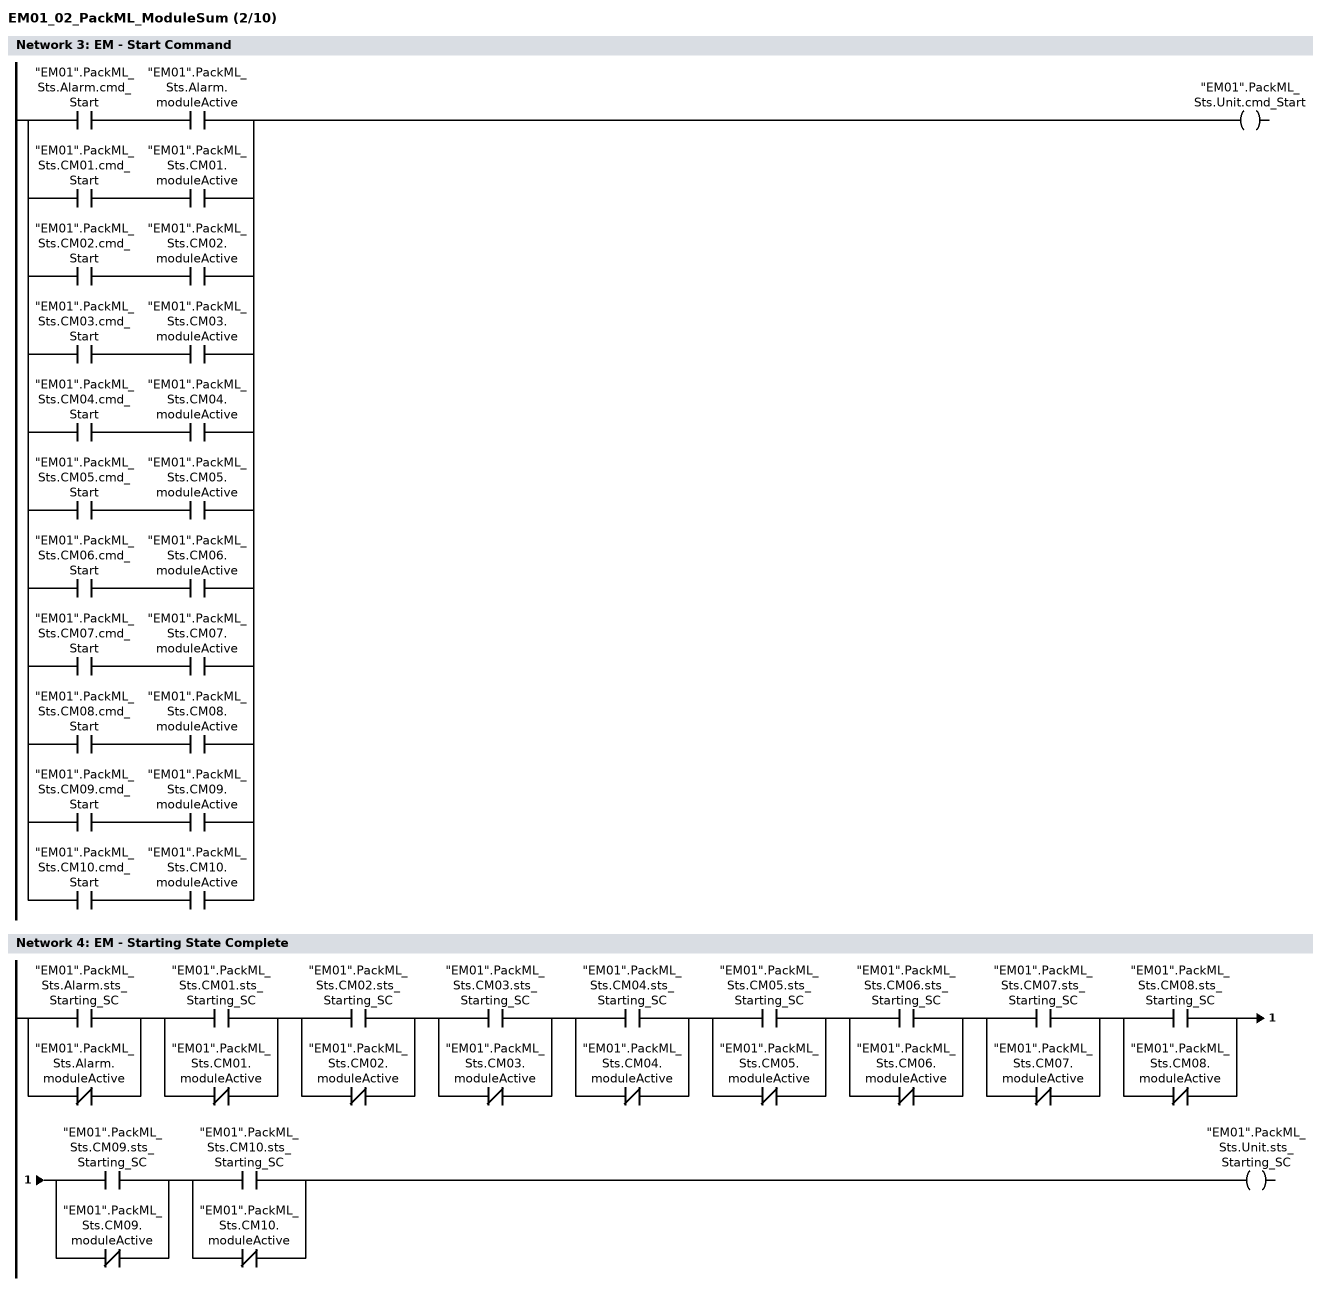
   RUNG wire#powerrail
      Contact( "EM01".PackML_Sts.Alarm.cmd_Start )
      Contact( "EM01".PackML_Sts.Alarm.moduleActive )
      wire#w1
      Coil( "EM01".PackML_Sts.Unit.cmd_Start )
   END_RUNG
   RUNG wire#powerrail
      Contact( "EM01".PackML_Sts.CM01.cmd_Start )
      Contact( "EM01".PackML_Sts.CM01.moduleActive )
   END_RUNG wire#w1
   RUNG wire#powerrail
      Contact( "EM01".PackML_Sts.CM02.cmd_Start )
      Contact( "EM01".PackML_Sts.CM02.moduleActive )
   END_RUNG wire#w1
   RUNG wire#powerrail
      Contact( "EM01".PackML_Sts.CM03.cmd_Start )
      Contact( "EM01".PackML_Sts.CM03.moduleActive )
   END_RUNG wire#w1
   RUNG wire#powerrail
      Contact( "EM01".PackML_Sts.CM04.cmd_Start )
      Contact( "EM01".PackML_Sts.CM04.moduleActive )
   END_RUNG wire#w1
   RUNG wire#powerrail
      Contact( "EM01".PackML_Sts.CM05.cmd_Start )
      Contact( "EM01".PackML_Sts.CM05.moduleActive )
   END_RUNG wire#w1
   RUNG wire#powerrail
      Contact( "EM01".PackML_Sts.CM06.cmd_Start )
      Contact( "EM01".PackML_Sts.CM06.moduleActive )
   END_RUNG wire#w1
   RUNG wire#powerrail
      Contact( "EM01".PackML_Sts.CM07.cmd_Start )
      Contact( "EM01".PackML_Sts.CM07.moduleActive )
   END_RUNG wire#w1
   RUNG wire#powerrail
      Contact( "EM01".PackML_Sts.CM08.cmd_Start )
      Contact( "EM01".PackML_Sts.CM08.moduleActive )
   END_RUNG wire#w1
   RUNG wire#powerrail
      Contact( "EM01".PackML_Sts.CM09.cmd_Start )
      Contact( "EM01".PackML_Sts.CM09.moduleActive )
   END_RUNG wire#w1
   RUNG wire#powerrail
      Contact( "EM01".PackML_Sts.CM10.cmd_Start )
      Contact( "EM01".PackML_Sts.CM10.moduleActive )
   END_RUNG wire#w1
   // the same network as SCL:
   "EM01".PackML_Sts.Unit.cmd_Start := ("EM01".PackML_Sts.Alarm.cmd_Start AND "EM01".PackML_Sts.Alarm.moduleActive) OR ("EM01".PackML_Sts.CM01.cmd_Start AND "EM01".PackML_Sts.CM01.moduleActive) OR ("EM01".PackML_Sts.CM02.cmd_Start AND "EM01".PackML_Sts.CM02.moduleActive) OR ("EM01".PackML_Sts.CM03.cmd_Start AND "EM01".PackML_Sts.CM03.moduleActive) OR ("EM01".PackML_Sts.CM04.cmd_Start AND "EM01".PackML_Sts.CM04.moduleActive) OR ("EM01".PackML_Sts.CM05.cmd_Start AND "EM01".PackML_Sts.CM05.moduleActive) OR ("EM01".PackML_Sts.CM06.cmd_Start AND "EM01".PackML_Sts.CM06.moduleActive) OR ("EM01".PackML_Sts.CM07.cmd_Start AND "EM01".PackML_Sts.CM07.moduleActive) OR ("EM01".PackML_Sts.CM08.cmd_Start AND "EM01".PackML_Sts.CM08.moduleActive) OR ("EM01".PackML_Sts.CM09.cmd_Start AND "EM01".PackML_Sts.CM09.moduleActive) OR ("EM01".PackML_Sts.CM10.cmd_Start AND "EM01".PackML_Sts.CM10.moduleActive);
END_REGION

